// TIA Portal V17 export
// export: Created 2025-07-01T14:26:11.2068104Z, ExportSetting WithDefaults, DisplayName Totally Integrated Automation Portal, DisplayVersion V17 Update 8, DisplayName TIA Portal Openness, DisplayVersion V17 Update 8, DisplayName TIA Portal Version Control Interface, DisplayVersion V17, DisplayName SINAMICS Startdrive Advanced, DisplayVersion V17 SP2, DisplayName SINAMICS Startdrive G110M, G120, G120C, G120D, G120P, G115D, DisplayVersion V17 SP2, DisplayName SINAMICS Startdrive G130, G150, S120, S150, SINAMICS MV, S210, DisplayVersion V17 SP2, DisplayName STEP 7 Professional, DisplayVersion V17 Update 8, DisplayName SINUMERIK ONE STEP 7 Toolbox, DisplayVersion V17 Update 12, DisplayName SINUMERIK ONE PLC Basic Program Plus, DisplayVersion V17 Update 12, DisplayName SINUMERIK 840D sl STEP 7 Toolbox, DisplayVersion V17 Update 12, DisplayName STEP 7 Safety, DisplayVersion V17 Update 6, DisplayName WinCC Advanced, DisplayVersion V17 Update 8
FUNCTION "FC16014_METHOD_CALLS_U2_STA3_MEAS" : Void   // FC16014, LAD
{ S7_Optimized_Access := 'FALSE' }
VERSION : 0.1
// STATUS VALUES:
// 0 = IDLE
// 1 = CALIBRATING
// 2 = ANALYZING DISTANCE
// 3 = ANALYZING LAYER THICKNESS
// -1 = ERROR
// stored: AutoNumber false, IsIECCheckEnabled false, SetENOAutomatically false, UDAEnableTagReadback false
   VAR_TEMP
      AUX_WSTRING_PART_ID_STA3 : WString;
      AUX_WCHARS : Array[0..63] of WChar;
      index : Int;
      ALARM_AUX : Bool;
      TEMP_PULSE : Bool;
      STATUS_BLKMOV : Int;   // STATUS BLKMOV
      ZERO : Int;
   END_VAR
   VAR CONSTANT
      VERSIONS_MAJOR : UInt := 2;
      VERSIONS_MINOR : UInt;
      FC_NUMBER : DInt := 16014;
   END_VAR
   VAR_TEMP   // added for the SCL form of the ladder/FBD networks
      _w1 : Bool;
      _w2 : Bool;
      _w3 : Bool;
      _s5time1 : S5Time;
      _w4 : Bool;
   END_VAR
BEGIN

REGION Network 1: ZERO
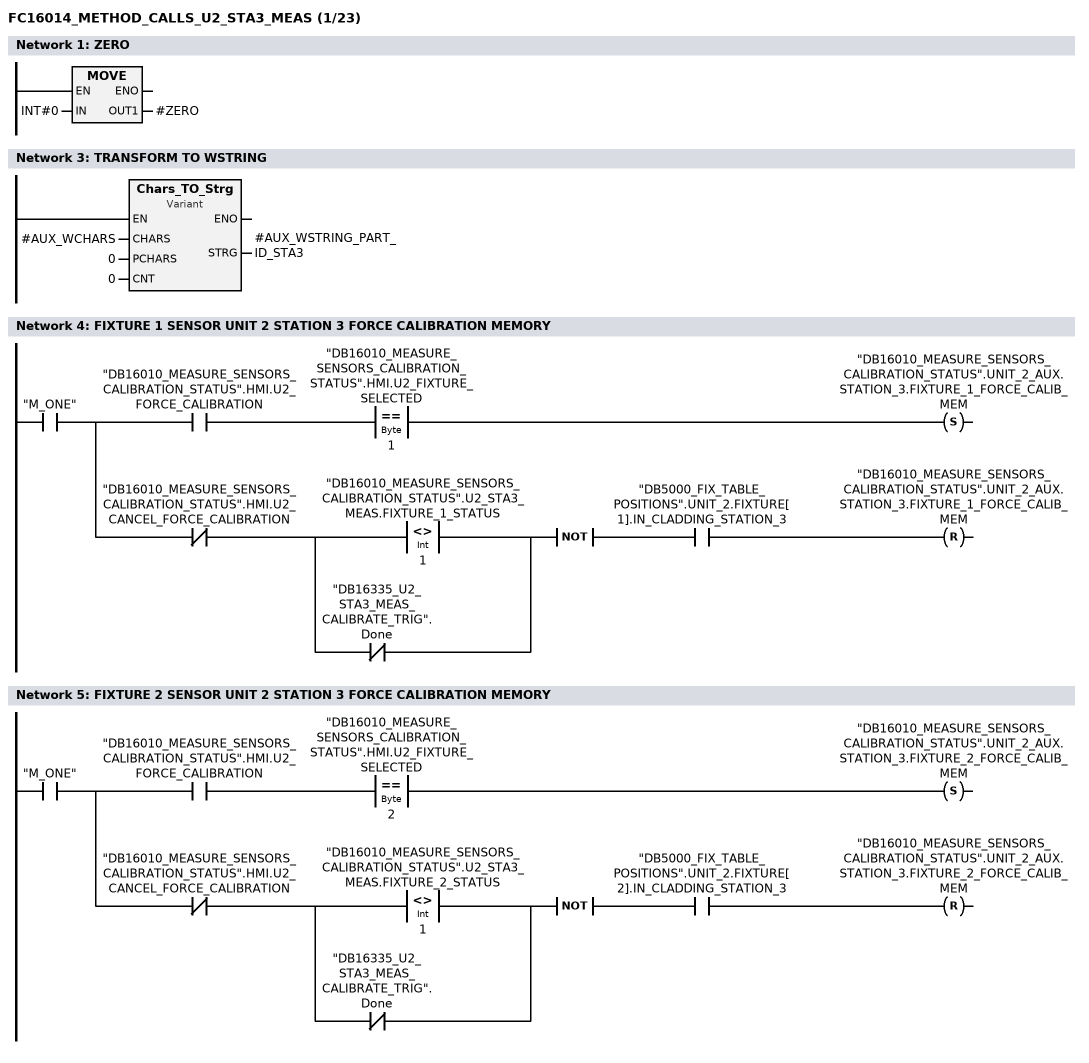
   RUNG wire#powerrail
      { S7_GenerateENO := "TRUE" } Move(in := INT#0, out1 => #ZERO)
   END_RUNG
   // the same network as SCL:
   #ZERO := INT#0;
END_REGION

REGION Network 2 (SCL): TRANSFORM TO WCHARS
   FOR #index := 0 TO 63 DO
       #AUX_WCHARS[#index] := CHAR_TO_WCHAR("DB8000_PART_STATUS".UNIT_2.STATION_3.PART_A.PART_ID[#index]);
   END_FOR;
END_REGION

REGION Network 3: TRANSFORM TO WSTRING
   RUNG wire#powerrail
      { S7_Templates := "[ptr_type := Variant, str_type := WString]" } Chars_TO_Strg(Chars := #AUX_WCHARS, pChars := 0, Cnt := 0, Strg => #AUX_WSTRING_PART_ID_STA3)
   END_RUNG
   // the same network as SCL:
   Chars_TO_Strg(Chars := #AUX_WCHARS, pChars := 0, Cnt := 0, Strg => #AUX_WSTRING_PART_ID_STA3);
END_REGION

REGION Network 4: FIXTURE 1 SENSOR UNIT 2 STATION 3 FORCE CALIBRATION MEMORY
   RUNG wire#powerrail
      Contact( "M_ONE" )
      wire#w1
      Contact( "DB16010_MEASURE_SENSORS_CALIBRATION_STATUS".HMI.U2_FORCE_CALIBRATION )
      { S7_Templates := "SrcType := Byte" } EQ_Contact(in1 := "DB16010_MEASURE_SENSORS_CALIBRATION_STATUS".HMI.U2_FIXTURE_SELECTED, in2 := 1)
      S_Coil( "DB16010_MEASURE_SENSORS_CALIBRATION_STATUS".UNIT_2_AUX.STATION_3.FIXTURE_1_FORCE_CALIB_MEM )
   END_RUNG
   RUNG wire#w1
      I_Contact( "DB16010_MEASURE_SENSORS_CALIBRATION_STATUS".HMI.U2_CANCEL_FORCE_CALIBRATION )
      wire#w2
      { S7_Templates := "SrcType := Int" } NE_Contact(in1 := "DB16010_MEASURE_SENSORS_CALIBRATION_STATUS".U2_STA3_MEAS.FIXTURE_1_STATUS, in2 := 1)
      wire#w3
      Not()
      Contact( "DB5000_FIX_TABLE_POSITIONS".UNIT_2.FIXTURE[1].IN_CLADDING_STATION_3 )
      R_Coil( "DB16010_MEASURE_SENSORS_CALIBRATION_STATUS".UNIT_2_AUX.STATION_3.FIXTURE_1_FORCE_CALIB_MEM )
   END_RUNG
   RUNG wire#w2
      I_Contact( "DB16335_U2_STA3_MEAS_CALIBRATE_TRIG".Done )
   END_RUNG wire#w3
   // the same network as SCL:
   IF "M_ONE" AND "DB16010_MEASURE_SENSORS_CALIBRATION_STATUS".HMI.U2_FORCE_CALIBRATION AND ("DB16010_MEASURE_SENSORS_CALIBRATION_STATUS".HMI.U2_FIXTURE_SELECTED = 1) THEN
       "DB16010_MEASURE_SENSORS_CALIBRATION_STATUS".UNIT_2_AUX.STATION_3.FIXTURE_1_FORCE_CALIB_MEM := TRUE;
   END_IF;
   IF NOT ("M_ONE" AND NOT "DB16010_MEASURE_SENSORS_CALIBRATION_STATUS".HMI.U2_CANCEL_FORCE_CALIBRATION AND (("DB16010_MEASURE_SENSORS_CALIBRATION_STATUS".U2_STA3_MEAS.FIXTURE_1_STATUS <> 1) OR NOT "DB16335_U2_STA3_MEAS_CALIBRATE_TRIG".Done)) AND "DB5000_FIX_TABLE_POSITIONS".UNIT_2.FIXTURE[1].IN_CLADDING_STATION_3 THEN
       "DB16010_MEASURE_SENSORS_CALIBRATION_STATUS".UNIT_2_AUX.STATION_3.FIXTURE_1_FORCE_CALIB_MEM := FALSE;
   END_IF;
END_REGION

REGION Network 5: FIXTURE 2 SENSOR UNIT 2 STATION 3 FORCE CALIBRATION MEMORY
   RUNG wire#powerrail
      Contact( "M_ONE" )
      wire#w1
      Contact( "DB16010_MEASURE_SENSORS_CALIBRATION_STATUS".HMI.U2_FORCE_CALIBRATION )
      { S7_Templates := "SrcType := Byte" } EQ_Contact(in1 := "DB16010_MEASURE_SENSORS_CALIBRATION_STATUS".HMI.U2_FIXTURE_SELECTED, in2 := 2)
      S_Coil( "DB16010_MEASURE_SENSORS_CALIBRATION_STATUS".UNIT_2_AUX.STATION_3.FIXTURE_2_FORCE_CALIB_MEM )
   END_RUNG
   RUNG wire#w1
      I_Contact( "DB16010_MEASURE_SENSORS_CALIBRATION_STATUS".HMI.U2_CANCEL_FORCE_CALIBRATION )
      wire#w2
      { S7_Templates := "SrcType := Int" } NE_Contact(in1 := "DB16010_MEASURE_SENSORS_CALIBRATION_STATUS".U2_STA3_MEAS.FIXTURE_2_STATUS, in2 := 1)
      wire#w3
      Not()
      Contact( "DB5000_FIX_TABLE_POSITIONS".UNIT_2.FIXTURE[2].IN_CLADDING_STATION_3 )
      R_Coil( "DB16010_MEASURE_SENSORS_CALIBRATION_STATUS".UNIT_2_AUX.STATION_3.FIXTURE_2_FORCE_CALIB_MEM )
   END_RUNG
   RUNG wire#w2
      I_Contact( "DB16335_U2_STA3_MEAS_CALIBRATE_TRIG".Done )
   END_RUNG wire#w3
   // the same network as SCL:
   IF "M_ONE" AND "DB16010_MEASURE_SENSORS_CALIBRATION_STATUS".HMI.U2_FORCE_CALIBRATION AND ("DB16010_MEASURE_SENSORS_CALIBRATION_STATUS".HMI.U2_FIXTURE_SELECTED = 2) THEN
       "DB16010_MEASURE_SENSORS_CALIBRATION_STATUS".UNIT_2_AUX.STATION_3.FIXTURE_2_FORCE_CALIB_MEM := TRUE;
   END_IF;
   IF NOT ("M_ONE" AND NOT "DB16010_MEASURE_SENSORS_CALIBRATION_STATUS".HMI.U2_CANCEL_FORCE_CALIBRATION AND (("DB16010_MEASURE_SENSORS_CALIBRATION_STATUS".U2_STA3_MEAS.FIXTURE_2_STATUS <> 1) OR NOT "DB16335_U2_STA3_MEAS_CALIBRATE_TRIG".Done)) AND "DB5000_FIX_TABLE_POSITIONS".UNIT_2.FIXTURE[2].IN_CLADDING_STATION_3 THEN
       "DB16010_MEASURE_SENSORS_CALIBRATION_STATUS".UNIT_2_AUX.STATION_3.FIXTURE_2_FORCE_CALIB_MEM := FALSE;
   END_IF;
END_REGION

REGION Network 6: FIXTURE 3 SENSOR UNIT 2 STATION 3 FORCE CALIBRATION MEMORY
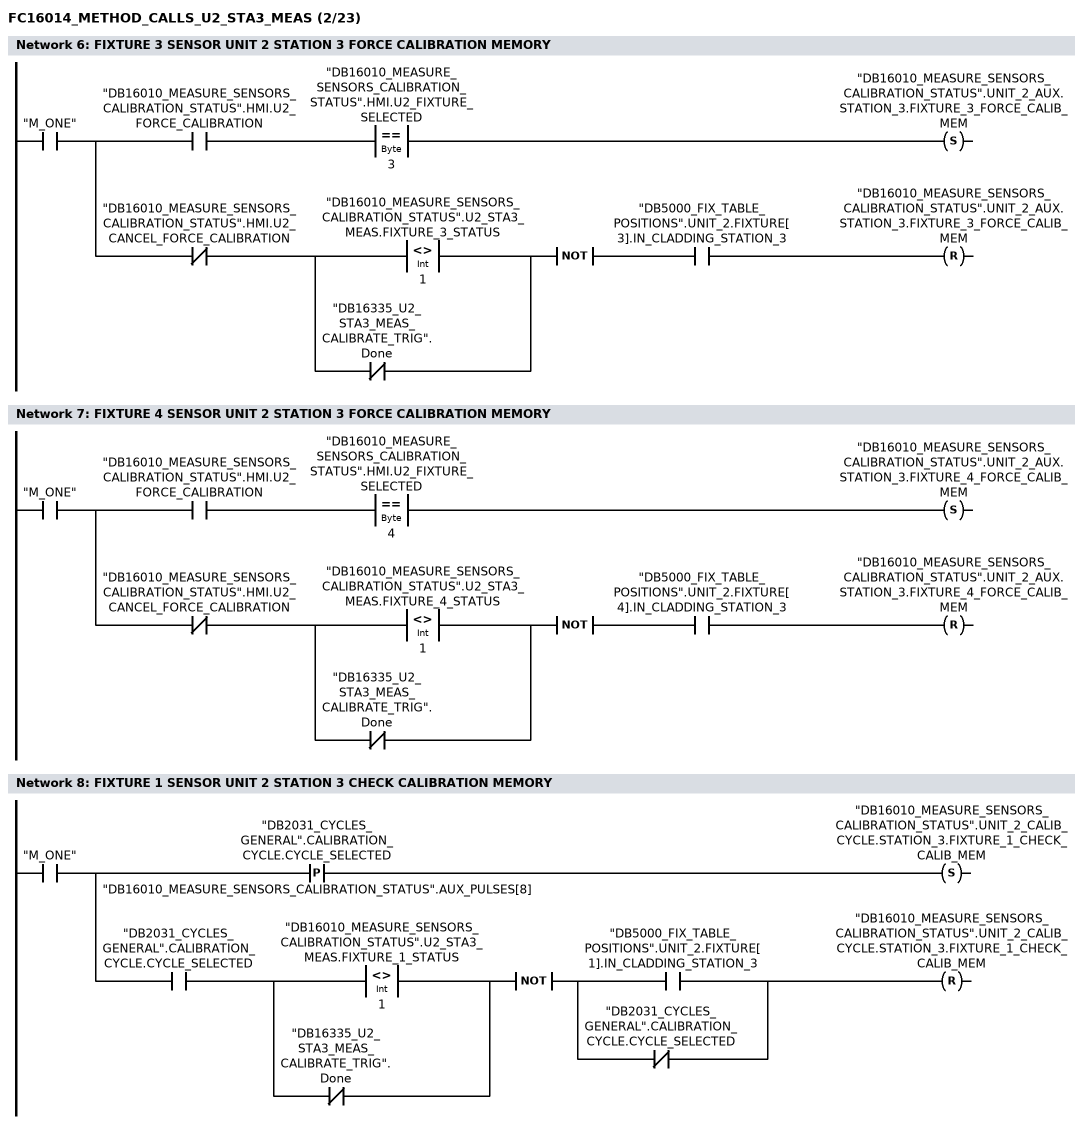
   RUNG wire#powerrail
      Contact( "M_ONE" )
      wire#w1
      Contact( "DB16010_MEASURE_SENSORS_CALIBRATION_STATUS".HMI.U2_FORCE_CALIBRATION )
      { S7_Templates := "SrcType := Byte" } EQ_Contact(in1 := "DB16010_MEASURE_SENSORS_CALIBRATION_STATUS".HMI.U2_FIXTURE_SELECTED, in2 := 3)
      S_Coil( "DB16010_MEASURE_SENSORS_CALIBRATION_STATUS".UNIT_2_AUX.STATION_3.FIXTURE_3_FORCE_CALIB_MEM )
   END_RUNG
   RUNG wire#w1
      I_Contact( "DB16010_MEASURE_SENSORS_CALIBRATION_STATUS".HMI.U2_CANCEL_FORCE_CALIBRATION )
      wire#w2
      { S7_Templates := "SrcType := Int" } NE_Contact(in1 := "DB16010_MEASURE_SENSORS_CALIBRATION_STATUS".U2_STA3_MEAS.FIXTURE_3_STATUS, in2 := 1)
      wire#w3
      Not()
      Contact( "DB5000_FIX_TABLE_POSITIONS".UNIT_2.FIXTURE[3].IN_CLADDING_STATION_3 )
      R_Coil( "DB16010_MEASURE_SENSORS_CALIBRATION_STATUS".UNIT_2_AUX.STATION_3.FIXTURE_3_FORCE_CALIB_MEM )
   END_RUNG
   RUNG wire#w2
      I_Contact( "DB16335_U2_STA3_MEAS_CALIBRATE_TRIG".Done )
   END_RUNG wire#w3
   // the same network as SCL:
   IF "M_ONE" AND "DB16010_MEASURE_SENSORS_CALIBRATION_STATUS".HMI.U2_FORCE_CALIBRATION AND ("DB16010_MEASURE_SENSORS_CALIBRATION_STATUS".HMI.U2_FIXTURE_SELECTED = 3) THEN
       "DB16010_MEASURE_SENSORS_CALIBRATION_STATUS".UNIT_2_AUX.STATION_3.FIXTURE_3_FORCE_CALIB_MEM := TRUE;
   END_IF;
   IF NOT ("M_ONE" AND NOT "DB16010_MEASURE_SENSORS_CALIBRATION_STATUS".HMI.U2_CANCEL_FORCE_CALIBRATION AND (("DB16010_MEASURE_SENSORS_CALIBRATION_STATUS".U2_STA3_MEAS.FIXTURE_3_STATUS <> 1) OR NOT "DB16335_U2_STA3_MEAS_CALIBRATE_TRIG".Done)) AND "DB5000_FIX_TABLE_POSITIONS".UNIT_2.FIXTURE[3].IN_CLADDING_STATION_3 THEN
       "DB16010_MEASURE_SENSORS_CALIBRATION_STATUS".UNIT_2_AUX.STATION_3.FIXTURE_3_FORCE_CALIB_MEM := FALSE;
   END_IF;
END_REGION

REGION Network 7: FIXTURE 4 SENSOR UNIT 2 STATION 3 FORCE CALIBRATION MEMORY
   RUNG wire#powerrail
      Contact( "M_ONE" )
      wire#w1
      Contact( "DB16010_MEASURE_SENSORS_CALIBRATION_STATUS".HMI.U2_FORCE_CALIBRATION )
      { S7_Templates := "SrcType := Byte" } EQ_Contact(in1 := "DB16010_MEASURE_SENSORS_CALIBRATION_STATUS".HMI.U2_FIXTURE_SELECTED, in2 := 4)
      S_Coil( "DB16010_MEASURE_SENSORS_CALIBRATION_STATUS".UNIT_2_AUX.STATION_3.FIXTURE_4_FORCE_CALIB_MEM )
   END_RUNG
   RUNG wire#w1
      I_Contact( "DB16010_MEASURE_SENSORS_CALIBRATION_STATUS".HMI.U2_CANCEL_FORCE_CALIBRATION )
      wire#w2
      { S7_Templates := "SrcType := Int" } NE_Contact(in1 := "DB16010_MEASURE_SENSORS_CALIBRATION_STATUS".U2_STA3_MEAS.FIXTURE_4_STATUS, in2 := 1)
      wire#w3
      Not()
      Contact( "DB5000_FIX_TABLE_POSITIONS".UNIT_2.FIXTURE[4].IN_CLADDING_STATION_3 )
      R_Coil( "DB16010_MEASURE_SENSORS_CALIBRATION_STATUS".UNIT_2_AUX.STATION_3.FIXTURE_4_FORCE_CALIB_MEM )
   END_RUNG
   RUNG wire#w2
      I_Contact( "DB16335_U2_STA3_MEAS_CALIBRATE_TRIG".Done )
   END_RUNG wire#w3
   // the same network as SCL:
   IF "M_ONE" AND "DB16010_MEASURE_SENSORS_CALIBRATION_STATUS".HMI.U2_FORCE_CALIBRATION AND ("DB16010_MEASURE_SENSORS_CALIBRATION_STATUS".HMI.U2_FIXTURE_SELECTED = 4) THEN
       "DB16010_MEASURE_SENSORS_CALIBRATION_STATUS".UNIT_2_AUX.STATION_3.FIXTURE_4_FORCE_CALIB_MEM := TRUE;
   END_IF;
   IF NOT ("M_ONE" AND NOT "DB16010_MEASURE_SENSORS_CALIBRATION_STATUS".HMI.U2_CANCEL_FORCE_CALIBRATION AND (("DB16010_MEASURE_SENSORS_CALIBRATION_STATUS".U2_STA3_MEAS.FIXTURE_4_STATUS <> 1) OR NOT "DB16335_U2_STA3_MEAS_CALIBRATE_TRIG".Done)) AND "DB5000_FIX_TABLE_POSITIONS".UNIT_2.FIXTURE[4].IN_CLADDING_STATION_3 THEN
       "DB16010_MEASURE_SENSORS_CALIBRATION_STATUS".UNIT_2_AUX.STATION_3.FIXTURE_4_FORCE_CALIB_MEM := FALSE;
   END_IF;
END_REGION

REGION Network 8: FIXTURE 1 SENSOR UNIT 2 STATION 3 CHECK CALIBRATION MEMORY
   RUNG wire#powerrail
      Contact( "M_ONE" )
      wire#w1
      P_Contact(operand := "DB2031_CYCLES_GENERAL".CALIBRATION_CYCLE.CYCLE_SELECTED, bit := "DB16010_MEASURE_SENSORS_CALIBRATION_STATUS".AUX_PULSES[8])
      S_Coil( "DB16010_MEASURE_SENSORS_CALIBRATION_STATUS".UNIT_2_CALIB_CYCLE.STATION_3.FIXTURE_1_CHECK_CALIB_MEM )
   END_RUNG
   RUNG wire#w1
      Contact( "DB2031_CYCLES_GENERAL".CALIBRATION_CYCLE.CYCLE_SELECTED )
      wire#w2
      { S7_Templates := "SrcType := Int" } NE_Contact(in1 := "DB16010_MEASURE_SENSORS_CALIBRATION_STATUS".U2_STA3_MEAS.FIXTURE_1_STATUS, in2 := 1)
      wire#w3
      Not()
      wire#w4
      Contact( "DB5000_FIX_TABLE_POSITIONS".UNIT_2.FIXTURE[1].IN_CLADDING_STATION_3 )
      wire#w5
      R_Coil( "DB16010_MEASURE_SENSORS_CALIBRATION_STATUS".UNIT_2_CALIB_CYCLE.STATION_3.FIXTURE_1_CHECK_CALIB_MEM )
   END_RUNG
   RUNG wire#w2
      I_Contact( "DB16335_U2_STA3_MEAS_CALIBRATE_TRIG".Done )
   END_RUNG wire#w3
   RUNG wire#w4
      I_Contact( "DB2031_CYCLES_GENERAL".CALIBRATION_CYCLE.CYCLE_SELECTED )
   END_RUNG wire#w5
   // the same network as SCL:
   #_w1 := "M_ONE" AND "DB2031_CYCLES_GENERAL".CALIBRATION_CYCLE.CYCLE_SELECTED AND NOT "DB16010_MEASURE_SENSORS_CALIBRATION_STATUS".AUX_PULSES[8];   // rising edge of "DB2031_CYCLES_GENERAL".CALIBRATION_CYCLE.CYCLE_SELECTED
   "DB16010_MEASURE_SENSORS_CALIBRATION_STATUS".AUX_PULSES[8] := "DB2031_CYCLES_GENERAL".CALIBRATION_CYCLE.CYCLE_SELECTED;
   IF #_w1 THEN
       "DB16010_MEASURE_SENSORS_CALIBRATION_STATUS".UNIT_2_CALIB_CYCLE.STATION_3.FIXTURE_1_CHECK_CALIB_MEM := TRUE;
   END_IF;
   IF NOT ("M_ONE" AND "DB2031_CYCLES_GENERAL".CALIBRATION_CYCLE.CYCLE_SELECTED AND (("DB16010_MEASURE_SENSORS_CALIBRATION_STATUS".U2_STA3_MEAS.FIXTURE_1_STATUS <> 1) OR NOT "DB16335_U2_STA3_MEAS_CALIBRATE_TRIG".Done)) AND ("DB5000_FIX_TABLE_POSITIONS".UNIT_2.FIXTURE[1].IN_CLADDING_STATION_3 OR NOT "DB2031_CYCLES_GENERAL".CALIBRATION_CYCLE.CYCLE_SELECTED) THEN
       "DB16010_MEASURE_SENSORS_CALIBRATION_STATUS".UNIT_2_CALIB_CYCLE.STATION_3.FIXTURE_1_CHECK_CALIB_MEM := FALSE;
   END_IF;
END_REGION

REGION Network 9: FIXTURE 2 SENSOR UNIT 2 STATION 3 CHECK CALIBRATION MEMORY
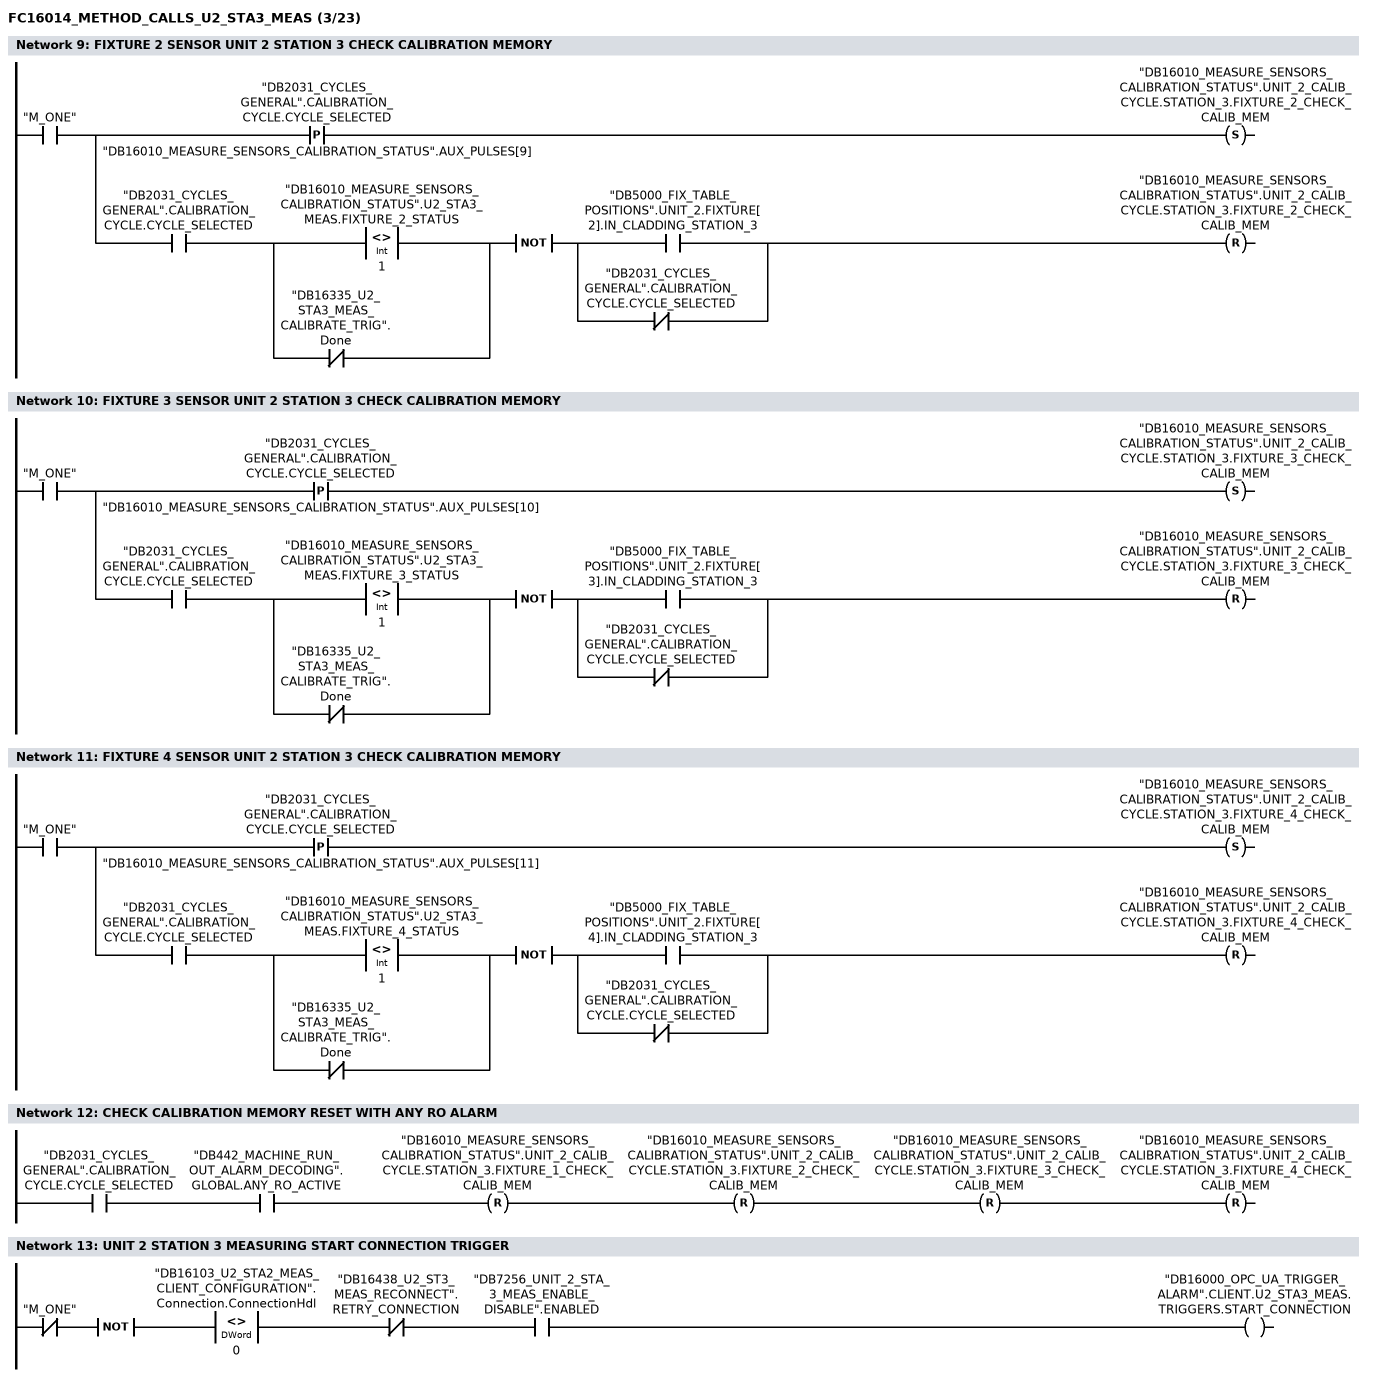
   RUNG wire#powerrail
      Contact( "M_ONE" )
      wire#w1
      P_Contact(operand := "DB2031_CYCLES_GENERAL".CALIBRATION_CYCLE.CYCLE_SELECTED, bit := "DB16010_MEASURE_SENSORS_CALIBRATION_STATUS".AUX_PULSES[9])
      S_Coil( "DB16010_MEASURE_SENSORS_CALIBRATION_STATUS".UNIT_2_CALIB_CYCLE.STATION_3.FIXTURE_2_CHECK_CALIB_MEM )
   END_RUNG
   RUNG wire#w1
      Contact( "DB2031_CYCLES_GENERAL".CALIBRATION_CYCLE.CYCLE_SELECTED )
      wire#w2
      { S7_Templates := "SrcType := Int" } NE_Contact(in1 := "DB16010_MEASURE_SENSORS_CALIBRATION_STATUS".U2_STA3_MEAS.FIXTURE_2_STATUS, in2 := 1)
      wire#w3
      Not()
      wire#w4
      Contact( "DB5000_FIX_TABLE_POSITIONS".UNIT_2.FIXTURE[2].IN_CLADDING_STATION_3 )
      wire#w5
      R_Coil( "DB16010_MEASURE_SENSORS_CALIBRATION_STATUS".UNIT_2_CALIB_CYCLE.STATION_3.FIXTURE_2_CHECK_CALIB_MEM )
   END_RUNG
   RUNG wire#w2
      I_Contact( "DB16335_U2_STA3_MEAS_CALIBRATE_TRIG".Done )
   END_RUNG wire#w3
   RUNG wire#w4
      I_Contact( "DB2031_CYCLES_GENERAL".CALIBRATION_CYCLE.CYCLE_SELECTED )
   END_RUNG wire#w5
   // the same network as SCL:
   #_w1 := "M_ONE" AND "DB2031_CYCLES_GENERAL".CALIBRATION_CYCLE.CYCLE_SELECTED AND NOT "DB16010_MEASURE_SENSORS_CALIBRATION_STATUS".AUX_PULSES[9];   // rising edge of "DB2031_CYCLES_GENERAL".CALIBRATION_CYCLE.CYCLE_SELECTED
   "DB16010_MEASURE_SENSORS_CALIBRATION_STATUS".AUX_PULSES[9] := "DB2031_CYCLES_GENERAL".CALIBRATION_CYCLE.CYCLE_SELECTED;
   IF #_w1 THEN
       "DB16010_MEASURE_SENSORS_CALIBRATION_STATUS".UNIT_2_CALIB_CYCLE.STATION_3.FIXTURE_2_CHECK_CALIB_MEM := TRUE;
   END_IF;
   IF NOT ("M_ONE" AND "DB2031_CYCLES_GENERAL".CALIBRATION_CYCLE.CYCLE_SELECTED AND (("DB16010_MEASURE_SENSORS_CALIBRATION_STATUS".U2_STA3_MEAS.FIXTURE_2_STATUS <> 1) OR NOT "DB16335_U2_STA3_MEAS_CALIBRATE_TRIG".Done)) AND ("DB5000_FIX_TABLE_POSITIONS".UNIT_2.FIXTURE[2].IN_CLADDING_STATION_3 OR NOT "DB2031_CYCLES_GENERAL".CALIBRATION_CYCLE.CYCLE_SELECTED) THEN
       "DB16010_MEASURE_SENSORS_CALIBRATION_STATUS".UNIT_2_CALIB_CYCLE.STATION_3.FIXTURE_2_CHECK_CALIB_MEM := FALSE;
   END_IF;
END_REGION

REGION Network 10: FIXTURE 3 SENSOR UNIT 2 STATION 3 CHECK CALIBRATION MEMORY
   RUNG wire#powerrail
      Contact( "M_ONE" )
      wire#w1
      P_Contact(operand := "DB2031_CYCLES_GENERAL".CALIBRATION_CYCLE.CYCLE_SELECTED, bit := "DB16010_MEASURE_SENSORS_CALIBRATION_STATUS".AUX_PULSES[10])
      S_Coil( "DB16010_MEASURE_SENSORS_CALIBRATION_STATUS".UNIT_2_CALIB_CYCLE.STATION_3.FIXTURE_3_CHECK_CALIB_MEM )
   END_RUNG
   RUNG wire#w1
      Contact( "DB2031_CYCLES_GENERAL".CALIBRATION_CYCLE.CYCLE_SELECTED )
      wire#w2
      { S7_Templates := "SrcType := Int" } NE_Contact(in1 := "DB16010_MEASURE_SENSORS_CALIBRATION_STATUS".U2_STA3_MEAS.FIXTURE_3_STATUS, in2 := 1)
      wire#w3
      Not()
      wire#w4
      Contact( "DB5000_FIX_TABLE_POSITIONS".UNIT_2.FIXTURE[3].IN_CLADDING_STATION_3 )
      wire#w5
      R_Coil( "DB16010_MEASURE_SENSORS_CALIBRATION_STATUS".UNIT_2_CALIB_CYCLE.STATION_3.FIXTURE_3_CHECK_CALIB_MEM )
   END_RUNG
   RUNG wire#w2
      I_Contact( "DB16335_U2_STA3_MEAS_CALIBRATE_TRIG".Done )
   END_RUNG wire#w3
   RUNG wire#w4
      I_Contact( "DB2031_CYCLES_GENERAL".CALIBRATION_CYCLE.CYCLE_SELECTED )
   END_RUNG wire#w5
   // the same network as SCL:
   #_w1 := "M_ONE" AND "DB2031_CYCLES_GENERAL".CALIBRATION_CYCLE.CYCLE_SELECTED AND NOT "DB16010_MEASURE_SENSORS_CALIBRATION_STATUS".AUX_PULSES[10];   // rising edge of "DB2031_CYCLES_GENERAL".CALIBRATION_CYCLE.CYCLE_SELECTED
   "DB16010_MEASURE_SENSORS_CALIBRATION_STATUS".AUX_PULSES[10] := "DB2031_CYCLES_GENERAL".CALIBRATION_CYCLE.CYCLE_SELECTED;
   IF #_w1 THEN
       "DB16010_MEASURE_SENSORS_CALIBRATION_STATUS".UNIT_2_CALIB_CYCLE.STATION_3.FIXTURE_3_CHECK_CALIB_MEM := TRUE;
   END_IF;
   IF NOT ("M_ONE" AND "DB2031_CYCLES_GENERAL".CALIBRATION_CYCLE.CYCLE_SELECTED AND (("DB16010_MEASURE_SENSORS_CALIBRATION_STATUS".U2_STA3_MEAS.FIXTURE_3_STATUS <> 1) OR NOT "DB16335_U2_STA3_MEAS_CALIBRATE_TRIG".Done)) AND ("DB5000_FIX_TABLE_POSITIONS".UNIT_2.FIXTURE[3].IN_CLADDING_STATION_3 OR NOT "DB2031_CYCLES_GENERAL".CALIBRATION_CYCLE.CYCLE_SELECTED) THEN
       "DB16010_MEASURE_SENSORS_CALIBRATION_STATUS".UNIT_2_CALIB_CYCLE.STATION_3.FIXTURE_3_CHECK_CALIB_MEM := FALSE;
   END_IF;
END_REGION

REGION Network 11: FIXTURE 4 SENSOR UNIT 2 STATION 3 CHECK CALIBRATION MEMORY
   RUNG wire#powerrail
      Contact( "M_ONE" )
      wire#w1
      P_Contact(operand := "DB2031_CYCLES_GENERAL".CALIBRATION_CYCLE.CYCLE_SELECTED, bit := "DB16010_MEASURE_SENSORS_CALIBRATION_STATUS".AUX_PULSES[11])
      S_Coil( "DB16010_MEASURE_SENSORS_CALIBRATION_STATUS".UNIT_2_CALIB_CYCLE.STATION_3.FIXTURE_4_CHECK_CALIB_MEM )
   END_RUNG
   RUNG wire#w1
      Contact( "DB2031_CYCLES_GENERAL".CALIBRATION_CYCLE.CYCLE_SELECTED )
      wire#w2
      { S7_Templates := "SrcType := Int" } NE_Contact(in1 := "DB16010_MEASURE_SENSORS_CALIBRATION_STATUS".U2_STA3_MEAS.FIXTURE_4_STATUS, in2 := 1)
      wire#w3
      Not()
      wire#w4
      Contact( "DB5000_FIX_TABLE_POSITIONS".UNIT_2.FIXTURE[4].IN_CLADDING_STATION_3 )
      wire#w5
      R_Coil( "DB16010_MEASURE_SENSORS_CALIBRATION_STATUS".UNIT_2_CALIB_CYCLE.STATION_3.FIXTURE_4_CHECK_CALIB_MEM )
   END_RUNG
   RUNG wire#w2
      I_Contact( "DB16335_U2_STA3_MEAS_CALIBRATE_TRIG".Done )
   END_RUNG wire#w3
   RUNG wire#w4
      I_Contact( "DB2031_CYCLES_GENERAL".CALIBRATION_CYCLE.CYCLE_SELECTED )
   END_RUNG wire#w5
   // the same network as SCL:
   #_w1 := "M_ONE" AND "DB2031_CYCLES_GENERAL".CALIBRATION_CYCLE.CYCLE_SELECTED AND NOT "DB16010_MEASURE_SENSORS_CALIBRATION_STATUS".AUX_PULSES[11];   // rising edge of "DB2031_CYCLES_GENERAL".CALIBRATION_CYCLE.CYCLE_SELECTED
   "DB16010_MEASURE_SENSORS_CALIBRATION_STATUS".AUX_PULSES[11] := "DB2031_CYCLES_GENERAL".CALIBRATION_CYCLE.CYCLE_SELECTED;
   IF #_w1 THEN
       "DB16010_MEASURE_SENSORS_CALIBRATION_STATUS".UNIT_2_CALIB_CYCLE.STATION_3.FIXTURE_4_CHECK_CALIB_MEM := TRUE;
   END_IF;
   IF NOT ("M_ONE" AND "DB2031_CYCLES_GENERAL".CALIBRATION_CYCLE.CYCLE_SELECTED AND (("DB16010_MEASURE_SENSORS_CALIBRATION_STATUS".U2_STA3_MEAS.FIXTURE_4_STATUS <> 1) OR NOT "DB16335_U2_STA3_MEAS_CALIBRATE_TRIG".Done)) AND ("DB5000_FIX_TABLE_POSITIONS".UNIT_2.FIXTURE[4].IN_CLADDING_STATION_3 OR NOT "DB2031_CYCLES_GENERAL".CALIBRATION_CYCLE.CYCLE_SELECTED) THEN
       "DB16010_MEASURE_SENSORS_CALIBRATION_STATUS".UNIT_2_CALIB_CYCLE.STATION_3.FIXTURE_4_CHECK_CALIB_MEM := FALSE;
   END_IF;
END_REGION

REGION Network 12: CHECK CALIBRATION MEMORY RESET WITH ANY RO ALARM
   RUNG wire#powerrail
      Contact( "DB2031_CYCLES_GENERAL".CALIBRATION_CYCLE.CYCLE_SELECTED )
      Contact( "DB442_MACHINE_RUN_OUT_ALARM_DECODING".GLOBAL.ANY_RO_ACTIVE )
      R_Coil( "DB16010_MEASURE_SENSORS_CALIBRATION_STATUS".UNIT_2_CALIB_CYCLE.STATION_3.FIXTURE_1_CHECK_CALIB_MEM )
      R_Coil( "DB16010_MEASURE_SENSORS_CALIBRATION_STATUS".UNIT_2_CALIB_CYCLE.STATION_3.FIXTURE_2_CHECK_CALIB_MEM )
      R_Coil( "DB16010_MEASURE_SENSORS_CALIBRATION_STATUS".UNIT_2_CALIB_CYCLE.STATION_3.FIXTURE_3_CHECK_CALIB_MEM )
      R_Coil( "DB16010_MEASURE_SENSORS_CALIBRATION_STATUS".UNIT_2_CALIB_CYCLE.STATION_3.FIXTURE_4_CHECK_CALIB_MEM )
   END_RUNG
   // the same network as SCL:
   IF "DB2031_CYCLES_GENERAL".CALIBRATION_CYCLE.CYCLE_SELECTED AND "DB442_MACHINE_RUN_OUT_ALARM_DECODING".GLOBAL.ANY_RO_ACTIVE THEN
       "DB16010_MEASURE_SENSORS_CALIBRATION_STATUS".UNIT_2_CALIB_CYCLE.STATION_3.FIXTURE_1_CHECK_CALIB_MEM := FALSE;
       "DB16010_MEASURE_SENSORS_CALIBRATION_STATUS".UNIT_2_CALIB_CYCLE.STATION_3.FIXTURE_2_CHECK_CALIB_MEM := FALSE;
       "DB16010_MEASURE_SENSORS_CALIBRATION_STATUS".UNIT_2_CALIB_CYCLE.STATION_3.FIXTURE_3_CHECK_CALIB_MEM := FALSE;
       "DB16010_MEASURE_SENSORS_CALIBRATION_STATUS".UNIT_2_CALIB_CYCLE.STATION_3.FIXTURE_4_CHECK_CALIB_MEM := FALSE;
   END_IF;
END_REGION

REGION Network 13: UNIT 2 STATION 3 MEASURING START CONNECTION TRIGGER
   RUNG wire#powerrail
      I_Contact( "M_ONE" )
      Not()
      { S7_Templates := "SrcType := DWord" } NE_Contact(in1 := "DB16103_U2_STA2_MEAS_CLIENT_CONFIGURATION".Connection.ConnectionHdl, in2 := 0)
      I_Contact( "DB16438_U2_ST3_MEAS_RECONNECT".RETRY_CONNECTION )
      Contact( "DB7256_UNIT_2_STA_3_MEAS_ENABLE_DISABLE".ENABLED )
      Coil( "DB16000_OPC_UA_TRIGGER_ALARM".CLIENT.U2_STA3_MEAS.TRIGGERS.START_CONNECTION )
   END_RUNG
   // the same network as SCL:
   "DB16000_OPC_UA_TRIGGER_ALARM".CLIENT.U2_STA3_MEAS.TRIGGERS.START_CONNECTION := NOT (NOT "M_ONE") AND ("DB16103_U2_STA2_MEAS_CLIENT_CONFIGURATION".Connection.ConnectionHdl <> 0) AND NOT "DB16438_U2_ST3_MEAS_RECONNECT".RETRY_CONNECTION AND "DB7256_UNIT_2_STA_3_MEAS_ENABLE_DISABLE".ENABLED;
END_REGION

REGION Network 14: UNIT 2 STATION 3 MEASURING GET INDEX LIST TRIGGER
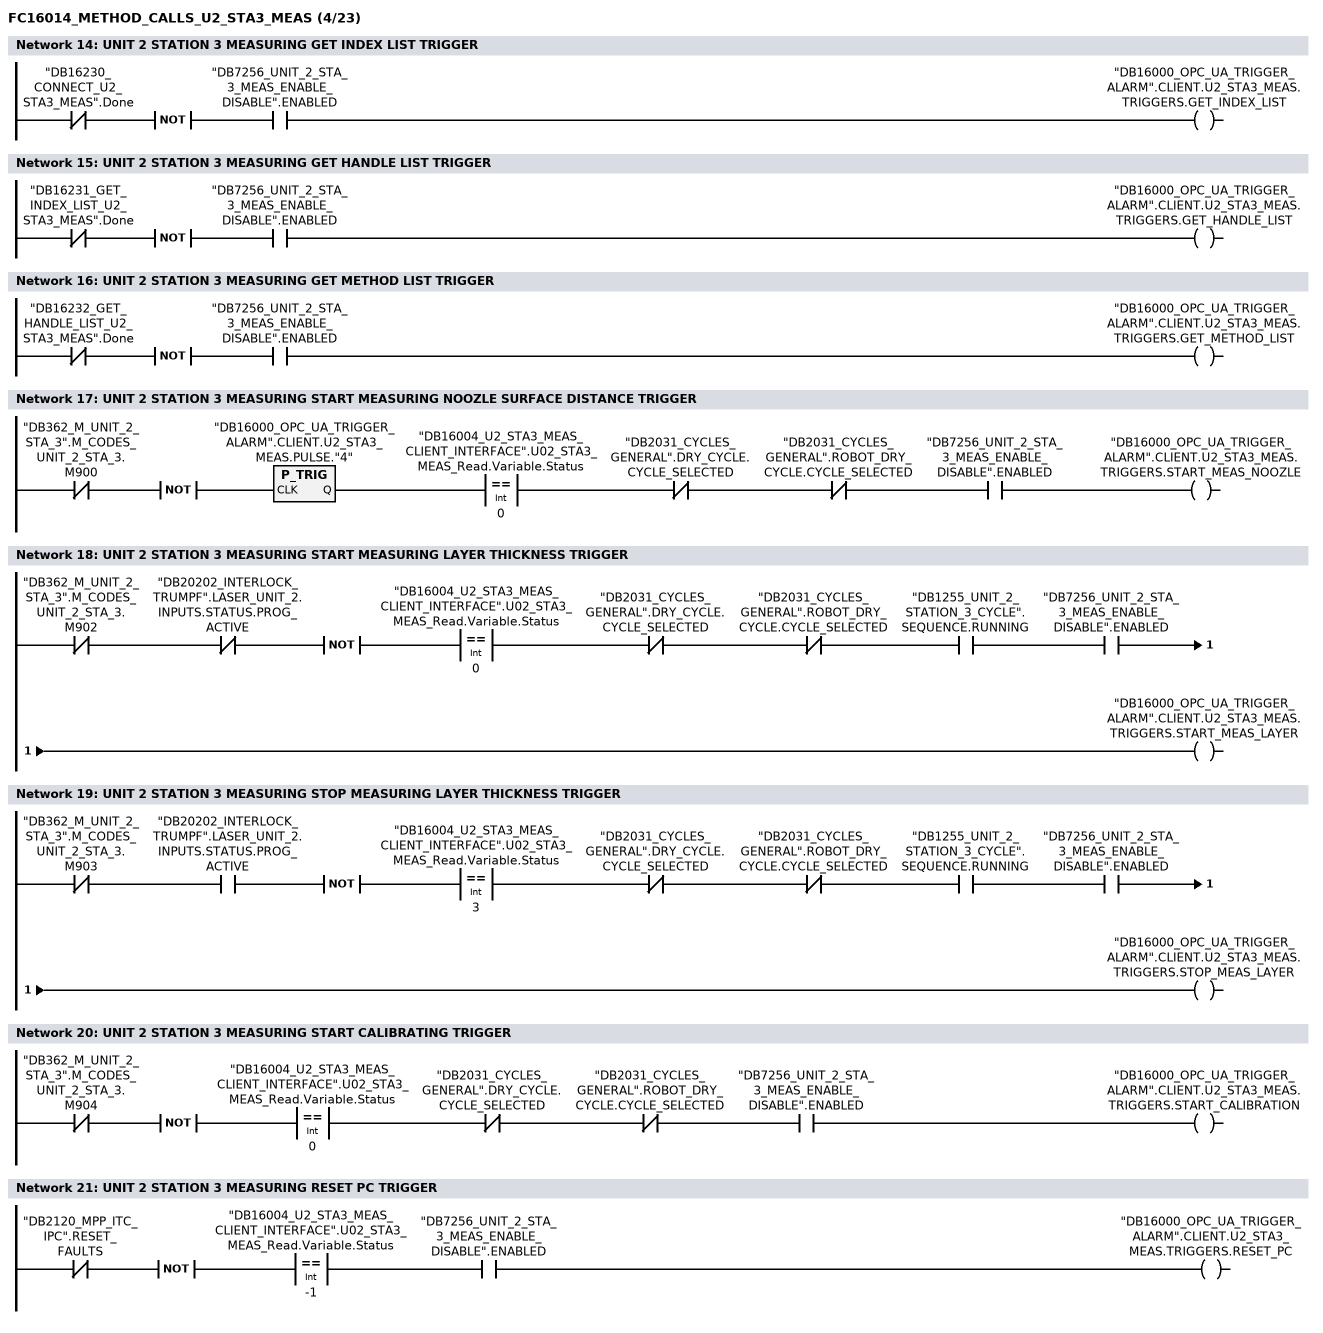
   RUNG wire#powerrail
      I_Contact( "DB16230_CONNECT_U2_STA3_MEAS".Done )
      Not()
      Contact( "DB7256_UNIT_2_STA_3_MEAS_ENABLE_DISABLE".ENABLED )
      Coil( "DB16000_OPC_UA_TRIGGER_ALARM".CLIENT.U2_STA3_MEAS.TRIGGERS.GET_INDEX_LIST )
   END_RUNG
   // the same network as SCL:
   "DB16000_OPC_UA_TRIGGER_ALARM".CLIENT.U2_STA3_MEAS.TRIGGERS.GET_INDEX_LIST := NOT (NOT "DB16230_CONNECT_U2_STA3_MEAS".Done) AND "DB7256_UNIT_2_STA_3_MEAS_ENABLE_DISABLE".ENABLED;
END_REGION

REGION Network 15: UNIT 2 STATION 3 MEASURING GET HANDLE LIST TRIGGER
   RUNG wire#powerrail
      I_Contact( "DB16231_GET_INDEX_LIST_U2_STA3_MEAS".Done )
      Not()
      Contact( "DB7256_UNIT_2_STA_3_MEAS_ENABLE_DISABLE".ENABLED )
      Coil( "DB16000_OPC_UA_TRIGGER_ALARM".CLIENT.U2_STA3_MEAS.TRIGGERS.GET_HANDLE_LIST )
   END_RUNG
   // the same network as SCL:
   "DB16000_OPC_UA_TRIGGER_ALARM".CLIENT.U2_STA3_MEAS.TRIGGERS.GET_HANDLE_LIST := NOT (NOT "DB16231_GET_INDEX_LIST_U2_STA3_MEAS".Done) AND "DB7256_UNIT_2_STA_3_MEAS_ENABLE_DISABLE".ENABLED;
END_REGION

REGION Network 16: UNIT 2 STATION 3 MEASURING GET METHOD LIST TRIGGER
   RUNG wire#powerrail
      I_Contact( "DB16232_GET_HANDLE_LIST_U2_STA3_MEAS".Done )
      Not()
      Contact( "DB7256_UNIT_2_STA_3_MEAS_ENABLE_DISABLE".ENABLED )
      Coil( "DB16000_OPC_UA_TRIGGER_ALARM".CLIENT.U2_STA3_MEAS.TRIGGERS.GET_METHOD_LIST )
   END_RUNG
   // the same network as SCL:
   "DB16000_OPC_UA_TRIGGER_ALARM".CLIENT.U2_STA3_MEAS.TRIGGERS.GET_METHOD_LIST := NOT (NOT "DB16232_GET_HANDLE_LIST_U2_STA3_MEAS".Done) AND "DB7256_UNIT_2_STA_3_MEAS_ENABLE_DISABLE".ENABLED;
END_REGION

REGION Network 17: UNIT 2 STATION 3 MEASURING START MEASURING NOOZLE SURFACE DISTANCE TRIGGER
   RUNG wire#powerrail
      I_Contact( "DB362_M_UNIT_2_STA_3".M_CODES_UNIT_2_STA_3.M900 )
      Not()
      P_Trig( "DB16000_OPC_UA_TRIGGER_ALARM".CLIENT.U2_STA3_MEAS.PULSE."4" )
      { S7_Templates := "SrcType := Int" } EQ_Contact(in1 := "DB16004_U2_STA3_MEAS_CLIENT_INTERFACE".U02_STA3_MEAS_Read.Variable.Status, in2 := 0)
      I_Contact( "DB2031_CYCLES_GENERAL".DRY_CYCLE.CYCLE_SELECTED )
      I_Contact( "DB2031_CYCLES_GENERAL".ROBOT_DRY_CYCLE.CYCLE_SELECTED )
      Contact( "DB7256_UNIT_2_STA_3_MEAS_ENABLE_DISABLE".ENABLED )
      Coil( "DB16000_OPC_UA_TRIGGER_ALARM".CLIENT.U2_STA3_MEAS.TRIGGERS.START_MEAS_NOOZLE )
   END_RUNG
   // the same network as SCL:
   #_w1 := NOT (NOT "DB362_M_UNIT_2_STA_3".M_CODES_UNIT_2_STA_3.M900) AND NOT "DB16000_OPC_UA_TRIGGER_ALARM".CLIENT.U2_STA3_MEAS.PULSE."4";   // rising edge
   "DB16000_OPC_UA_TRIGGER_ALARM".CLIENT.U2_STA3_MEAS.PULSE."4" := NOT (NOT "DB362_M_UNIT_2_STA_3".M_CODES_UNIT_2_STA_3.M900);
   "DB16000_OPC_UA_TRIGGER_ALARM".CLIENT.U2_STA3_MEAS.TRIGGERS.START_MEAS_NOOZLE := #_w1 AND ("DB16004_U2_STA3_MEAS_CLIENT_INTERFACE".U02_STA3_MEAS_Read.Variable.Status = 0) AND NOT "DB2031_CYCLES_GENERAL".DRY_CYCLE.CYCLE_SELECTED AND NOT "DB2031_CYCLES_GENERAL".ROBOT_DRY_CYCLE.CYCLE_SELECTED AND "DB7256_UNIT_2_STA_3_MEAS_ENABLE_DISABLE".ENABLED;
END_REGION

REGION Network 18: UNIT 2 STATION 3 MEASURING START MEASURING LAYER THICKNESS TRIGGER
   RUNG wire#powerrail
      I_Contact( "DB362_M_UNIT_2_STA_3".M_CODES_UNIT_2_STA_3.M902 )
      I_Contact( "DB20202_INTERLOCK_TRUMPF".LASER_UNIT_2.INPUTS.STATUS.PROG_ACTIVE )
      Not()
      { S7_Templates := "SrcType := Int" } EQ_Contact(in1 := "DB16004_U2_STA3_MEAS_CLIENT_INTERFACE".U02_STA3_MEAS_Read.Variable.Status, in2 := 0)
      I_Contact( "DB2031_CYCLES_GENERAL".DRY_CYCLE.CYCLE_SELECTED )
      I_Contact( "DB2031_CYCLES_GENERAL".ROBOT_DRY_CYCLE.CYCLE_SELECTED )
      Contact( "DB1255_UNIT_2_STATION_3_CYCLE".SEQUENCE.RUNNING )
      Contact( "DB7256_UNIT_2_STA_3_MEAS_ENABLE_DISABLE".ENABLED )
      Coil( "DB16000_OPC_UA_TRIGGER_ALARM".CLIENT.U2_STA3_MEAS.TRIGGERS.START_MEAS_LAYER )
   END_RUNG
   // the same network as SCL:
   "DB16000_OPC_UA_TRIGGER_ALARM".CLIENT.U2_STA3_MEAS.TRIGGERS.START_MEAS_LAYER := NOT (NOT "DB362_M_UNIT_2_STA_3".M_CODES_UNIT_2_STA_3.M902 AND NOT "DB20202_INTERLOCK_TRUMPF".LASER_UNIT_2.INPUTS.STATUS.PROG_ACTIVE) AND ("DB16004_U2_STA3_MEAS_CLIENT_INTERFACE".U02_STA3_MEAS_Read.Variable.Status = 0) AND NOT "DB2031_CYCLES_GENERAL".DRY_CYCLE.CYCLE_SELECTED AND NOT "DB2031_CYCLES_GENERAL".ROBOT_DRY_CYCLE.CYCLE_SELECTED AND "DB1255_UNIT_2_STATION_3_CYCLE".SEQUENCE.RUNNING AND "DB7256_UNIT_2_STA_3_MEAS_ENABLE_DISABLE".ENABLED;
END_REGION

REGION Network 19: UNIT 2 STATION 3 MEASURING STOP MEASURING LAYER THICKNESS TRIGGER
   RUNG wire#powerrail
      I_Contact( "DB362_M_UNIT_2_STA_3".M_CODES_UNIT_2_STA_3.M903 )
      Contact( "DB20202_INTERLOCK_TRUMPF".LASER_UNIT_2.INPUTS.STATUS.PROG_ACTIVE )
      Not()
      { S7_Templates := "SrcType := Int" } EQ_Contact(in1 := "DB16004_U2_STA3_MEAS_CLIENT_INTERFACE".U02_STA3_MEAS_Read.Variable.Status, in2 := 3)
      I_Contact( "DB2031_CYCLES_GENERAL".DRY_CYCLE.CYCLE_SELECTED )
      I_Contact( "DB2031_CYCLES_GENERAL".ROBOT_DRY_CYCLE.CYCLE_SELECTED )
      Contact( "DB1255_UNIT_2_STATION_3_CYCLE".SEQUENCE.RUNNING )
      Contact( "DB7256_UNIT_2_STA_3_MEAS_ENABLE_DISABLE".ENABLED )
      Coil( "DB16000_OPC_UA_TRIGGER_ALARM".CLIENT.U2_STA3_MEAS.TRIGGERS.STOP_MEAS_LAYER )
   END_RUNG
   // the same network as SCL:
   "DB16000_OPC_UA_TRIGGER_ALARM".CLIENT.U2_STA3_MEAS.TRIGGERS.STOP_MEAS_LAYER := NOT (NOT "DB362_M_UNIT_2_STA_3".M_CODES_UNIT_2_STA_3.M903 AND "DB20202_INTERLOCK_TRUMPF".LASER_UNIT_2.INPUTS.STATUS.PROG_ACTIVE) AND ("DB16004_U2_STA3_MEAS_CLIENT_INTERFACE".U02_STA3_MEAS_Read.Variable.Status = 3) AND NOT "DB2031_CYCLES_GENERAL".DRY_CYCLE.CYCLE_SELECTED AND NOT "DB2031_CYCLES_GENERAL".ROBOT_DRY_CYCLE.CYCLE_SELECTED AND "DB1255_UNIT_2_STATION_3_CYCLE".SEQUENCE.RUNNING AND "DB7256_UNIT_2_STA_3_MEAS_ENABLE_DISABLE".ENABLED;
END_REGION

REGION Network 20: UNIT 2 STATION 3 MEASURING START CALIBRATING TRIGGER
   RUNG wire#powerrail
      I_Contact( "DB362_M_UNIT_2_STA_3".M_CODES_UNIT_2_STA_3.M904 )
      Not()
      { S7_Templates := "SrcType := Int" } EQ_Contact(in1 := "DB16004_U2_STA3_MEAS_CLIENT_INTERFACE".U02_STA3_MEAS_Read.Variable.Status, in2 := 0)
      I_Contact( "DB2031_CYCLES_GENERAL".DRY_CYCLE.CYCLE_SELECTED )
      I_Contact( "DB2031_CYCLES_GENERAL".ROBOT_DRY_CYCLE.CYCLE_SELECTED )
      Contact( "DB7256_UNIT_2_STA_3_MEAS_ENABLE_DISABLE".ENABLED )
      Coil( "DB16000_OPC_UA_TRIGGER_ALARM".CLIENT.U2_STA3_MEAS.TRIGGERS.START_CALIBRATION )
   END_RUNG
   // the same network as SCL:
   "DB16000_OPC_UA_TRIGGER_ALARM".CLIENT.U2_STA3_MEAS.TRIGGERS.START_CALIBRATION := NOT (NOT "DB362_M_UNIT_2_STA_3".M_CODES_UNIT_2_STA_3.M904) AND ("DB16004_U2_STA3_MEAS_CLIENT_INTERFACE".U02_STA3_MEAS_Read.Variable.Status = 0) AND NOT "DB2031_CYCLES_GENERAL".DRY_CYCLE.CYCLE_SELECTED AND NOT "DB2031_CYCLES_GENERAL".ROBOT_DRY_CYCLE.CYCLE_SELECTED AND "DB7256_UNIT_2_STA_3_MEAS_ENABLE_DISABLE".ENABLED;
END_REGION

REGION Network 21: UNIT 2 STATION 3 MEASURING RESET PC TRIGGER
   RUNG wire#powerrail
      I_Contact( "DB2120_MPP_ITC_IPC".RESET_FAULTS )
      Not()
      { S7_Templates := "SrcType := Int" } EQ_Contact(in1 := "DB16004_U2_STA3_MEAS_CLIENT_INTERFACE".U02_STA3_MEAS_Read.Variable.Status, in2 := -1)
      Contact( "DB7256_UNIT_2_STA_3_MEAS_ENABLE_DISABLE".ENABLED )
      Coil( "DB16000_OPC_UA_TRIGGER_ALARM".CLIENT.U2_STA3_MEAS.TRIGGERS.RESET_PC )
   END_RUNG
   // the same network as SCL:
   "DB16000_OPC_UA_TRIGGER_ALARM".CLIENT.U2_STA3_MEAS.TRIGGERS.RESET_PC := NOT (NOT "DB2120_MPP_ITC_IPC".RESET_FAULTS) AND ("DB16004_U2_STA3_MEAS_CLIENT_INTERFACE".U02_STA3_MEAS_Read.Variable.Status = (-1)) AND "DB7256_UNIT_2_STA_3_MEAS_ENABLE_DISABLE".ENABLED;
END_REGION

REGION Network 22: UNIT 2 STATION 3 MEASURING READ VARIABLES TRIGGER
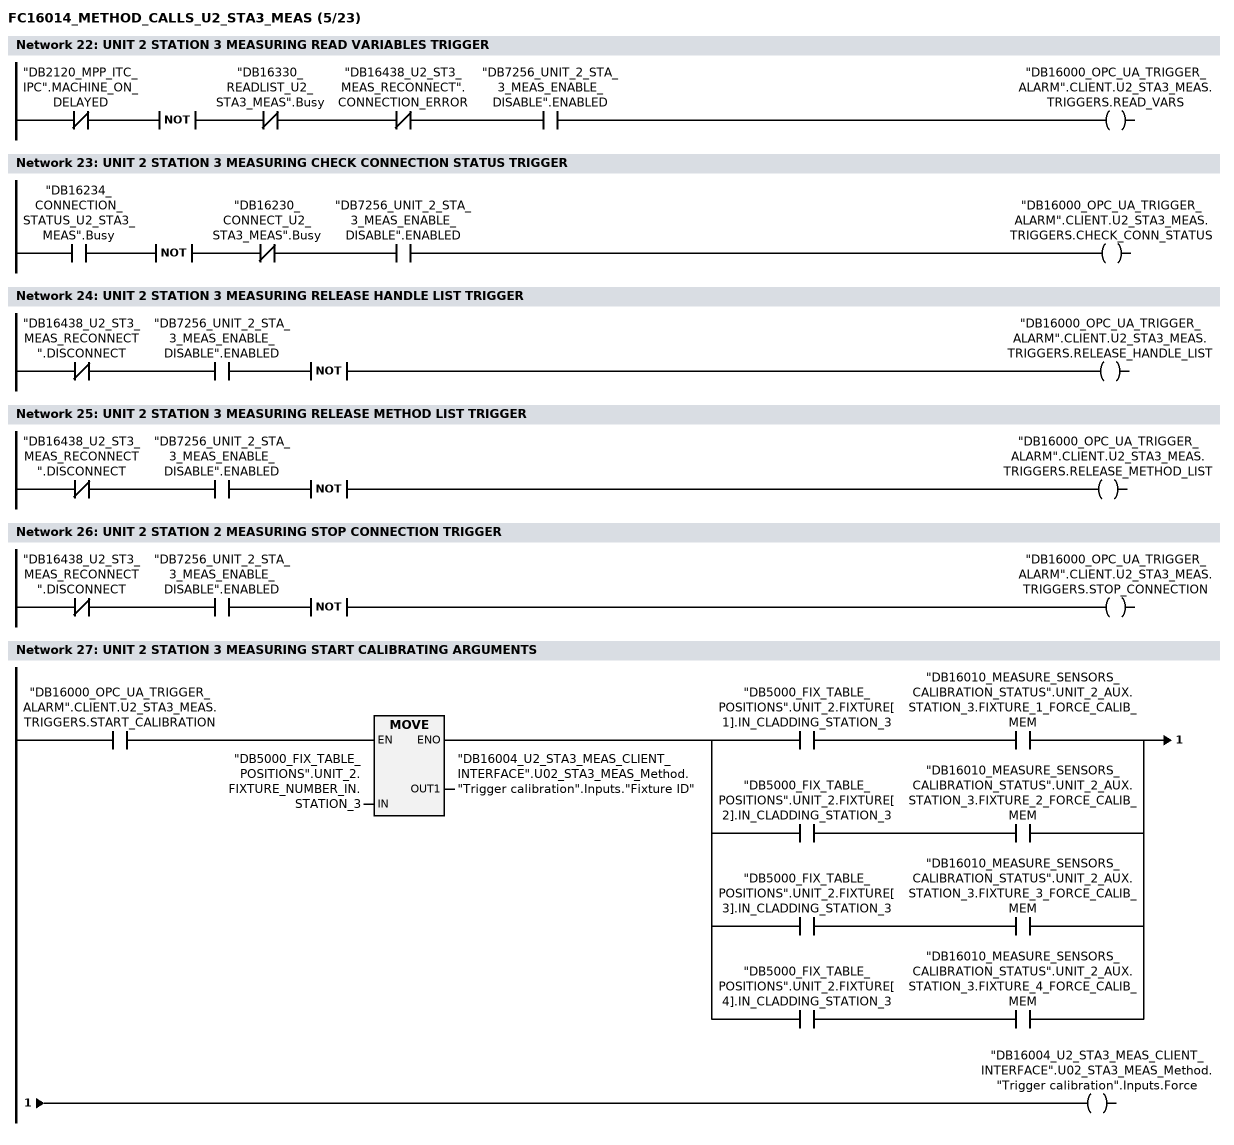
   RUNG wire#powerrail
      I_Contact( "DB2120_MPP_ITC_IPC".MACHINE_ON_DELAYED )
      Not()
      I_Contact( "DB16330_READLIST_U2_STA3_MEAS".Busy )
      I_Contact( "DB16438_U2_ST3_MEAS_RECONNECT".CONNECTION_ERROR )
      Contact( "DB7256_UNIT_2_STA_3_MEAS_ENABLE_DISABLE".ENABLED )
      Coil( "DB16000_OPC_UA_TRIGGER_ALARM".CLIENT.U2_STA3_MEAS.TRIGGERS.READ_VARS )
   END_RUNG
   // the same network as SCL:
   "DB16000_OPC_UA_TRIGGER_ALARM".CLIENT.U2_STA3_MEAS.TRIGGERS.READ_VARS := NOT (NOT "DB2120_MPP_ITC_IPC".MACHINE_ON_DELAYED) AND NOT "DB16330_READLIST_U2_STA3_MEAS".Busy AND NOT "DB16438_U2_ST3_MEAS_RECONNECT".CONNECTION_ERROR AND "DB7256_UNIT_2_STA_3_MEAS_ENABLE_DISABLE".ENABLED;
END_REGION

REGION Network 23: UNIT 2 STATION 3 MEASURING CHECK CONNECTION STATUS TRIGGER
   RUNG wire#powerrail
      Contact( "DB16234_CONNECTION_STATUS_U2_STA3_MEAS".Busy )
      Not()
      I_Contact( "DB16230_CONNECT_U2_STA3_MEAS".Busy )
      Contact( "DB7256_UNIT_2_STA_3_MEAS_ENABLE_DISABLE".ENABLED )
      Coil( "DB16000_OPC_UA_TRIGGER_ALARM".CLIENT.U2_STA3_MEAS.TRIGGERS.CHECK_CONN_STATUS )
   END_RUNG
   // the same network as SCL:
   "DB16000_OPC_UA_TRIGGER_ALARM".CLIENT.U2_STA3_MEAS.TRIGGERS.CHECK_CONN_STATUS := NOT "DB16234_CONNECTION_STATUS_U2_STA3_MEAS".Busy AND NOT "DB16230_CONNECT_U2_STA3_MEAS".Busy AND "DB7256_UNIT_2_STA_3_MEAS_ENABLE_DISABLE".ENABLED;
END_REGION

REGION Network 24: UNIT 2 STATION 3 MEASURING RELEASE HANDLE LIST TRIGGER
   RUNG wire#powerrail
      I_Contact( "DB16438_U2_ST3_MEAS_RECONNECT".DISCONNECT )
      Contact( "DB7256_UNIT_2_STA_3_MEAS_ENABLE_DISABLE".ENABLED )
      Not()
      Coil( "DB16000_OPC_UA_TRIGGER_ALARM".CLIENT.U2_STA3_MEAS.TRIGGERS.RELEASE_HANDLE_LIST )
   END_RUNG
   // the same network as SCL:
   "DB16000_OPC_UA_TRIGGER_ALARM".CLIENT.U2_STA3_MEAS.TRIGGERS.RELEASE_HANDLE_LIST := NOT (NOT "DB16438_U2_ST3_MEAS_RECONNECT".DISCONNECT AND "DB7256_UNIT_2_STA_3_MEAS_ENABLE_DISABLE".ENABLED);
END_REGION

REGION Network 25: UNIT 2 STATION 3 MEASURING RELEASE METHOD LIST TRIGGER
   RUNG wire#powerrail
      I_Contact( "DB16438_U2_ST3_MEAS_RECONNECT".DISCONNECT )
      Contact( "DB7256_UNIT_2_STA_3_MEAS_ENABLE_DISABLE".ENABLED )
      Not()
      Coil( "DB16000_OPC_UA_TRIGGER_ALARM".CLIENT.U2_STA3_MEAS.TRIGGERS.RELEASE_METHOD_LIST )
   END_RUNG
   // the same network as SCL:
   "DB16000_OPC_UA_TRIGGER_ALARM".CLIENT.U2_STA3_MEAS.TRIGGERS.RELEASE_METHOD_LIST := NOT (NOT "DB16438_U2_ST3_MEAS_RECONNECT".DISCONNECT AND "DB7256_UNIT_2_STA_3_MEAS_ENABLE_DISABLE".ENABLED);
END_REGION

REGION Network 26: UNIT 2 STATION 2 MEASURING STOP CONNECTION TRIGGER
   RUNG wire#powerrail
      I_Contact( "DB16438_U2_ST3_MEAS_RECONNECT".DISCONNECT )
      Contact( "DB7256_UNIT_2_STA_3_MEAS_ENABLE_DISABLE".ENABLED )
      Not()
      Coil( "DB16000_OPC_UA_TRIGGER_ALARM".CLIENT.U2_STA3_MEAS.TRIGGERS.STOP_CONNECTION )
   END_RUNG
   // the same network as SCL:
   "DB16000_OPC_UA_TRIGGER_ALARM".CLIENT.U2_STA3_MEAS.TRIGGERS.STOP_CONNECTION := NOT (NOT "DB16438_U2_ST3_MEAS_RECONNECT".DISCONNECT AND "DB7256_UNIT_2_STA_3_MEAS_ENABLE_DISABLE".ENABLED);
END_REGION

REGION Network 27: UNIT 2 STATION 3 MEASURING START CALIBRATING ARGUMENTS
   RUNG wire#powerrail
      Contact( "DB16000_OPC_UA_TRIGGER_ALARM".CLIENT.U2_STA3_MEAS.TRIGGERS.START_CALIBRATION )
      Move(in := "DB5000_FIX_TABLE_POSITIONS".UNIT_2.FIXTURE_NUMBER_IN.STATION_3, out1 => "DB16004_U2_STA3_MEAS_CLIENT_INTERFACE".U02_STA3_MEAS_Method."Trigger calibration".Inputs."Fixture ID")
      wire#w1
      Contact( "DB5000_FIX_TABLE_POSITIONS".UNIT_2.FIXTURE[1].IN_CLADDING_STATION_3 )
      Contact( "DB16010_MEASURE_SENSORS_CALIBRATION_STATUS".UNIT_2_AUX.STATION_3.FIXTURE_1_FORCE_CALIB_MEM )
      wire#w2
      Coil( "DB16004_U2_STA3_MEAS_CLIENT_INTERFACE".U02_STA3_MEAS_Method."Trigger calibration".Inputs.Force )
   END_RUNG
   RUNG wire#w1
      Contact( "DB5000_FIX_TABLE_POSITIONS".UNIT_2.FIXTURE[2].IN_CLADDING_STATION_3 )
      Contact( "DB16010_MEASURE_SENSORS_CALIBRATION_STATUS".UNIT_2_AUX.STATION_3.FIXTURE_2_FORCE_CALIB_MEM )
   END_RUNG wire#w2
   RUNG wire#w1
      Contact( "DB5000_FIX_TABLE_POSITIONS".UNIT_2.FIXTURE[3].IN_CLADDING_STATION_3 )
      Contact( "DB16010_MEASURE_SENSORS_CALIBRATION_STATUS".UNIT_2_AUX.STATION_3.FIXTURE_3_FORCE_CALIB_MEM )
   END_RUNG wire#w2
   RUNG wire#w1
      Contact( "DB5000_FIX_TABLE_POSITIONS".UNIT_2.FIXTURE[4].IN_CLADDING_STATION_3 )
      Contact( "DB16010_MEASURE_SENSORS_CALIBRATION_STATUS".UNIT_2_AUX.STATION_3.FIXTURE_4_FORCE_CALIB_MEM )
   END_RUNG wire#w2
   // the same network as SCL:
   IF "DB16000_OPC_UA_TRIGGER_ALARM".CLIENT.U2_STA3_MEAS.TRIGGERS.START_CALIBRATION THEN
       "DB16004_U2_STA3_MEAS_CLIENT_INTERFACE".U02_STA3_MEAS_Method."Trigger calibration".Inputs."Fixture ID" := "DB5000_FIX_TABLE_POSITIONS".UNIT_2.FIXTURE_NUMBER_IN.STATION_3;
   END_IF;
   "DB16004_U2_STA3_MEAS_CLIENT_INTERFACE".U02_STA3_MEAS_Method."Trigger calibration".Inputs.Force := "DB16000_OPC_UA_TRIGGER_ALARM".CLIENT.U2_STA3_MEAS.TRIGGERS.START_CALIBRATION AND (("DB5000_FIX_TABLE_POSITIONS".UNIT_2.FIXTURE[1].IN_CLADDING_STATION_3 AND "DB16010_MEASURE_SENSORS_CALIBRATION_STATUS".UNIT_2_AUX.STATION_3.FIXTURE_1_FORCE_CALIB_MEM) OR ("DB5000_FIX_TABLE_POSITIONS".UNIT_2.FIXTURE[2].IN_CLADDING_STATION_3 AND "DB16010_MEASURE_SENSORS_CALIBRATION_STATUS".UNIT_2_AUX.STATION_3.FIXTURE_2_FORCE_CALIB_MEM) OR ("DB5000_FIX_TABLE_POSITIONS".UNIT_2.FIXTURE[3].IN_CLADDING_STATION_3 AND "DB16010_MEASURE_SENSORS_CALIBRATION_STATUS".UNIT_2_AUX.STATION_3.FIXTURE_3_FORCE_CALIB_MEM) OR ("DB5000_FIX_TABLE_POSITIONS".UNIT_2.FIXTURE[4].IN_CLADDING_STATION_3 AND "DB16010_MEASURE_SENSORS_CALIBRATION_STATUS".UNIT_2_AUX.STATION_3.FIXTURE_4_FORCE_CALIB_MEM));
END_REGION

REGION Network 28: UNIT 2 STATION 3 CONNECTION CALL
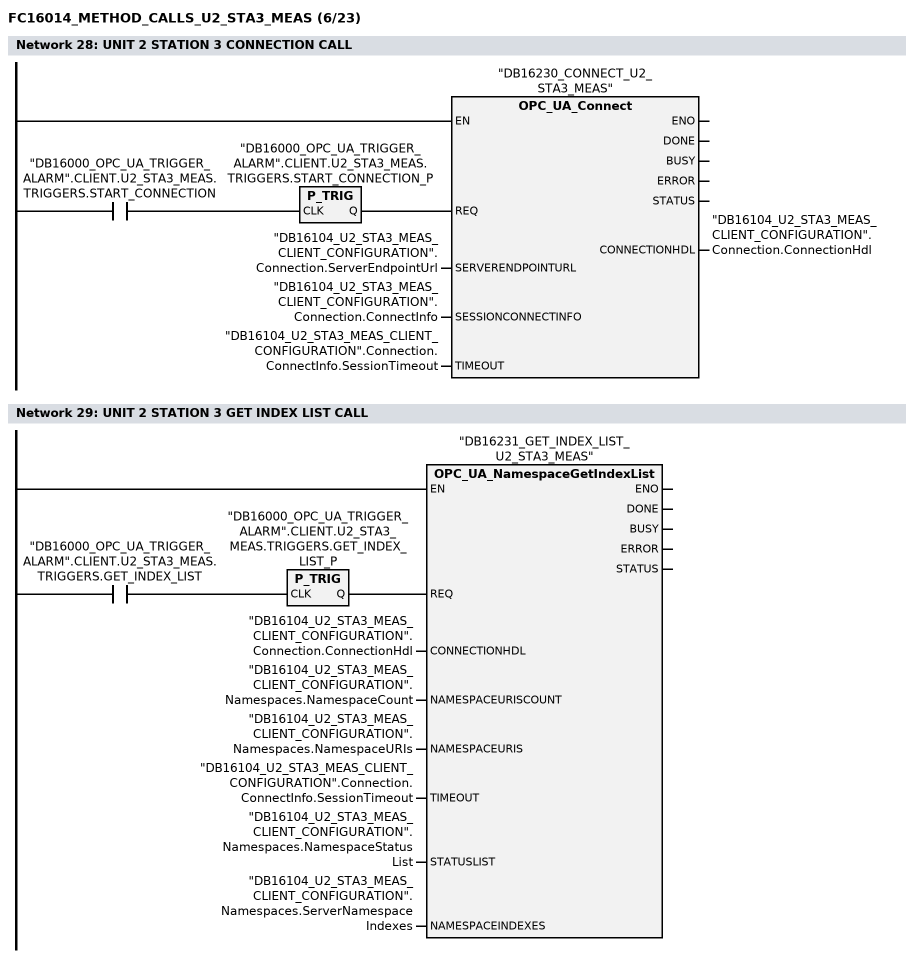
   RUNG wire#powerrail
      "DB16230_CONNECT_U2_STA3_MEAS".OPC_UA_Connect(REQ := wire#w1, ServerEndpointUrl := "DB16104_U2_STA3_MEAS_CLIENT_CONFIGURATION".Connection.ServerEndpointUrl, SessionConnectInfo := "DB16104_U2_STA3_MEAS_CLIENT_CONFIGURATION".Connection.ConnectInfo, Timeout := "DB16104_U2_STA3_MEAS_CLIENT_CONFIGURATION".Connection.ConnectInfo.SessionTimeout, Done =>, Busy =>, Error =>, Status =>, ConnectionHdl => "DB16104_U2_STA3_MEAS_CLIENT_CONFIGURATION".Connection.ConnectionHdl)
   END_RUNG
   RUNG wire#powerrail
      Contact( "DB16000_OPC_UA_TRIGGER_ALARM".CLIENT.U2_STA3_MEAS.TRIGGERS.START_CONNECTION )
      P_Trig( "DB16000_OPC_UA_TRIGGER_ALARM".CLIENT.U2_STA3_MEAS.TRIGGERS.START_CONNECTION_P )
   END_RUNG wire#w1
   // the same network as SCL:
   #_w1 := "DB16000_OPC_UA_TRIGGER_ALARM".CLIENT.U2_STA3_MEAS.TRIGGERS.START_CONNECTION AND NOT "DB16000_OPC_UA_TRIGGER_ALARM".CLIENT.U2_STA3_MEAS.TRIGGERS.START_CONNECTION_P;   // rising edge
   "DB16000_OPC_UA_TRIGGER_ALARM".CLIENT.U2_STA3_MEAS.TRIGGERS.START_CONNECTION_P := "DB16000_OPC_UA_TRIGGER_ALARM".CLIENT.U2_STA3_MEAS.TRIGGERS.START_CONNECTION;
   "DB16230_CONNECT_U2_STA3_MEAS"(REQ := #_w1,   // OPC_UA_Connect
                           ServerEndpointUrl := "DB16104_U2_STA3_MEAS_CLIENT_CONFIGURATION".Connection.ServerEndpointUrl,
                           SessionConnectInfo := "DB16104_U2_STA3_MEAS_CLIENT_CONFIGURATION".Connection.ConnectInfo,
                           Timeout := "DB16104_U2_STA3_MEAS_CLIENT_CONFIGURATION".Connection.ConnectInfo.SessionTimeout,
                           ConnectionHdl => "DB16104_U2_STA3_MEAS_CLIENT_CONFIGURATION".Connection.ConnectionHdl);
END_REGION

REGION Network 29: UNIT 2 STATION 3 GET INDEX LIST CALL
   RUNG wire#powerrail
      "DB16231_GET_INDEX_LIST_U2_STA3_MEAS".OPC_UA_NamespaceGetIndexList(REQ := wire#w1, ConnectionHdl := "DB16104_U2_STA3_MEAS_CLIENT_CONFIGURATION".Connection.ConnectionHdl, NamespaceUrisCount := "DB16104_U2_STA3_MEAS_CLIENT_CONFIGURATION".Namespaces.NamespaceCount, NamespaceUris := "DB16104_U2_STA3_MEAS_CLIENT_CONFIGURATION".Namespaces.NamespaceURIs, Timeout := "DB16104_U2_STA3_MEAS_CLIENT_CONFIGURATION".Connection.ConnectInfo.SessionTimeout, StatusList := "DB16104_U2_STA3_MEAS_CLIENT_CONFIGURATION".Namespaces.NamespaceStatusList, NamespaceIndexes := "DB16104_U2_STA3_MEAS_CLIENT_CONFIGURATION".Namespaces.ServerNamespaceIndexes, Done =>, Busy =>, Error =>, Status =>)
   END_RUNG
   RUNG wire#powerrail
      Contact( "DB16000_OPC_UA_TRIGGER_ALARM".CLIENT.U2_STA3_MEAS.TRIGGERS.GET_INDEX_LIST )
      P_Trig( "DB16000_OPC_UA_TRIGGER_ALARM".CLIENT.U2_STA3_MEAS.TRIGGERS.GET_INDEX_LIST_P )
   END_RUNG wire#w1
   // the same network as SCL:
   #_w1 := "DB16000_OPC_UA_TRIGGER_ALARM".CLIENT.U2_STA3_MEAS.TRIGGERS.GET_INDEX_LIST AND NOT "DB16000_OPC_UA_TRIGGER_ALARM".CLIENT.U2_STA3_MEAS.TRIGGERS.GET_INDEX_LIST_P;   // rising edge
   "DB16000_OPC_UA_TRIGGER_ALARM".CLIENT.U2_STA3_MEAS.TRIGGERS.GET_INDEX_LIST_P := "DB16000_OPC_UA_TRIGGER_ALARM".CLIENT.U2_STA3_MEAS.TRIGGERS.GET_INDEX_LIST;
   "DB16231_GET_INDEX_LIST_U2_STA3_MEAS"(REQ := #_w1,   // OPC_UA_NamespaceGetIndexList
                           ConnectionHdl := "DB16104_U2_STA3_MEAS_CLIENT_CONFIGURATION".Connection.ConnectionHdl,
                           NamespaceUrisCount := "DB16104_U2_STA3_MEAS_CLIENT_CONFIGURATION".Namespaces.NamespaceCount,
                           NamespaceUris := "DB16104_U2_STA3_MEAS_CLIENT_CONFIGURATION".Namespaces.NamespaceURIs,
                           Timeout := "DB16104_U2_STA3_MEAS_CLIENT_CONFIGURATION".Connection.ConnectInfo.SessionTimeout,
                           StatusList := "DB16104_U2_STA3_MEAS_CLIENT_CONFIGURATION".Namespaces.NamespaceStatusList,
                           NamespaceIndexes := "DB16104_U2_STA3_MEAS_CLIENT_CONFIGURATION".Namespaces.ServerNamespaceIndexes);
END_REGION

REGION Network 30: UNIT 2 STATION 3 GET HANDLE LIST CALL
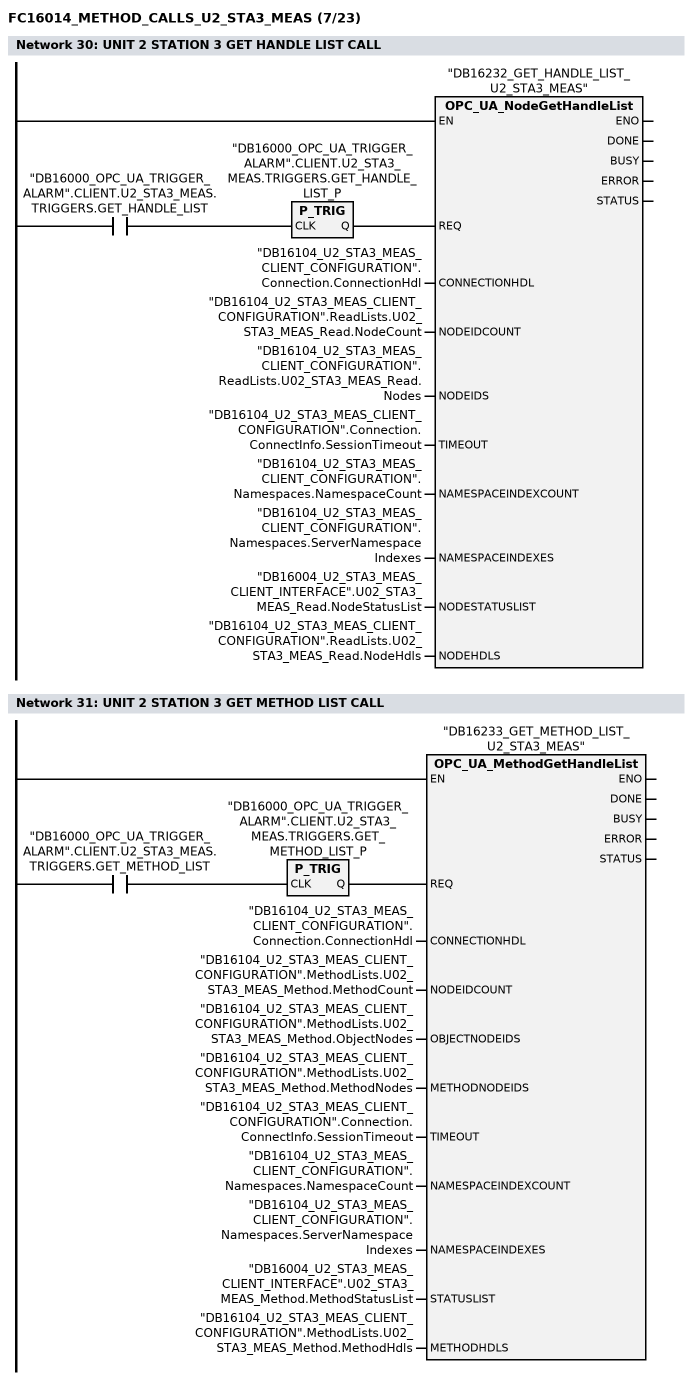
   RUNG wire#powerrail
      "DB16232_GET_HANDLE_LIST_U2_STA3_MEAS".OPC_UA_NodeGetHandleList(REQ := wire#w1, ConnectionHdl := "DB16104_U2_STA3_MEAS_CLIENT_CONFIGURATION".Connection.ConnectionHdl, NodeIDCount := "DB16104_U2_STA3_MEAS_CLIENT_CONFIGURATION".ReadLists.U02_STA3_MEAS_Read.NodeCount, NodeIDs := "DB16104_U2_STA3_MEAS_CLIENT_CONFIGURATION".ReadLists.U02_STA3_MEAS_Read.Nodes, Timeout := "DB16104_U2_STA3_MEAS_CLIENT_CONFIGURATION".Connection.ConnectInfo.SessionTimeout, NamespaceIndexCount := "DB16104_U2_STA3_MEAS_CLIENT_CONFIGURATION".Namespaces.NamespaceCount, NamespaceIndexes := "DB16104_U2_STA3_MEAS_CLIENT_CONFIGURATION".Namespaces.ServerNamespaceIndexes, NodeStatusList := "DB16004_U2_STA3_MEAS_CLIENT_INTERFACE".U02_STA3_MEAS_Read.NodeStatusList, NodeHdls := "DB16104_U2_STA3_MEAS_CLIENT_CONFIGURATION".ReadLists.U02_STA3_MEAS_Read.NodeHdls, Done =>, Busy =>, Error =>, Status =>)
   END_RUNG
   RUNG wire#powerrail
      Contact( "DB16000_OPC_UA_TRIGGER_ALARM".CLIENT.U2_STA3_MEAS.TRIGGERS.GET_HANDLE_LIST )
      P_Trig( "DB16000_OPC_UA_TRIGGER_ALARM".CLIENT.U2_STA3_MEAS.TRIGGERS.GET_HANDLE_LIST_P )
   END_RUNG wire#w1
   // the same network as SCL:
   #_w1 := "DB16000_OPC_UA_TRIGGER_ALARM".CLIENT.U2_STA3_MEAS.TRIGGERS.GET_HANDLE_LIST AND NOT "DB16000_OPC_UA_TRIGGER_ALARM".CLIENT.U2_STA3_MEAS.TRIGGERS.GET_HANDLE_LIST_P;   // rising edge
   "DB16000_OPC_UA_TRIGGER_ALARM".CLIENT.U2_STA3_MEAS.TRIGGERS.GET_HANDLE_LIST_P := "DB16000_OPC_UA_TRIGGER_ALARM".CLIENT.U2_STA3_MEAS.TRIGGERS.GET_HANDLE_LIST;
   "DB16232_GET_HANDLE_LIST_U2_STA3_MEAS"(REQ := #_w1,   // OPC_UA_NodeGetHandleList
                           ConnectionHdl := "DB16104_U2_STA3_MEAS_CLIENT_CONFIGURATION".Connection.ConnectionHdl,
                           NodeIDCount := "DB16104_U2_STA3_MEAS_CLIENT_CONFIGURATION".ReadLists.U02_STA3_MEAS_Read.NodeCount,
                           NodeIDs := "DB16104_U2_STA3_MEAS_CLIENT_CONFIGURATION".ReadLists.U02_STA3_MEAS_Read.Nodes,
                           Timeout := "DB16104_U2_STA3_MEAS_CLIENT_CONFIGURATION".Connection.ConnectInfo.SessionTimeout,
                           NamespaceIndexCount := "DB16104_U2_STA3_MEAS_CLIENT_CONFIGURATION".Namespaces.NamespaceCount,
                           NamespaceIndexes := "DB16104_U2_STA3_MEAS_CLIENT_CONFIGURATION".Namespaces.ServerNamespaceIndexes,
                           NodeStatusList := "DB16004_U2_STA3_MEAS_CLIENT_INTERFACE".U02_STA3_MEAS_Read.NodeStatusList,
                           NodeHdls := "DB16104_U2_STA3_MEAS_CLIENT_CONFIGURATION".ReadLists.U02_STA3_MEAS_Read.NodeHdls);
END_REGION

REGION Network 31: UNIT 2 STATION 3 GET METHOD LIST CALL
   RUNG wire#powerrail
      "DB16233_GET_METHOD_LIST_U2_STA3_MEAS".OPC_UA_MethodGetHandleList(REQ := wire#w1, ConnectionHdl := "DB16104_U2_STA3_MEAS_CLIENT_CONFIGURATION".Connection.ConnectionHdl, NodeIDCount := "DB16104_U2_STA3_MEAS_CLIENT_CONFIGURATION".MethodLists.U02_STA3_MEAS_Method.MethodCount, ObjectNodeIDs := "DB16104_U2_STA3_MEAS_CLIENT_CONFIGURATION".MethodLists.U02_STA3_MEAS_Method.ObjectNodes, MethodNodeIDs := "DB16104_U2_STA3_MEAS_CLIENT_CONFIGURATION".MethodLists.U02_STA3_MEAS_Method.MethodNodes, Timeout := "DB16104_U2_STA3_MEAS_CLIENT_CONFIGURATION".Connection.ConnectInfo.SessionTimeout, NamespaceIndexCount := "DB16104_U2_STA3_MEAS_CLIENT_CONFIGURATION".Namespaces.NamespaceCount, NamespaceIndexes := "DB16104_U2_STA3_MEAS_CLIENT_CONFIGURATION".Namespaces.ServerNamespaceIndexes, StatusList := "DB16004_U2_STA3_MEAS_CLIENT_INTERFACE".U02_STA3_MEAS_Method.MethodStatusList, MethodHdls := "DB16104_U2_STA3_MEAS_CLIENT_CONFIGURATION".MethodLists.U02_STA3_MEAS_Method.MethodHdls, Done =>, Busy =>, Error =>, Status =>)
   END_RUNG
   RUNG wire#powerrail
      Contact( "DB16000_OPC_UA_TRIGGER_ALARM".CLIENT.U2_STA3_MEAS.TRIGGERS.GET_METHOD_LIST )
      P_Trig( "DB16000_OPC_UA_TRIGGER_ALARM".CLIENT.U2_STA3_MEAS.TRIGGERS.GET_METHOD_LIST_P )
   END_RUNG wire#w1
   // the same network as SCL:
   #_w1 := "DB16000_OPC_UA_TRIGGER_ALARM".CLIENT.U2_STA3_MEAS.TRIGGERS.GET_METHOD_LIST AND NOT "DB16000_OPC_UA_TRIGGER_ALARM".CLIENT.U2_STA3_MEAS.TRIGGERS.GET_METHOD_LIST_P;   // rising edge
   "DB16000_OPC_UA_TRIGGER_ALARM".CLIENT.U2_STA3_MEAS.TRIGGERS.GET_METHOD_LIST_P := "DB16000_OPC_UA_TRIGGER_ALARM".CLIENT.U2_STA3_MEAS.TRIGGERS.GET_METHOD_LIST;
   "DB16233_GET_METHOD_LIST_U2_STA3_MEAS"(REQ := #_w1,   // OPC_UA_MethodGetHandleList
                           ConnectionHdl := "DB16104_U2_STA3_MEAS_CLIENT_CONFIGURATION".Connection.ConnectionHdl,
                           NodeIDCount := "DB16104_U2_STA3_MEAS_CLIENT_CONFIGURATION".MethodLists.U02_STA3_MEAS_Method.MethodCount,
                           ObjectNodeIDs := "DB16104_U2_STA3_MEAS_CLIENT_CONFIGURATION".MethodLists.U02_STA3_MEAS_Method.ObjectNodes,
                           MethodNodeIDs := "DB16104_U2_STA3_MEAS_CLIENT_CONFIGURATION".MethodLists.U02_STA3_MEAS_Method.MethodNodes,
                           Timeout := "DB16104_U2_STA3_MEAS_CLIENT_CONFIGURATION".Connection.ConnectInfo.SessionTimeout,
                           NamespaceIndexCount := "DB16104_U2_STA3_MEAS_CLIENT_CONFIGURATION".Namespaces.NamespaceCount,
                           NamespaceIndexes := "DB16104_U2_STA3_MEAS_CLIENT_CONFIGURATION".Namespaces.ServerNamespaceIndexes,
                           StatusList := "DB16004_U2_STA3_MEAS_CLIENT_INTERFACE".U02_STA3_MEAS_Method.MethodStatusList,
                           MethodHdls := "DB16104_U2_STA3_MEAS_CLIENT_CONFIGURATION".MethodLists.U02_STA3_MEAS_Method.MethodHdls);
END_REGION

REGION Network 32: UNIT 2 STATION 3 MEASURING START MEASURING NOOZLE SURFACE DISTANCE TRIGGER CALL
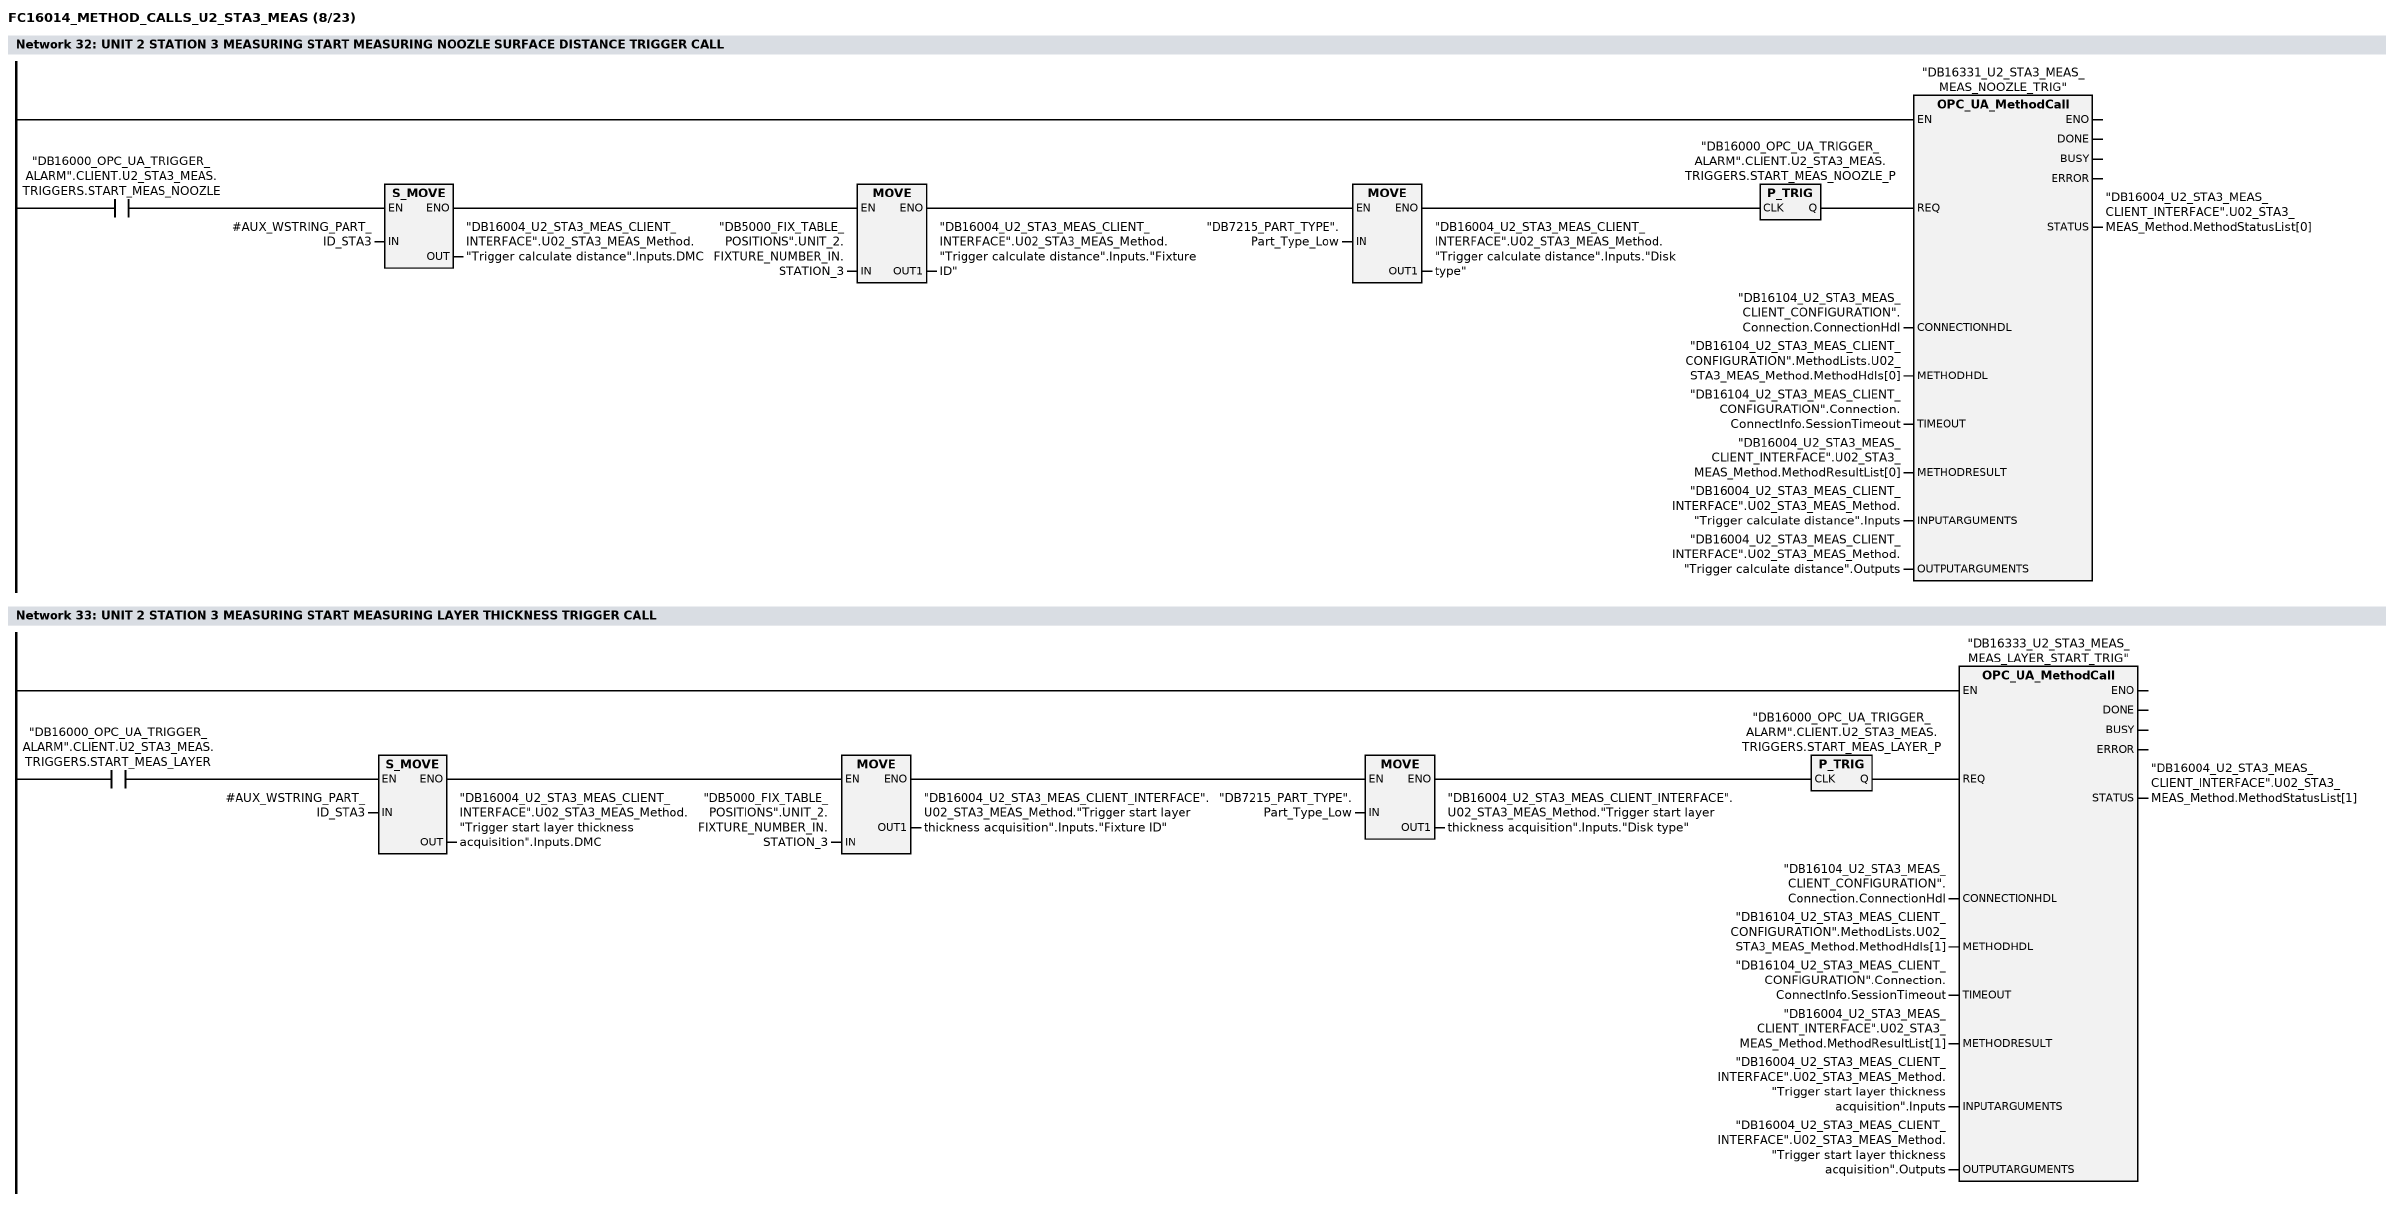
   RUNG wire#powerrail
      "DB16331_U2_STA3_MEAS_MEAS_NOOZLE_TRIG".OPC_UA_MethodCall(REQ := wire#w1, ConnectionHdl := "DB16104_U2_STA3_MEAS_CLIENT_CONFIGURATION".Connection.ConnectionHdl, MethodHdl := "DB16104_U2_STA3_MEAS_CLIENT_CONFIGURATION".MethodLists.U02_STA3_MEAS_Method.MethodHdls[0], Timeout := "DB16104_U2_STA3_MEAS_CLIENT_CONFIGURATION".Connection.ConnectInfo.SessionTimeout, MethodResult := "DB16004_U2_STA3_MEAS_CLIENT_INTERFACE".U02_STA3_MEAS_Method.MethodResultList[0], InputArguments := "DB16004_U2_STA3_MEAS_CLIENT_INTERFACE".U02_STA3_MEAS_Method."Trigger calculate distance".Inputs, OutputArguments := "DB16004_U2_STA3_MEAS_CLIENT_INTERFACE".U02_STA3_MEAS_Method."Trigger calculate distance".Outputs, Done =>, Busy =>, Error =>, Status => "DB16004_U2_STA3_MEAS_CLIENT_INTERFACE".U02_STA3_MEAS_Method.MethodStatusList[0])
   END_RUNG
   RUNG wire#powerrail
      Contact( "DB16000_OPC_UA_TRIGGER_ALARM".CLIENT.U2_STA3_MEAS.TRIGGERS.START_MEAS_NOOZLE )
      S_Move(in := #AUX_WSTRING_PART_ID_STA3, out => "DB16004_U2_STA3_MEAS_CLIENT_INTERFACE".U02_STA3_MEAS_Method."Trigger calculate distance".Inputs.DMC)
      Move(in := "DB5000_FIX_TABLE_POSITIONS".UNIT_2.FIXTURE_NUMBER_IN.STATION_3, out1 => "DB16004_U2_STA3_MEAS_CLIENT_INTERFACE".U02_STA3_MEAS_Method."Trigger calculate distance".Inputs."Fixture ID")
      Move(in := "DB7215_PART_TYPE".Part_Type_Low, out1 => "DB16004_U2_STA3_MEAS_CLIENT_INTERFACE".U02_STA3_MEAS_Method."Trigger calculate distance".Inputs."Disk type")
      P_Trig( "DB16000_OPC_UA_TRIGGER_ALARM".CLIENT.U2_STA3_MEAS.TRIGGERS.START_MEAS_NOOZLE_P )
   END_RUNG wire#w1
   // the same network as SCL:
   IF "DB16000_OPC_UA_TRIGGER_ALARM".CLIENT.U2_STA3_MEAS.TRIGGERS.START_MEAS_NOOZLE THEN
       "DB16004_U2_STA3_MEAS_CLIENT_INTERFACE".U02_STA3_MEAS_Method."Trigger calculate distance".Inputs.DMC := #AUX_WSTRING_PART_ID_STA3;
       "DB16004_U2_STA3_MEAS_CLIENT_INTERFACE".U02_STA3_MEAS_Method."Trigger calculate distance".Inputs."Fixture ID" := "DB5000_FIX_TABLE_POSITIONS".UNIT_2.FIXTURE_NUMBER_IN.STATION_3;
       "DB16004_U2_STA3_MEAS_CLIENT_INTERFACE".U02_STA3_MEAS_Method."Trigger calculate distance".Inputs."Disk type" := "DB7215_PART_TYPE".Part_Type_Low;
   END_IF;
   #_w1 := "DB16000_OPC_UA_TRIGGER_ALARM".CLIENT.U2_STA3_MEAS.TRIGGERS.START_MEAS_NOOZLE AND NOT "DB16000_OPC_UA_TRIGGER_ALARM".CLIENT.U2_STA3_MEAS.TRIGGERS.START_MEAS_NOOZLE_P;   // rising edge
   "DB16000_OPC_UA_TRIGGER_ALARM".CLIENT.U2_STA3_MEAS.TRIGGERS.START_MEAS_NOOZLE_P := "DB16000_OPC_UA_TRIGGER_ALARM".CLIENT.U2_STA3_MEAS.TRIGGERS.START_MEAS_NOOZLE;
   "DB16331_U2_STA3_MEAS_MEAS_NOOZLE_TRIG"(REQ := #_w1,   // OPC_UA_MethodCall
                           ConnectionHdl := "DB16104_U2_STA3_MEAS_CLIENT_CONFIGURATION".Connection.ConnectionHdl,
                           MethodHdl := "DB16104_U2_STA3_MEAS_CLIENT_CONFIGURATION".MethodLists.U02_STA3_MEAS_Method.MethodHdls[0],
                           Timeout := "DB16104_U2_STA3_MEAS_CLIENT_CONFIGURATION".Connection.ConnectInfo.SessionTimeout,
                           MethodResult := "DB16004_U2_STA3_MEAS_CLIENT_INTERFACE".U02_STA3_MEAS_Method.MethodResultList[0],
                           InputArguments := "DB16004_U2_STA3_MEAS_CLIENT_INTERFACE".U02_STA3_MEAS_Method."Trigger calculate distance".Inputs,
                           OutputArguments := "DB16004_U2_STA3_MEAS_CLIENT_INTERFACE".U02_STA3_MEAS_Method."Trigger calculate distance".Outputs,
                           Status => "DB16004_U2_STA3_MEAS_CLIENT_INTERFACE".U02_STA3_MEAS_Method.MethodStatusList[0]);
END_REGION

REGION Network 33: UNIT 2 STATION 3 MEASURING START MEASURING LAYER THICKNESS TRIGGER CALL
   RUNG wire#powerrail
      "DB16333_U2_STA3_MEAS_MEAS_LAYER_START_TRIG".OPC_UA_MethodCall(REQ := wire#w1, ConnectionHdl := "DB16104_U2_STA3_MEAS_CLIENT_CONFIGURATION".Connection.ConnectionHdl, MethodHdl := "DB16104_U2_STA3_MEAS_CLIENT_CONFIGURATION".MethodLists.U02_STA3_MEAS_Method.MethodHdls[1], Timeout := "DB16104_U2_STA3_MEAS_CLIENT_CONFIGURATION".Connection.ConnectInfo.SessionTimeout, MethodResult := "DB16004_U2_STA3_MEAS_CLIENT_INTERFACE".U02_STA3_MEAS_Method.MethodResultList[1], InputArguments := "DB16004_U2_STA3_MEAS_CLIENT_INTERFACE".U02_STA3_MEAS_Method."Trigger start layer thickness acquisition".Inputs, OutputArguments := "DB16004_U2_STA3_MEAS_CLIENT_INTERFACE".U02_STA3_MEAS_Method."Trigger start layer thickness acquisition".Outputs, Done =>, Busy =>, Error =>, Status => "DB16004_U2_STA3_MEAS_CLIENT_INTERFACE".U02_STA3_MEAS_Method.MethodStatusList[1])
   END_RUNG
   RUNG wire#powerrail
      Contact( "DB16000_OPC_UA_TRIGGER_ALARM".CLIENT.U2_STA3_MEAS.TRIGGERS.START_MEAS_LAYER )
      S_Move(in := #AUX_WSTRING_PART_ID_STA3, out => "DB16004_U2_STA3_MEAS_CLIENT_INTERFACE".U02_STA3_MEAS_Method."Trigger start layer thickness acquisition".Inputs.DMC)
      Move(in := "DB5000_FIX_TABLE_POSITIONS".UNIT_2.FIXTURE_NUMBER_IN.STATION_3, out1 => "DB16004_U2_STA3_MEAS_CLIENT_INTERFACE".U02_STA3_MEAS_Method."Trigger start layer thickness acquisition".Inputs."Fixture ID")
      Move(in := "DB7215_PART_TYPE".Part_Type_Low, out1 => "DB16004_U2_STA3_MEAS_CLIENT_INTERFACE".U02_STA3_MEAS_Method."Trigger start layer thickness acquisition".Inputs."Disk type")
      P_Trig( "DB16000_OPC_UA_TRIGGER_ALARM".CLIENT.U2_STA3_MEAS.TRIGGERS.START_MEAS_LAYER_P )
   END_RUNG wire#w1
   // the same network as SCL:
   IF "DB16000_OPC_UA_TRIGGER_ALARM".CLIENT.U2_STA3_MEAS.TRIGGERS.START_MEAS_LAYER THEN
       "DB16004_U2_STA3_MEAS_CLIENT_INTERFACE".U02_STA3_MEAS_Method."Trigger start layer thickness acquisition".Inputs.DMC := #AUX_WSTRING_PART_ID_STA3;
       "DB16004_U2_STA3_MEAS_CLIENT_INTERFACE".U02_STA3_MEAS_Method."Trigger start layer thickness acquisition".Inputs."Fixture ID" := "DB5000_FIX_TABLE_POSITIONS".UNIT_2.FIXTURE_NUMBER_IN.STATION_3;
       "DB16004_U2_STA3_MEAS_CLIENT_INTERFACE".U02_STA3_MEAS_Method."Trigger start layer thickness acquisition".Inputs."Disk type" := "DB7215_PART_TYPE".Part_Type_Low;
   END_IF;
   #_w1 := "DB16000_OPC_UA_TRIGGER_ALARM".CLIENT.U2_STA3_MEAS.TRIGGERS.START_MEAS_LAYER AND NOT "DB16000_OPC_UA_TRIGGER_ALARM".CLIENT.U2_STA3_MEAS.TRIGGERS.START_MEAS_LAYER_P;   // rising edge
   "DB16000_OPC_UA_TRIGGER_ALARM".CLIENT.U2_STA3_MEAS.TRIGGERS.START_MEAS_LAYER_P := "DB16000_OPC_UA_TRIGGER_ALARM".CLIENT.U2_STA3_MEAS.TRIGGERS.START_MEAS_LAYER;
   "DB16333_U2_STA3_MEAS_MEAS_LAYER_START_TRIG"(REQ := #_w1,   // OPC_UA_MethodCall
                           ConnectionHdl := "DB16104_U2_STA3_MEAS_CLIENT_CONFIGURATION".Connection.ConnectionHdl,
                           MethodHdl := "DB16104_U2_STA3_MEAS_CLIENT_CONFIGURATION".MethodLists.U02_STA3_MEAS_Method.MethodHdls[1],
                           Timeout := "DB16104_U2_STA3_MEAS_CLIENT_CONFIGURATION".Connection.ConnectInfo.SessionTimeout,
                           MethodResult := "DB16004_U2_STA3_MEAS_CLIENT_INTERFACE".U02_STA3_MEAS_Method.MethodResultList[1],
                           InputArguments := "DB16004_U2_STA3_MEAS_CLIENT_INTERFACE".U02_STA3_MEAS_Method."Trigger start layer thickness acquisition".Inputs,
                           OutputArguments := "DB16004_U2_STA3_MEAS_CLIENT_INTERFACE".U02_STA3_MEAS_Method."Trigger start layer thickness acquisition".Outputs,
                           Status => "DB16004_U2_STA3_MEAS_CLIENT_INTERFACE".U02_STA3_MEAS_Method.MethodStatusList[1]);
END_REGION

REGION Network 34: UNIT 2 STATION 3 MEASURING STOP MEASURING LAYER THICKNESS TRIGGER CALL
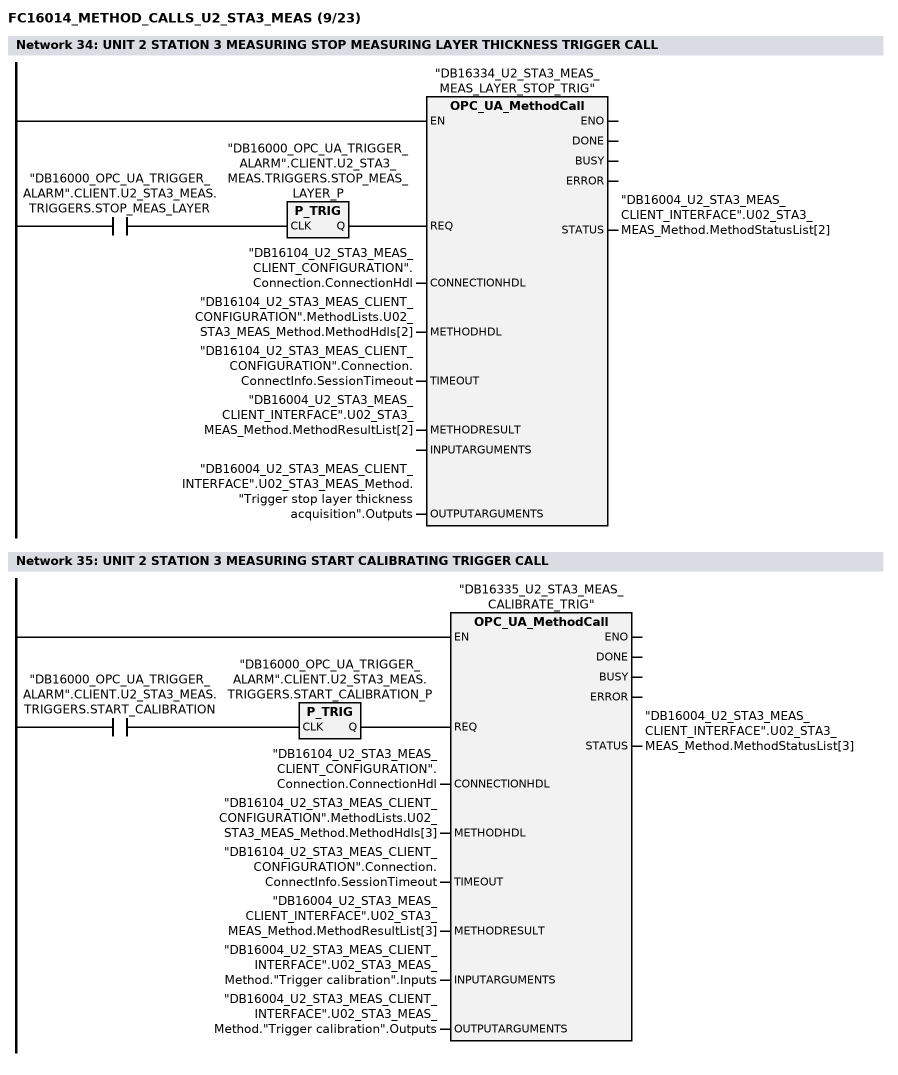
   RUNG wire#powerrail
      "DB16334_U2_STA3_MEAS_MEAS_LAYER_STOP_TRIG".OPC_UA_MethodCall(REQ := wire#w1, ConnectionHdl := "DB16104_U2_STA3_MEAS_CLIENT_CONFIGURATION".Connection.ConnectionHdl, MethodHdl := "DB16104_U2_STA3_MEAS_CLIENT_CONFIGURATION".MethodLists.U02_STA3_MEAS_Method.MethodHdls[2], Timeout := "DB16104_U2_STA3_MEAS_CLIENT_CONFIGURATION".Connection.ConnectInfo.SessionTimeout, MethodResult := "DB16004_U2_STA3_MEAS_CLIENT_INTERFACE".U02_STA3_MEAS_Method.MethodResultList[2], InputArguments :=, OutputArguments := "DB16004_U2_STA3_MEAS_CLIENT_INTERFACE".U02_STA3_MEAS_Method."Trigger stop layer thickness acquisition".Outputs, Done =>, Busy =>, Error =>, Status => "DB16004_U2_STA3_MEAS_CLIENT_INTERFACE".U02_STA3_MEAS_Method.MethodStatusList[2])
   END_RUNG
   RUNG wire#powerrail
      Contact( "DB16000_OPC_UA_TRIGGER_ALARM".CLIENT.U2_STA3_MEAS.TRIGGERS.STOP_MEAS_LAYER )
      P_Trig( "DB16000_OPC_UA_TRIGGER_ALARM".CLIENT.U2_STA3_MEAS.TRIGGERS.STOP_MEAS_LAYER_P )
   END_RUNG wire#w1
   // the same network as SCL:
   #_w1 := "DB16000_OPC_UA_TRIGGER_ALARM".CLIENT.U2_STA3_MEAS.TRIGGERS.STOP_MEAS_LAYER AND NOT "DB16000_OPC_UA_TRIGGER_ALARM".CLIENT.U2_STA3_MEAS.TRIGGERS.STOP_MEAS_LAYER_P;   // rising edge
   "DB16000_OPC_UA_TRIGGER_ALARM".CLIENT.U2_STA3_MEAS.TRIGGERS.STOP_MEAS_LAYER_P := "DB16000_OPC_UA_TRIGGER_ALARM".CLIENT.U2_STA3_MEAS.TRIGGERS.STOP_MEAS_LAYER;
   "DB16334_U2_STA3_MEAS_MEAS_LAYER_STOP_TRIG"(REQ := #_w1,   // OPC_UA_MethodCall
                           ConnectionHdl := "DB16104_U2_STA3_MEAS_CLIENT_CONFIGURATION".Connection.ConnectionHdl,
                           MethodHdl := "DB16104_U2_STA3_MEAS_CLIENT_CONFIGURATION".MethodLists.U02_STA3_MEAS_Method.MethodHdls[2],
                           Timeout := "DB16104_U2_STA3_MEAS_CLIENT_CONFIGURATION".Connection.ConnectInfo.SessionTimeout,
                           MethodResult := "DB16004_U2_STA3_MEAS_CLIENT_INTERFACE".U02_STA3_MEAS_Method.MethodResultList[2],
                           OutputArguments := "DB16004_U2_STA3_MEAS_CLIENT_INTERFACE".U02_STA3_MEAS_Method."Trigger stop layer thickness acquisition".Outputs,
                           Status => "DB16004_U2_STA3_MEAS_CLIENT_INTERFACE".U02_STA3_MEAS_Method.MethodStatusList[2]);
END_REGION

REGION Network 35: UNIT 2 STATION 3 MEASURING START CALIBRATING TRIGGER CALL
   RUNG wire#powerrail
      "DB16335_U2_STA3_MEAS_CALIBRATE_TRIG".OPC_UA_MethodCall(REQ := wire#w1, ConnectionHdl := "DB16104_U2_STA3_MEAS_CLIENT_CONFIGURATION".Connection.ConnectionHdl, MethodHdl := "DB16104_U2_STA3_MEAS_CLIENT_CONFIGURATION".MethodLists.U02_STA3_MEAS_Method.MethodHdls[3], Timeout := "DB16104_U2_STA3_MEAS_CLIENT_CONFIGURATION".Connection.ConnectInfo.SessionTimeout, MethodResult := "DB16004_U2_STA3_MEAS_CLIENT_INTERFACE".U02_STA3_MEAS_Method.MethodResultList[3], InputArguments := "DB16004_U2_STA3_MEAS_CLIENT_INTERFACE".U02_STA3_MEAS_Method."Trigger calibration".Inputs, OutputArguments := "DB16004_U2_STA3_MEAS_CLIENT_INTERFACE".U02_STA3_MEAS_Method."Trigger calibration".Outputs, Done =>, Busy =>, Error =>, Status => "DB16004_U2_STA3_MEAS_CLIENT_INTERFACE".U02_STA3_MEAS_Method.MethodStatusList[3])
   END_RUNG
   RUNG wire#powerrail
      Contact( "DB16000_OPC_UA_TRIGGER_ALARM".CLIENT.U2_STA3_MEAS.TRIGGERS.START_CALIBRATION )
      P_Trig( "DB16000_OPC_UA_TRIGGER_ALARM".CLIENT.U2_STA3_MEAS.TRIGGERS.START_CALIBRATION_P )
   END_RUNG wire#w1
   // the same network as SCL:
   #_w1 := "DB16000_OPC_UA_TRIGGER_ALARM".CLIENT.U2_STA3_MEAS.TRIGGERS.START_CALIBRATION AND NOT "DB16000_OPC_UA_TRIGGER_ALARM".CLIENT.U2_STA3_MEAS.TRIGGERS.START_CALIBRATION_P;   // rising edge
   "DB16000_OPC_UA_TRIGGER_ALARM".CLIENT.U2_STA3_MEAS.TRIGGERS.START_CALIBRATION_P := "DB16000_OPC_UA_TRIGGER_ALARM".CLIENT.U2_STA3_MEAS.TRIGGERS.START_CALIBRATION;
   "DB16335_U2_STA3_MEAS_CALIBRATE_TRIG"(REQ := #_w1,   // OPC_UA_MethodCall
                           ConnectionHdl := "DB16104_U2_STA3_MEAS_CLIENT_CONFIGURATION".Connection.ConnectionHdl,
                           MethodHdl := "DB16104_U2_STA3_MEAS_CLIENT_CONFIGURATION".MethodLists.U02_STA3_MEAS_Method.MethodHdls[3],
                           Timeout := "DB16104_U2_STA3_MEAS_CLIENT_CONFIGURATION".Connection.ConnectInfo.SessionTimeout,
                           MethodResult := "DB16004_U2_STA3_MEAS_CLIENT_INTERFACE".U02_STA3_MEAS_Method.MethodResultList[3],
                           InputArguments := "DB16004_U2_STA3_MEAS_CLIENT_INTERFACE".U02_STA3_MEAS_Method."Trigger calibration".Inputs,
                           OutputArguments := "DB16004_U2_STA3_MEAS_CLIENT_INTERFACE".U02_STA3_MEAS_Method."Trigger calibration".Outputs,
                           Status => "DB16004_U2_STA3_MEAS_CLIENT_INTERFACE".U02_STA3_MEAS_Method.MethodStatusList[3]);
END_REGION

REGION Network 36: UNIT 2 STATION 3 MEASURING RESET PC TRIGGER CALL
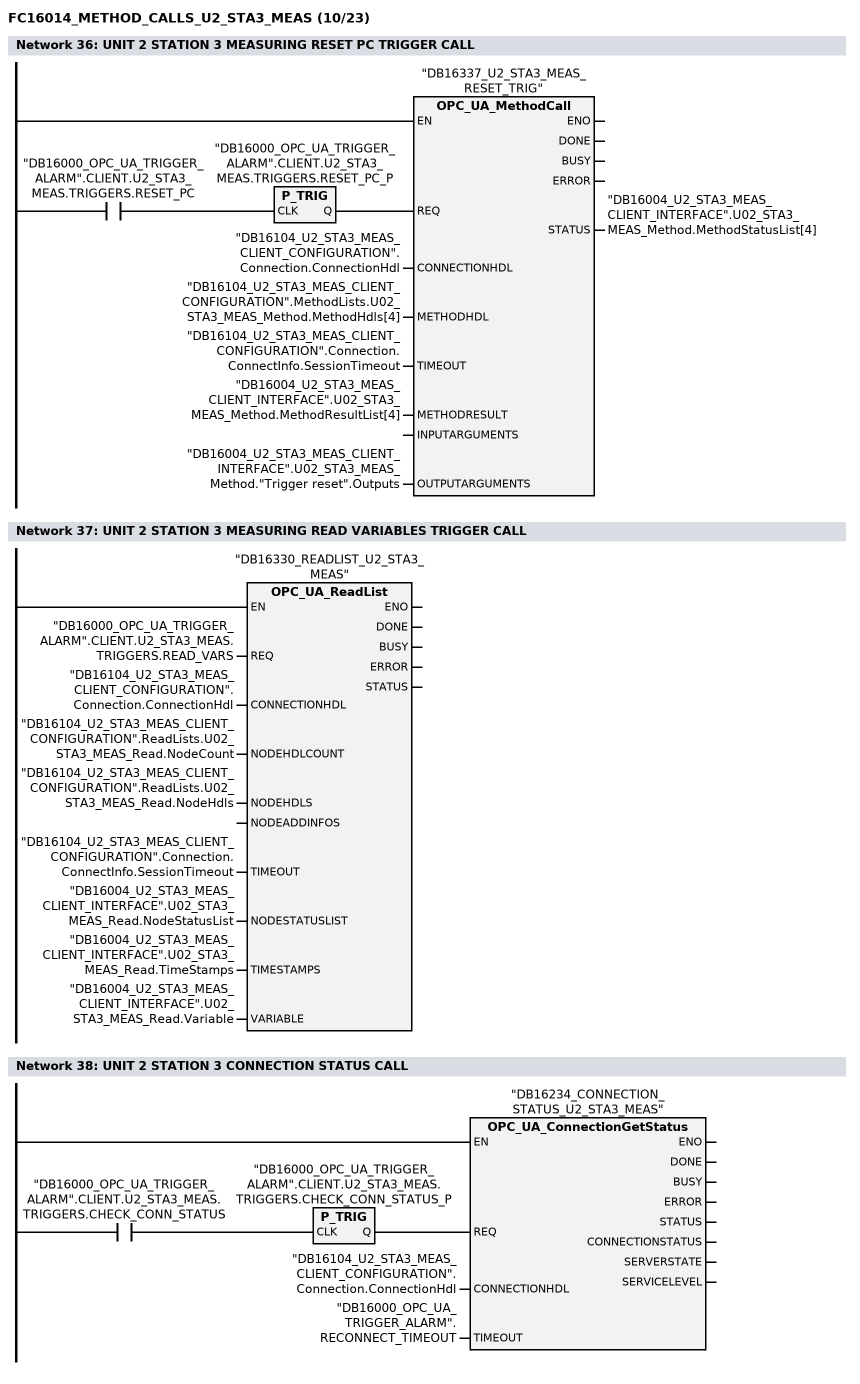
   RUNG wire#powerrail
      "DB16337_U2_STA3_MEAS_RESET_TRIG".OPC_UA_MethodCall(REQ := wire#w1, ConnectionHdl := "DB16104_U2_STA3_MEAS_CLIENT_CONFIGURATION".Connection.ConnectionHdl, MethodHdl := "DB16104_U2_STA3_MEAS_CLIENT_CONFIGURATION".MethodLists.U02_STA3_MEAS_Method.MethodHdls[4], Timeout := "DB16104_U2_STA3_MEAS_CLIENT_CONFIGURATION".Connection.ConnectInfo.SessionTimeout, MethodResult := "DB16004_U2_STA3_MEAS_CLIENT_INTERFACE".U02_STA3_MEAS_Method.MethodResultList[4], InputArguments :=, OutputArguments := "DB16004_U2_STA3_MEAS_CLIENT_INTERFACE".U02_STA3_MEAS_Method."Trigger reset".Outputs, Done =>, Busy =>, Error =>, Status => "DB16004_U2_STA3_MEAS_CLIENT_INTERFACE".U02_STA3_MEAS_Method.MethodStatusList[4])
   END_RUNG
   RUNG wire#powerrail
      Contact( "DB16000_OPC_UA_TRIGGER_ALARM".CLIENT.U2_STA3_MEAS.TRIGGERS.RESET_PC )
      P_Trig( "DB16000_OPC_UA_TRIGGER_ALARM".CLIENT.U2_STA3_MEAS.TRIGGERS.RESET_PC_P )
   END_RUNG wire#w1
   // the same network as SCL:
   #_w1 := "DB16000_OPC_UA_TRIGGER_ALARM".CLIENT.U2_STA3_MEAS.TRIGGERS.RESET_PC AND NOT "DB16000_OPC_UA_TRIGGER_ALARM".CLIENT.U2_STA3_MEAS.TRIGGERS.RESET_PC_P;   // rising edge
   "DB16000_OPC_UA_TRIGGER_ALARM".CLIENT.U2_STA3_MEAS.TRIGGERS.RESET_PC_P := "DB16000_OPC_UA_TRIGGER_ALARM".CLIENT.U2_STA3_MEAS.TRIGGERS.RESET_PC;
   "DB16337_U2_STA3_MEAS_RESET_TRIG"(REQ := #_w1,   // OPC_UA_MethodCall
                           ConnectionHdl := "DB16104_U2_STA3_MEAS_CLIENT_CONFIGURATION".Connection.ConnectionHdl,
                           MethodHdl := "DB16104_U2_STA3_MEAS_CLIENT_CONFIGURATION".MethodLists.U02_STA3_MEAS_Method.MethodHdls[4],
                           Timeout := "DB16104_U2_STA3_MEAS_CLIENT_CONFIGURATION".Connection.ConnectInfo.SessionTimeout,
                           MethodResult := "DB16004_U2_STA3_MEAS_CLIENT_INTERFACE".U02_STA3_MEAS_Method.MethodResultList[4],
                           OutputArguments := "DB16004_U2_STA3_MEAS_CLIENT_INTERFACE".U02_STA3_MEAS_Method."Trigger reset".Outputs,
                           Status => "DB16004_U2_STA3_MEAS_CLIENT_INTERFACE".U02_STA3_MEAS_Method.MethodStatusList[4]);
END_REGION

REGION Network 37: UNIT 2 STATION 3 MEASURING READ VARIABLES TRIGGER CALL
   RUNG wire#powerrail
      "DB16330_READLIST_U2_STA3_MEAS".OPC_UA_ReadList(REQ := "DB16000_OPC_UA_TRIGGER_ALARM".CLIENT.U2_STA3_MEAS.TRIGGERS.READ_VARS, ConnectionHdl := "DB16104_U2_STA3_MEAS_CLIENT_CONFIGURATION".Connection.ConnectionHdl, NodeHdlCount := "DB16104_U2_STA3_MEAS_CLIENT_CONFIGURATION".ReadLists.U02_STA3_MEAS_Read.NodeCount, NodeHdls := "DB16104_U2_STA3_MEAS_CLIENT_CONFIGURATION".ReadLists.U02_STA3_MEAS_Read.NodeHdls, NodeAddInfos :=, Timeout := "DB16104_U2_STA3_MEAS_CLIENT_CONFIGURATION".Connection.ConnectInfo.SessionTimeout, NodeStatusList := "DB16004_U2_STA3_MEAS_CLIENT_INTERFACE".U02_STA3_MEAS_Read.NodeStatusList, TimeStamps := "DB16004_U2_STA3_MEAS_CLIENT_INTERFACE".U02_STA3_MEAS_Read.TimeStamps, Variable := "DB16004_U2_STA3_MEAS_CLIENT_INTERFACE".U02_STA3_MEAS_Read.Variable, Done =>, Busy =>, Error =>, Status =>)
   END_RUNG
   // the same network as SCL:
   "DB16330_READLIST_U2_STA3_MEAS"(REQ := "DB16000_OPC_UA_TRIGGER_ALARM".CLIENT.U2_STA3_MEAS.TRIGGERS.READ_VARS,   // OPC_UA_ReadList
                           ConnectionHdl := "DB16104_U2_STA3_MEAS_CLIENT_CONFIGURATION".Connection.ConnectionHdl,
                           NodeHdlCount := "DB16104_U2_STA3_MEAS_CLIENT_CONFIGURATION".ReadLists.U02_STA3_MEAS_Read.NodeCount,
                           NodeHdls := "DB16104_U2_STA3_MEAS_CLIENT_CONFIGURATION".ReadLists.U02_STA3_MEAS_Read.NodeHdls,
                           Timeout := "DB16104_U2_STA3_MEAS_CLIENT_CONFIGURATION".Connection.ConnectInfo.SessionTimeout,
                           NodeStatusList := "DB16004_U2_STA3_MEAS_CLIENT_INTERFACE".U02_STA3_MEAS_Read.NodeStatusList,
                           TimeStamps := "DB16004_U2_STA3_MEAS_CLIENT_INTERFACE".U02_STA3_MEAS_Read.TimeStamps,
                           Variable := "DB16004_U2_STA3_MEAS_CLIENT_INTERFACE".U02_STA3_MEAS_Read.Variable);
END_REGION

REGION Network 38: UNIT 2 STATION 3 CONNECTION STATUS CALL
   RUNG wire#powerrail
      "DB16234_CONNECTION_STATUS_U2_STA3_MEAS".OPC_UA_ConnectionGetStatus(REQ := wire#w1, ConnectionHdl := "DB16104_U2_STA3_MEAS_CLIENT_CONFIGURATION".Connection.ConnectionHdl, Timeout := "DB16000_OPC_UA_TRIGGER_ALARM".RECONNECT_TIMEOUT, Done =>, Busy =>, Error =>, Status =>, ConnectionStatus =>, ServerState =>, ServiceLevel =>)
   END_RUNG
   RUNG wire#powerrail
      Contact( "DB16000_OPC_UA_TRIGGER_ALARM".CLIENT.U2_STA3_MEAS.TRIGGERS.CHECK_CONN_STATUS )
      P_Trig( "DB16000_OPC_UA_TRIGGER_ALARM".CLIENT.U2_STA3_MEAS.TRIGGERS.CHECK_CONN_STATUS_P )
   END_RUNG wire#w1
   // the same network as SCL:
   #_w1 := "DB16000_OPC_UA_TRIGGER_ALARM".CLIENT.U2_STA3_MEAS.TRIGGERS.CHECK_CONN_STATUS AND NOT "DB16000_OPC_UA_TRIGGER_ALARM".CLIENT.U2_STA3_MEAS.TRIGGERS.CHECK_CONN_STATUS_P;   // rising edge
   "DB16000_OPC_UA_TRIGGER_ALARM".CLIENT.U2_STA3_MEAS.TRIGGERS.CHECK_CONN_STATUS_P := "DB16000_OPC_UA_TRIGGER_ALARM".CLIENT.U2_STA3_MEAS.TRIGGERS.CHECK_CONN_STATUS;
   "DB16234_CONNECTION_STATUS_U2_STA3_MEAS"(REQ := #_w1,   // OPC_UA_ConnectionGetStatus
                           ConnectionHdl := "DB16104_U2_STA3_MEAS_CLIENT_CONFIGURATION".Connection.ConnectionHdl,
                           Timeout := "DB16000_OPC_UA_TRIGGER_ALARM".RECONNECT_TIMEOUT);
END_REGION

REGION Network 39: UNIT 2 STATION 3 RELEASE HANDLE LIST CALL
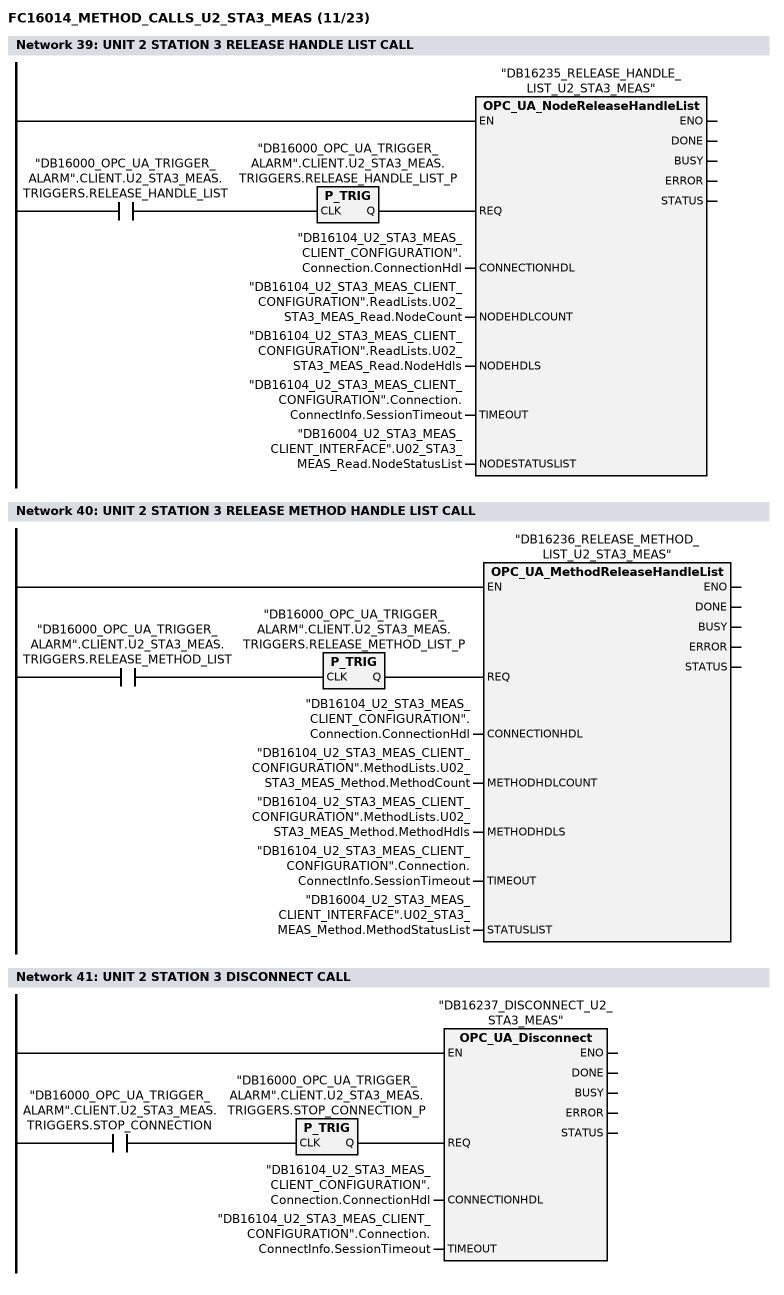
   RUNG wire#powerrail
      "DB16235_RELEASE_HANDLE_LIST_U2_STA3_MEAS".OPC_UA_NodeReleaseHandleList(REQ := wire#w1, ConnectionHdl := "DB16104_U2_STA3_MEAS_CLIENT_CONFIGURATION".Connection.ConnectionHdl, NodeHdlCount := "DB16104_U2_STA3_MEAS_CLIENT_CONFIGURATION".ReadLists.U02_STA3_MEAS_Read.NodeCount, NodeHdls := "DB16104_U2_STA3_MEAS_CLIENT_CONFIGURATION".ReadLists.U02_STA3_MEAS_Read.NodeHdls, Timeout := "DB16104_U2_STA3_MEAS_CLIENT_CONFIGURATION".Connection.ConnectInfo.SessionTimeout, NodeStatusList := "DB16004_U2_STA3_MEAS_CLIENT_INTERFACE".U02_STA3_MEAS_Read.NodeStatusList, Done =>, Busy =>, Error =>, Status =>)
   END_RUNG
   RUNG wire#powerrail
      Contact( "DB16000_OPC_UA_TRIGGER_ALARM".CLIENT.U2_STA3_MEAS.TRIGGERS.RELEASE_HANDLE_LIST )
      P_Trig( "DB16000_OPC_UA_TRIGGER_ALARM".CLIENT.U2_STA3_MEAS.TRIGGERS.RELEASE_HANDLE_LIST_P )
   END_RUNG wire#w1
   // the same network as SCL:
   #_w1 := "DB16000_OPC_UA_TRIGGER_ALARM".CLIENT.U2_STA3_MEAS.TRIGGERS.RELEASE_HANDLE_LIST AND NOT "DB16000_OPC_UA_TRIGGER_ALARM".CLIENT.U2_STA3_MEAS.TRIGGERS.RELEASE_HANDLE_LIST_P;   // rising edge
   "DB16000_OPC_UA_TRIGGER_ALARM".CLIENT.U2_STA3_MEAS.TRIGGERS.RELEASE_HANDLE_LIST_P := "DB16000_OPC_UA_TRIGGER_ALARM".CLIENT.U2_STA3_MEAS.TRIGGERS.RELEASE_HANDLE_LIST;
   "DB16235_RELEASE_HANDLE_LIST_U2_STA3_MEAS"(REQ := #_w1,   // OPC_UA_NodeReleaseHandleList
                           ConnectionHdl := "DB16104_U2_STA3_MEAS_CLIENT_CONFIGURATION".Connection.ConnectionHdl,
                           NodeHdlCount := "DB16104_U2_STA3_MEAS_CLIENT_CONFIGURATION".ReadLists.U02_STA3_MEAS_Read.NodeCount,
                           NodeHdls := "DB16104_U2_STA3_MEAS_CLIENT_CONFIGURATION".ReadLists.U02_STA3_MEAS_Read.NodeHdls,
                           Timeout := "DB16104_U2_STA3_MEAS_CLIENT_CONFIGURATION".Connection.ConnectInfo.SessionTimeout,
                           NodeStatusList := "DB16004_U2_STA3_MEAS_CLIENT_INTERFACE".U02_STA3_MEAS_Read.NodeStatusList);
END_REGION

REGION Network 40: UNIT 2 STATION 3 RELEASE METHOD HANDLE LIST CALL
   RUNG wire#powerrail
      "DB16236_RELEASE_METHOD_LIST_U2_STA3_MEAS".OPC_UA_MethodReleaseHandleList(REQ := wire#w1, ConnectionHdl := "DB16104_U2_STA3_MEAS_CLIENT_CONFIGURATION".Connection.ConnectionHdl, MethodHdlCount := "DB16104_U2_STA3_MEAS_CLIENT_CONFIGURATION".MethodLists.U02_STA3_MEAS_Method.MethodCount, MethodHdls := "DB16104_U2_STA3_MEAS_CLIENT_CONFIGURATION".MethodLists.U02_STA3_MEAS_Method.MethodHdls, Timeout := "DB16104_U2_STA3_MEAS_CLIENT_CONFIGURATION".Connection.ConnectInfo.SessionTimeout, StatusList := "DB16004_U2_STA3_MEAS_CLIENT_INTERFACE".U02_STA3_MEAS_Method.MethodStatusList, Done =>, Busy =>, Error =>, Status =>)
   END_RUNG
   RUNG wire#powerrail
      Contact( "DB16000_OPC_UA_TRIGGER_ALARM".CLIENT.U2_STA3_MEAS.TRIGGERS.RELEASE_METHOD_LIST )
      P_Trig( "DB16000_OPC_UA_TRIGGER_ALARM".CLIENT.U2_STA3_MEAS.TRIGGERS.RELEASE_METHOD_LIST_P )
   END_RUNG wire#w1
   // the same network as SCL:
   #_w1 := "DB16000_OPC_UA_TRIGGER_ALARM".CLIENT.U2_STA3_MEAS.TRIGGERS.RELEASE_METHOD_LIST AND NOT "DB16000_OPC_UA_TRIGGER_ALARM".CLIENT.U2_STA3_MEAS.TRIGGERS.RELEASE_METHOD_LIST_P;   // rising edge
   "DB16000_OPC_UA_TRIGGER_ALARM".CLIENT.U2_STA3_MEAS.TRIGGERS.RELEASE_METHOD_LIST_P := "DB16000_OPC_UA_TRIGGER_ALARM".CLIENT.U2_STA3_MEAS.TRIGGERS.RELEASE_METHOD_LIST;
   "DB16236_RELEASE_METHOD_LIST_U2_STA3_MEAS"(REQ := #_w1,   // OPC_UA_MethodReleaseHandleList
                           ConnectionHdl := "DB16104_U2_STA3_MEAS_CLIENT_CONFIGURATION".Connection.ConnectionHdl,
                           MethodHdlCount := "DB16104_U2_STA3_MEAS_CLIENT_CONFIGURATION".MethodLists.U02_STA3_MEAS_Method.MethodCount,
                           MethodHdls := "DB16104_U2_STA3_MEAS_CLIENT_CONFIGURATION".MethodLists.U02_STA3_MEAS_Method.MethodHdls,
                           Timeout := "DB16104_U2_STA3_MEAS_CLIENT_CONFIGURATION".Connection.ConnectInfo.SessionTimeout,
                           StatusList := "DB16004_U2_STA3_MEAS_CLIENT_INTERFACE".U02_STA3_MEAS_Method.MethodStatusList);
END_REGION

REGION Network 41: UNIT 2 STATION 3 DISCONNECT CALL
   RUNG wire#powerrail
      "DB16237_DISCONNECT_U2_STA3_MEAS".OPC_UA_Disconnect(REQ := wire#w1, ConnectionHdl := "DB16104_U2_STA3_MEAS_CLIENT_CONFIGURATION".Connection.ConnectionHdl, Timeout := "DB16104_U2_STA3_MEAS_CLIENT_CONFIGURATION".Connection.ConnectInfo.SessionTimeout, Done =>, Busy =>, Error =>, Status =>)
   END_RUNG
   RUNG wire#powerrail
      Contact( "DB16000_OPC_UA_TRIGGER_ALARM".CLIENT.U2_STA3_MEAS.TRIGGERS.STOP_CONNECTION )
      P_Trig( "DB16000_OPC_UA_TRIGGER_ALARM".CLIENT.U2_STA3_MEAS.TRIGGERS.STOP_CONNECTION_P )
   END_RUNG wire#w1
   // the same network as SCL:
   #_w1 := "DB16000_OPC_UA_TRIGGER_ALARM".CLIENT.U2_STA3_MEAS.TRIGGERS.STOP_CONNECTION AND NOT "DB16000_OPC_UA_TRIGGER_ALARM".CLIENT.U2_STA3_MEAS.TRIGGERS.STOP_CONNECTION_P;   // rising edge
   "DB16000_OPC_UA_TRIGGER_ALARM".CLIENT.U2_STA3_MEAS.TRIGGERS.STOP_CONNECTION_P := "DB16000_OPC_UA_TRIGGER_ALARM".CLIENT.U2_STA3_MEAS.TRIGGERS.STOP_CONNECTION;
   "DB16237_DISCONNECT_U2_STA3_MEAS"(REQ := #_w1,   // OPC_UA_Disconnect
                           ConnectionHdl := "DB16104_U2_STA3_MEAS_CLIENT_CONFIGURATION".Connection.ConnectionHdl,
                           Timeout := "DB16104_U2_STA3_MEAS_CLIENT_CONFIGURATION".Connection.ConnectInfo.SessionTimeout);
END_REGION

REGION Network 42: UNIT 2 STATION 3 MEAS RECONNECT
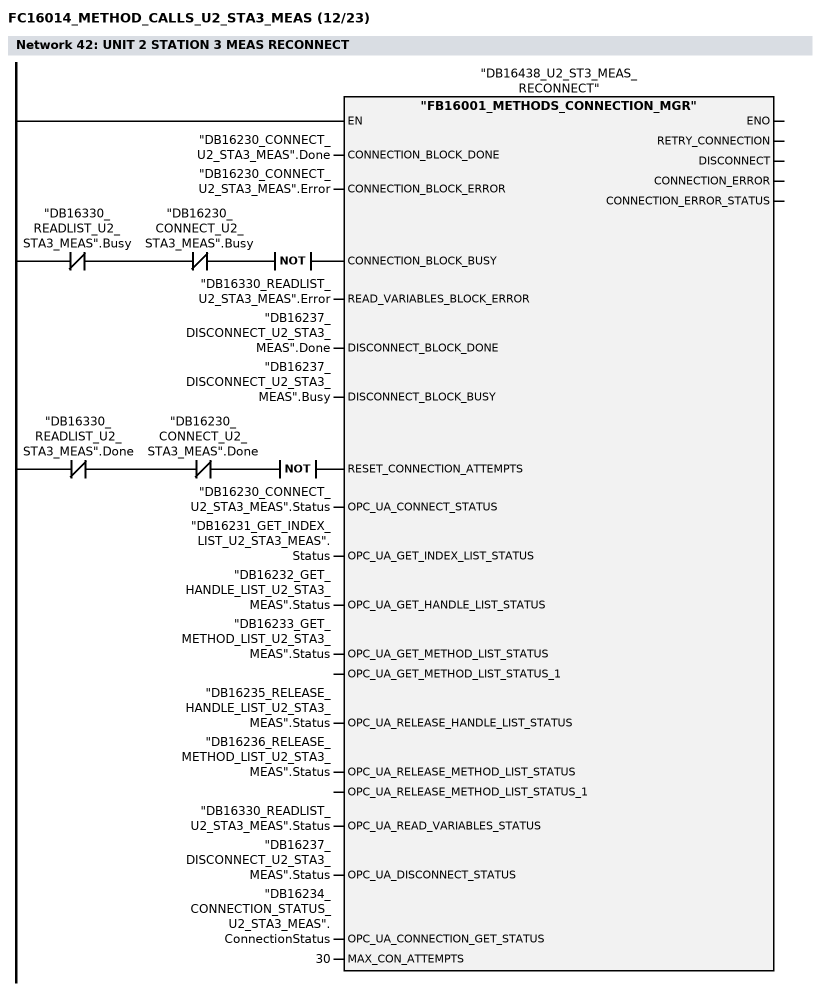
   RUNG wire#powerrail
      "DB16438_U2_ST3_MEAS_RECONNECT"(CONNECTION_BLOCK_BUSY := wire#w1, RESET_CONNECTION_ATTEMPTS := wire#w2, CONNECTION_BLOCK_DONE := "DB16230_CONNECT_U2_STA3_MEAS".Done, CONNECTION_BLOCK_ERROR := "DB16230_CONNECT_U2_STA3_MEAS".Error, READ_VARIABLES_BLOCK_ERROR := "DB16330_READLIST_U2_STA3_MEAS".Error, DISCONNECT_BLOCK_DONE := "DB16237_DISCONNECT_U2_STA3_MEAS".Done, DISCONNECT_BLOCK_BUSY := "DB16237_DISCONNECT_U2_STA3_MEAS".Busy, OPC_UA_CONNECT_STATUS := "DB16230_CONNECT_U2_STA3_MEAS".Status, OPC_UA_GET_INDEX_LIST_STATUS := "DB16231_GET_INDEX_LIST_U2_STA3_MEAS".Status, OPC_UA_GET_HANDLE_LIST_STATUS := "DB16232_GET_HANDLE_LIST_U2_STA3_MEAS".Status, OPC_UA_GET_METHOD_LIST_STATUS := "DB16233_GET_METHOD_LIST_U2_STA3_MEAS".Status, OPC_UA_GET_METHOD_LIST_STATUS_1 :=, OPC_UA_RELEASE_HANDLE_LIST_STATUS := "DB16235_RELEASE_HANDLE_LIST_U2_STA3_MEAS".Status, OPC_UA_RELEASE_METHOD_LIST_STATUS := "DB16236_RELEASE_METHOD_LIST_U2_STA3_MEAS".Status, OPC_UA_RELEASE_METHOD_LIST_STATUS_1 :=, OPC_UA_READ_VARIABLES_STATUS := "DB16330_READLIST_U2_STA3_MEAS".Status, OPC_UA_DISCONNECT_STATUS := "DB16237_DISCONNECT_U2_STA3_MEAS".Status, OPC_UA_CONNECTION_GET_STATUS := "DB16234_CONNECTION_STATUS_U2_STA3_MEAS".ConnectionStatus, MAX_CON_ATTEMPTS := 30, RETRY_CONNECTION =>, DISCONNECT =>, CONNECTION_ERROR =>, CONNECTION_ERROR_STATUS =>)
   END_RUNG
   RUNG wire#powerrail
      I_Contact( "DB16330_READLIST_U2_STA3_MEAS".Busy )
      I_Contact( "DB16230_CONNECT_U2_STA3_MEAS".Busy )
      Not()
   END_RUNG wire#w1
   RUNG wire#powerrail
      I_Contact( "DB16330_READLIST_U2_STA3_MEAS".Done )
      I_Contact( "DB16230_CONNECT_U2_STA3_MEAS".Done )
      Not()
   END_RUNG wire#w2
   // the same network as SCL:
   "DB16438_U2_ST3_MEAS_RECONNECT"(CONNECTION_BLOCK_DONE := "DB16230_CONNECT_U2_STA3_MEAS".Done,   // "FB16001_METHODS_CONNECTION_MGR"
                           CONNECTION_BLOCK_ERROR := "DB16230_CONNECT_U2_STA3_MEAS".Error,
                           CONNECTION_BLOCK_BUSY := NOT (NOT "DB16330_READLIST_U2_STA3_MEAS".Busy AND NOT "DB16230_CONNECT_U2_STA3_MEAS".Busy),
                           READ_VARIABLES_BLOCK_ERROR := "DB16330_READLIST_U2_STA3_MEAS".Error,
                           DISCONNECT_BLOCK_DONE := "DB16237_DISCONNECT_U2_STA3_MEAS".Done,
                           DISCONNECT_BLOCK_BUSY := "DB16237_DISCONNECT_U2_STA3_MEAS".Busy,
                           RESET_CONNECTION_ATTEMPTS := NOT (NOT "DB16330_READLIST_U2_STA3_MEAS".Done AND NOT "DB16230_CONNECT_U2_STA3_MEAS".Done),
                           OPC_UA_CONNECT_STATUS := "DB16230_CONNECT_U2_STA3_MEAS".Status,
                           OPC_UA_GET_INDEX_LIST_STATUS := "DB16231_GET_INDEX_LIST_U2_STA3_MEAS".Status,
                           OPC_UA_GET_HANDLE_LIST_STATUS := "DB16232_GET_HANDLE_LIST_U2_STA3_MEAS".Status,
                           OPC_UA_GET_METHOD_LIST_STATUS := "DB16233_GET_METHOD_LIST_U2_STA3_MEAS".Status,
                           OPC_UA_RELEASE_HANDLE_LIST_STATUS := "DB16235_RELEASE_HANDLE_LIST_U2_STA3_MEAS".Status,
                           OPC_UA_RELEASE_METHOD_LIST_STATUS := "DB16236_RELEASE_METHOD_LIST_U2_STA3_MEAS".Status,
                           OPC_UA_READ_VARIABLES_STATUS := "DB16330_READLIST_U2_STA3_MEAS".Status,
                           OPC_UA_DISCONNECT_STATUS := "DB16237_DISCONNECT_U2_STA3_MEAS".Status,
                           OPC_UA_CONNECTION_GET_STATUS := "DB16234_CONNECTION_STATUS_U2_STA3_MEAS".ConnectionStatus,
                           MAX_CON_ATTEMPTS := 30);
END_REGION

REGION Network 43: UNIT 2 NOOZLE SURFACE DISTANCE UPDATE
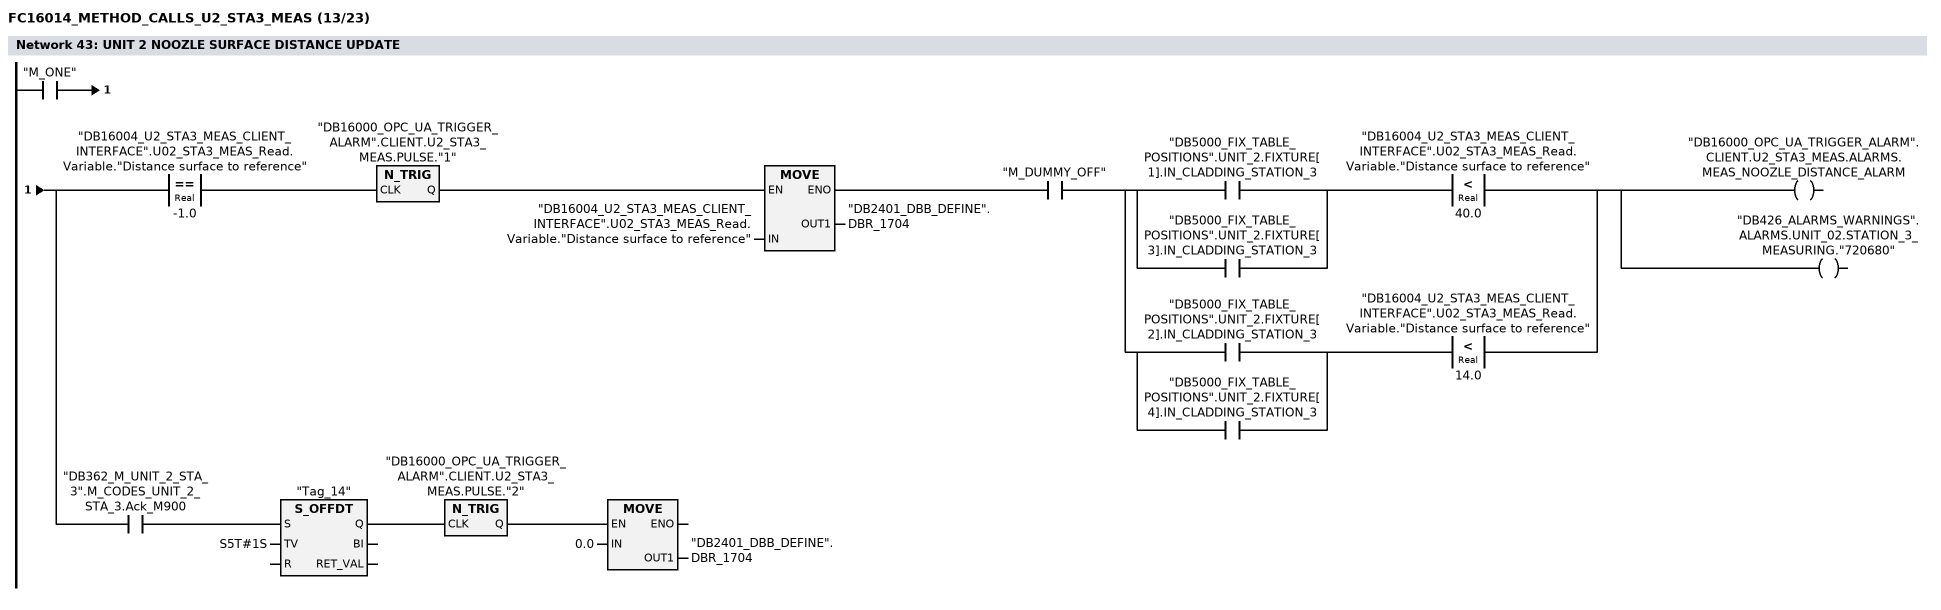
   RUNG wire#powerrail
      Contact( "M_ONE" )
      wire#w1
      { S7_Templates := "SrcType := Real" } EQ_Contact(in1 := "DB16004_U2_STA3_MEAS_CLIENT_INTERFACE".U02_STA3_MEAS_Read.Variable."Distance surface to reference", in2 := -1.0)
      N_Trig( "DB16000_OPC_UA_TRIGGER_ALARM".CLIENT.U2_STA3_MEAS.PULSE."1" )
      Move(in := "DB16004_U2_STA3_MEAS_CLIENT_INTERFACE".U02_STA3_MEAS_Read.Variable."Distance surface to reference", out1 => "DB2401_DBB_DEFINE".DBR_1704)
      Contact( "M_DUMMY_OFF" )
      wire#w2
      Contact( "DB5000_FIX_TABLE_POSITIONS".UNIT_2.FIXTURE[1].IN_CLADDING_STATION_3 )
      wire#w3
      { S7_Templates := "SrcType := Real" } LT_Contact(in1 := "DB16004_U2_STA3_MEAS_CLIENT_INTERFACE".U02_STA3_MEAS_Read.Variable."Distance surface to reference", in2 := 40.0)
      wire#w4
      Coil( "DB16000_OPC_UA_TRIGGER_ALARM".CLIENT.U2_STA3_MEAS.ALARMS.MEAS_NOOZLE_DISTANCE_ALARM )
   END_RUNG
   RUNG wire#w2
      Contact( "DB5000_FIX_TABLE_POSITIONS".UNIT_2.FIXTURE[3].IN_CLADDING_STATION_3 )
   END_RUNG wire#w3
   RUNG wire#w2
      Contact( "DB5000_FIX_TABLE_POSITIONS".UNIT_2.FIXTURE[2].IN_CLADDING_STATION_3 )
      wire#w5
      { S7_Templates := "SrcType := Real" } LT_Contact(in1 := "DB16004_U2_STA3_MEAS_CLIENT_INTERFACE".U02_STA3_MEAS_Read.Variable."Distance surface to reference", in2 := 14.0)
   END_RUNG wire#w4
   RUNG wire#w2
      Contact( "DB5000_FIX_TABLE_POSITIONS".UNIT_2.FIXTURE[4].IN_CLADDING_STATION_3 )
   END_RUNG wire#w5
   RUNG wire#w4
      Coil( "DB426_ALARMS_WARNINGS".ALARMS.UNIT_02.STATION_3_MEASURING."720680" )
   END_RUNG
   RUNG wire#w1
      Contact( "DB362_M_UNIT_2_STA_3".M_CODES_UNIT_2_STA_3.Ack_M900 )
      S_OFFDT(T_NO := "Tag_14", TV := S5T#1S, R :=, BI =>, RET_VAL =>)
      N_Trig( "DB16000_OPC_UA_TRIGGER_ALARM".CLIENT.U2_STA3_MEAS.PULSE."2" )
      Move(in := 0.0, out1 => "DB2401_DBB_DEFINE".DBR_1704)
   END_RUNG
   // the same network as SCL:
   #_w1 := "M_ONE" AND ("DB16004_U2_STA3_MEAS_CLIENT_INTERFACE".U02_STA3_MEAS_Read.Variable."Distance surface to reference" = (-1.0));
   #_w2 := NOT #_w1 AND "DB16000_OPC_UA_TRIGGER_ALARM".CLIENT.U2_STA3_MEAS.PULSE."1";   // falling edge
   "DB16000_OPC_UA_TRIGGER_ALARM".CLIENT.U2_STA3_MEAS.PULSE."1" := #_w1;
   IF #_w2 THEN
       "DB2401_DBB_DEFINE".DBR_1704 := "DB16004_U2_STA3_MEAS_CLIENT_INTERFACE".U02_STA3_MEAS_Read.Variable."Distance surface to reference";
   END_IF;
   "DB16000_OPC_UA_TRIGGER_ALARM".CLIENT.U2_STA3_MEAS.ALARMS.MEAS_NOOZLE_DISTANCE_ALARM := #_w2 AND "M_DUMMY_OFF" AND ((("DB5000_FIX_TABLE_POSITIONS".UNIT_2.FIXTURE[1].IN_CLADDING_STATION_3 OR "DB5000_FIX_TABLE_POSITIONS".UNIT_2.FIXTURE[3].IN_CLADDING_STATION_3) AND ("DB16004_U2_STA3_MEAS_CLIENT_INTERFACE".U02_STA3_MEAS_Read.Variable."Distance surface to reference" < 40.0)) OR (("DB5000_FIX_TABLE_POSITIONS".UNIT_2.FIXTURE[2].IN_CLADDING_STATION_3 OR "DB5000_FIX_TABLE_POSITIONS".UNIT_2.FIXTURE[4].IN_CLADDING_STATION_3) AND ("DB16004_U2_STA3_MEAS_CLIENT_INTERFACE".U02_STA3_MEAS_Read.Variable."Distance surface to reference" < 14.0)));
   "DB426_ALARMS_WARNINGS".ALARMS.UNIT_02.STATION_3_MEASURING."720680" := "DB16000_OPC_UA_TRIGGER_ALARM".CLIENT.U2_STA3_MEAS.ALARMS.MEAS_NOOZLE_DISTANCE_ALARM;
   #_s5time1 := S_OFFDT(T_NO := "Tag_14",
                        S := "M_ONE" AND "DB362_M_UNIT_2_STA_3".M_CODES_UNIT_2_STA_3.Ack_M900,
                        TV := S5T#1S,
                        Q => #_w3);
   #_w4 := NOT #_w3 AND "DB16000_OPC_UA_TRIGGER_ALARM".CLIENT.U2_STA3_MEAS.PULSE."2";   // falling edge
   "DB16000_OPC_UA_TRIGGER_ALARM".CLIENT.U2_STA3_MEAS.PULSE."2" := #_w3;
   IF #_w4 THEN "DB2401_DBB_DEFINE".DBR_1704 := 0.0; END_IF;
END_REGION

REGION Network 44: UNIT 2 FIXTURES CALIBRATION STATUS UPDATE
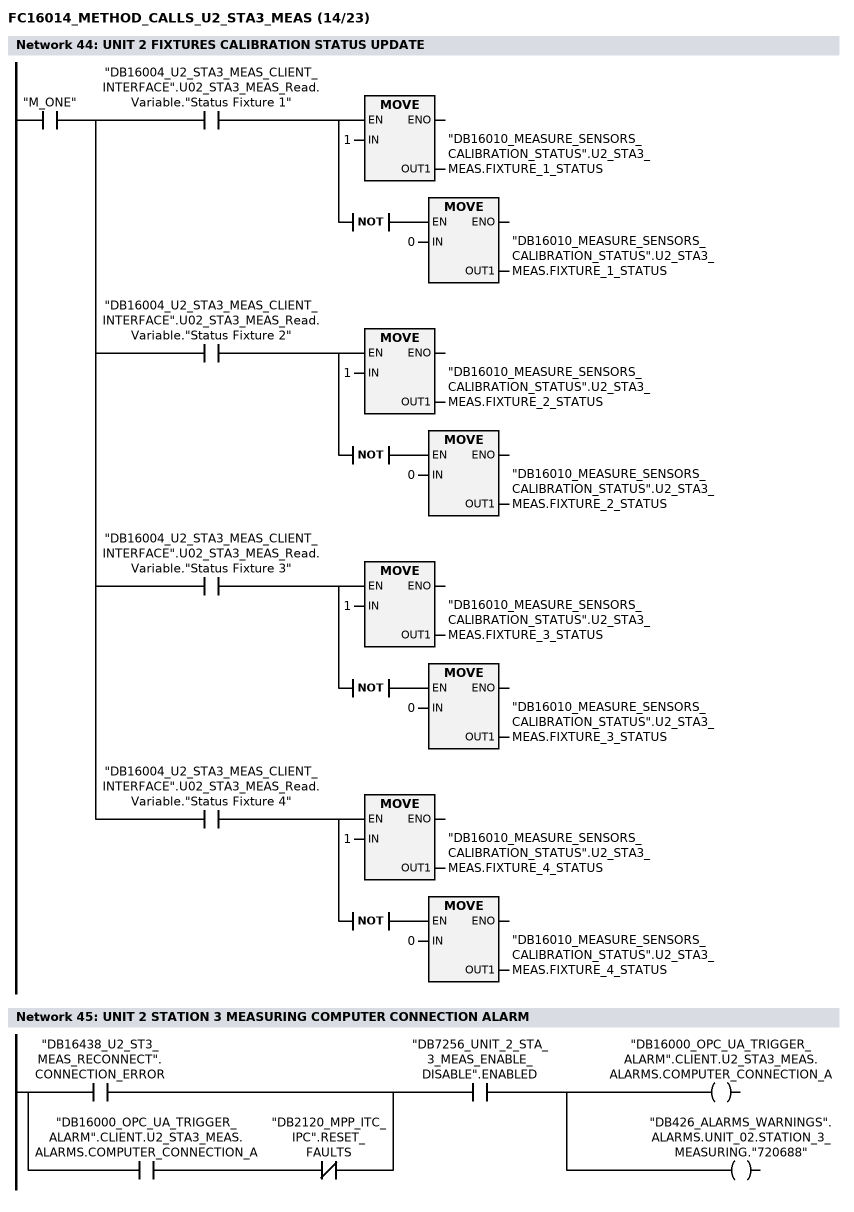
   RUNG wire#powerrail
      Contact( "M_ONE" )
      wire#w1
      Contact( "DB16004_U2_STA3_MEAS_CLIENT_INTERFACE".U02_STA3_MEAS_Read.Variable."Status Fixture 1" )
      wire#w2
      Move(in := 1, out1 => "DB16010_MEASURE_SENSORS_CALIBRATION_STATUS".U2_STA3_MEAS.FIXTURE_1_STATUS)
   END_RUNG
   RUNG wire#w2
      Not()
      Move(in := 0, out1 => "DB16010_MEASURE_SENSORS_CALIBRATION_STATUS".U2_STA3_MEAS.FIXTURE_1_STATUS)
   END_RUNG
   RUNG wire#w1
      Contact( "DB16004_U2_STA3_MEAS_CLIENT_INTERFACE".U02_STA3_MEAS_Read.Variable."Status Fixture 2" )
      wire#w3
      Move(in := 1, out1 => "DB16010_MEASURE_SENSORS_CALIBRATION_STATUS".U2_STA3_MEAS.FIXTURE_2_STATUS)
   END_RUNG
   RUNG wire#w3
      Not()
      Move(in := 0, out1 => "DB16010_MEASURE_SENSORS_CALIBRATION_STATUS".U2_STA3_MEAS.FIXTURE_2_STATUS)
   END_RUNG
   RUNG wire#w1
      Contact( "DB16004_U2_STA3_MEAS_CLIENT_INTERFACE".U02_STA3_MEAS_Read.Variable."Status Fixture 3" )
      wire#w4
      Move(in := 1, out1 => "DB16010_MEASURE_SENSORS_CALIBRATION_STATUS".U2_STA3_MEAS.FIXTURE_3_STATUS)
   END_RUNG
   RUNG wire#w4
      Not()
      Move(in := 0, out1 => "DB16010_MEASURE_SENSORS_CALIBRATION_STATUS".U2_STA3_MEAS.FIXTURE_3_STATUS)
   END_RUNG
   RUNG wire#w1
      Contact( "DB16004_U2_STA3_MEAS_CLIENT_INTERFACE".U02_STA3_MEAS_Read.Variable."Status Fixture 4" )
      wire#w5
      Move(in := 1, out1 => "DB16010_MEASURE_SENSORS_CALIBRATION_STATUS".U2_STA3_MEAS.FIXTURE_4_STATUS)
   END_RUNG
   RUNG wire#w5
      Not()
      Move(in := 0, out1 => "DB16010_MEASURE_SENSORS_CALIBRATION_STATUS".U2_STA3_MEAS.FIXTURE_4_STATUS)
   END_RUNG
   // the same network as SCL:
   #_w1 := "M_ONE" AND "DB16004_U2_STA3_MEAS_CLIENT_INTERFACE".U02_STA3_MEAS_Read.Variable."Status Fixture 1";
   IF #_w1 THEN "DB16010_MEASURE_SENSORS_CALIBRATION_STATUS".U2_STA3_MEAS.FIXTURE_1_STATUS := 1; END_IF;
   IF NOT #_w1 THEN "DB16010_MEASURE_SENSORS_CALIBRATION_STATUS".U2_STA3_MEAS.FIXTURE_1_STATUS := 0; END_IF;
   #_w2 := "M_ONE" AND "DB16004_U2_STA3_MEAS_CLIENT_INTERFACE".U02_STA3_MEAS_Read.Variable."Status Fixture 2";
   IF #_w2 THEN "DB16010_MEASURE_SENSORS_CALIBRATION_STATUS".U2_STA3_MEAS.FIXTURE_2_STATUS := 1; END_IF;
   IF NOT #_w2 THEN "DB16010_MEASURE_SENSORS_CALIBRATION_STATUS".U2_STA3_MEAS.FIXTURE_2_STATUS := 0; END_IF;
   #_w3 := "M_ONE" AND "DB16004_U2_STA3_MEAS_CLIENT_INTERFACE".U02_STA3_MEAS_Read.Variable."Status Fixture 3";
   IF #_w3 THEN "DB16010_MEASURE_SENSORS_CALIBRATION_STATUS".U2_STA3_MEAS.FIXTURE_3_STATUS := 1; END_IF;
   IF NOT #_w3 THEN "DB16010_MEASURE_SENSORS_CALIBRATION_STATUS".U2_STA3_MEAS.FIXTURE_3_STATUS := 0; END_IF;
   #_w4 := "M_ONE" AND "DB16004_U2_STA3_MEAS_CLIENT_INTERFACE".U02_STA3_MEAS_Read.Variable."Status Fixture 4";
   IF #_w4 THEN "DB16010_MEASURE_SENSORS_CALIBRATION_STATUS".U2_STA3_MEAS.FIXTURE_4_STATUS := 1; END_IF;
   IF NOT #_w4 THEN "DB16010_MEASURE_SENSORS_CALIBRATION_STATUS".U2_STA3_MEAS.FIXTURE_4_STATUS := 0; END_IF;
END_REGION

REGION Network 45: UNIT 2 STATION 3 MEASURING COMPUTER CONNECTION ALARM
   RUNG wire#powerrail
      Contact( "DB16438_U2_ST3_MEAS_RECONNECT".CONNECTION_ERROR )
      wire#w1
      Contact( "DB7256_UNIT_2_STA_3_MEAS_ENABLE_DISABLE".ENABLED )
      wire#w2
      Coil( "DB16000_OPC_UA_TRIGGER_ALARM".CLIENT.U2_STA3_MEAS.ALARMS.COMPUTER_CONNECTION_A )
   END_RUNG
   RUNG wire#powerrail
      Contact( "DB16000_OPC_UA_TRIGGER_ALARM".CLIENT.U2_STA3_MEAS.ALARMS.COMPUTER_CONNECTION_A )
      I_Contact( "DB2120_MPP_ITC_IPC".RESET_FAULTS )
   END_RUNG wire#w1
   RUNG wire#w2
      Coil( "DB426_ALARMS_WARNINGS".ALARMS.UNIT_02.STATION_3_MEASURING."720688" )
   END_RUNG
   // the same network as SCL:
   "DB16000_OPC_UA_TRIGGER_ALARM".CLIENT.U2_STA3_MEAS.ALARMS.COMPUTER_CONNECTION_A := ("DB16438_U2_ST3_MEAS_RECONNECT".CONNECTION_ERROR OR ("DB16000_OPC_UA_TRIGGER_ALARM".CLIENT.U2_STA3_MEAS.ALARMS.COMPUTER_CONNECTION_A AND NOT "DB2120_MPP_ITC_IPC".RESET_FAULTS)) AND "DB7256_UNIT_2_STA_3_MEAS_ENABLE_DISABLE".ENABLED;
   "DB426_ALARMS_WARNINGS".ALARMS.UNIT_02.STATION_3_MEASURING."720688" := "DB16000_OPC_UA_TRIGGER_ALARM".CLIENT.U2_STA3_MEAS.ALARMS.COMPUTER_CONNECTION_A;
END_REGION

REGION Network 46: UNIT 2 STATION 3 MEASURING COMPUTER GET INDEX LIST ALARM
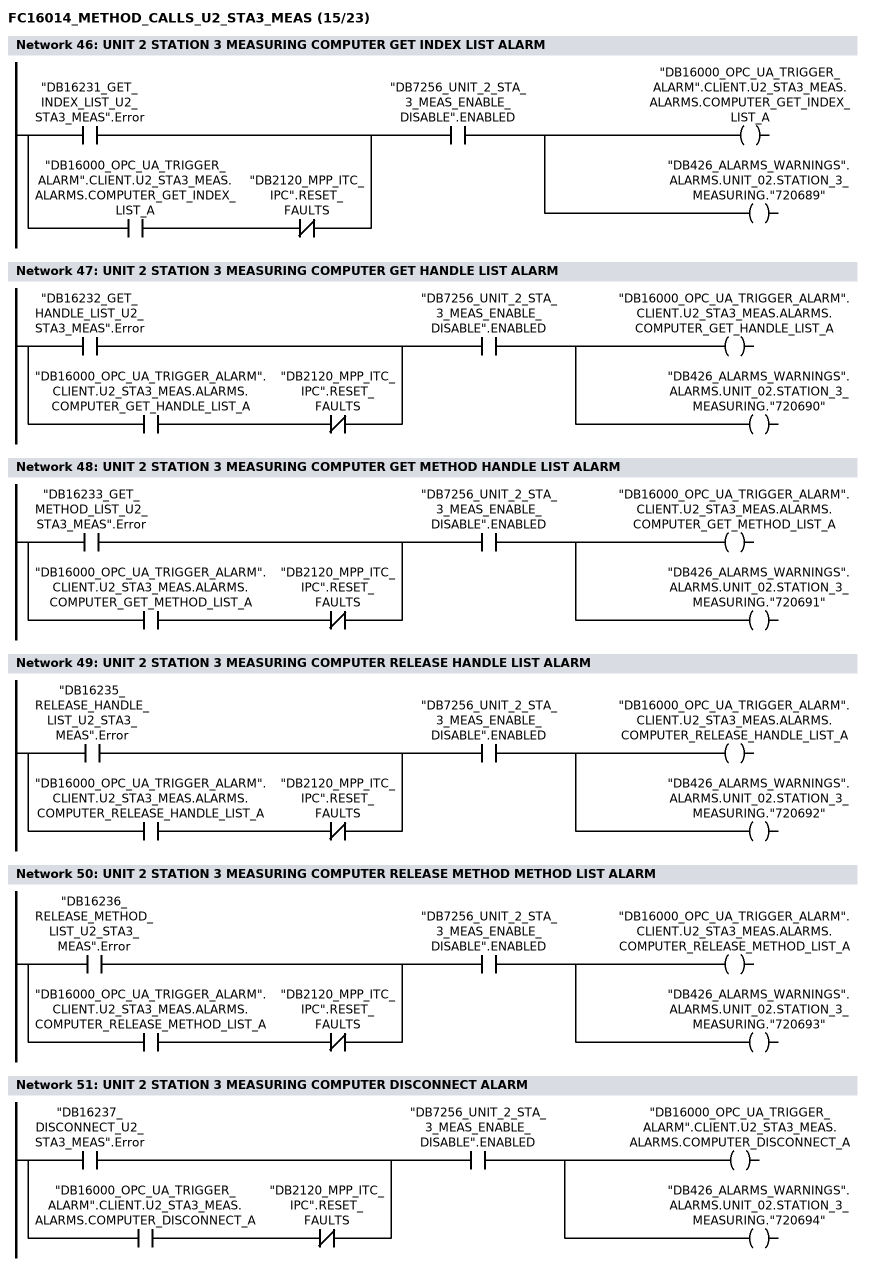
   RUNG wire#powerrail
      Contact( "DB16231_GET_INDEX_LIST_U2_STA3_MEAS".Error )
      wire#w1
      Contact( "DB7256_UNIT_2_STA_3_MEAS_ENABLE_DISABLE".ENABLED )
      wire#w2
      Coil( "DB16000_OPC_UA_TRIGGER_ALARM".CLIENT.U2_STA3_MEAS.ALARMS.COMPUTER_GET_INDEX_LIST_A )
   END_RUNG
   RUNG wire#powerrail
      Contact( "DB16000_OPC_UA_TRIGGER_ALARM".CLIENT.U2_STA3_MEAS.ALARMS.COMPUTER_GET_INDEX_LIST_A )
      I_Contact( "DB2120_MPP_ITC_IPC".RESET_FAULTS )
   END_RUNG wire#w1
   RUNG wire#w2
      Coil( "DB426_ALARMS_WARNINGS".ALARMS.UNIT_02.STATION_3_MEASURING."720689" )
   END_RUNG
   // the same network as SCL:
   "DB16000_OPC_UA_TRIGGER_ALARM".CLIENT.U2_STA3_MEAS.ALARMS.COMPUTER_GET_INDEX_LIST_A := ("DB16231_GET_INDEX_LIST_U2_STA3_MEAS".Error OR ("DB16000_OPC_UA_TRIGGER_ALARM".CLIENT.U2_STA3_MEAS.ALARMS.COMPUTER_GET_INDEX_LIST_A AND NOT "DB2120_MPP_ITC_IPC".RESET_FAULTS)) AND "DB7256_UNIT_2_STA_3_MEAS_ENABLE_DISABLE".ENABLED;
   "DB426_ALARMS_WARNINGS".ALARMS.UNIT_02.STATION_3_MEASURING."720689" := "DB16000_OPC_UA_TRIGGER_ALARM".CLIENT.U2_STA3_MEAS.ALARMS.COMPUTER_GET_INDEX_LIST_A;
END_REGION

REGION Network 47: UNIT 2 STATION 3 MEASURING COMPUTER GET HANDLE LIST ALARM
   RUNG wire#powerrail
      Contact( "DB16232_GET_HANDLE_LIST_U2_STA3_MEAS".Error )
      wire#w1
      Contact( "DB7256_UNIT_2_STA_3_MEAS_ENABLE_DISABLE".ENABLED )
      wire#w2
      Coil( "DB16000_OPC_UA_TRIGGER_ALARM".CLIENT.U2_STA3_MEAS.ALARMS.COMPUTER_GET_HANDLE_LIST_A )
   END_RUNG
   RUNG wire#powerrail
      Contact( "DB16000_OPC_UA_TRIGGER_ALARM".CLIENT.U2_STA3_MEAS.ALARMS.COMPUTER_GET_HANDLE_LIST_A )
      I_Contact( "DB2120_MPP_ITC_IPC".RESET_FAULTS )
   END_RUNG wire#w1
   RUNG wire#w2
      Coil( "DB426_ALARMS_WARNINGS".ALARMS.UNIT_02.STATION_3_MEASURING."720690" )
   END_RUNG
   // the same network as SCL:
   "DB16000_OPC_UA_TRIGGER_ALARM".CLIENT.U2_STA3_MEAS.ALARMS.COMPUTER_GET_HANDLE_LIST_A := ("DB16232_GET_HANDLE_LIST_U2_STA3_MEAS".Error OR ("DB16000_OPC_UA_TRIGGER_ALARM".CLIENT.U2_STA3_MEAS.ALARMS.COMPUTER_GET_HANDLE_LIST_A AND NOT "DB2120_MPP_ITC_IPC".RESET_FAULTS)) AND "DB7256_UNIT_2_STA_3_MEAS_ENABLE_DISABLE".ENABLED;
   "DB426_ALARMS_WARNINGS".ALARMS.UNIT_02.STATION_3_MEASURING."720690" := "DB16000_OPC_UA_TRIGGER_ALARM".CLIENT.U2_STA3_MEAS.ALARMS.COMPUTER_GET_HANDLE_LIST_A;
END_REGION

REGION Network 48: UNIT 2 STATION 3 MEASURING COMPUTER GET METHOD HANDLE LIST ALARM
   RUNG wire#powerrail
      Contact( "DB16233_GET_METHOD_LIST_U2_STA3_MEAS".Error )
      wire#w1
      Contact( "DB7256_UNIT_2_STA_3_MEAS_ENABLE_DISABLE".ENABLED )
      wire#w2
      Coil( "DB16000_OPC_UA_TRIGGER_ALARM".CLIENT.U2_STA3_MEAS.ALARMS.COMPUTER_GET_METHOD_LIST_A )
   END_RUNG
   RUNG wire#powerrail
      Contact( "DB16000_OPC_UA_TRIGGER_ALARM".CLIENT.U2_STA3_MEAS.ALARMS.COMPUTER_GET_METHOD_LIST_A )
      I_Contact( "DB2120_MPP_ITC_IPC".RESET_FAULTS )
   END_RUNG wire#w1
   RUNG wire#w2
      Coil( "DB426_ALARMS_WARNINGS".ALARMS.UNIT_02.STATION_3_MEASURING."720691" )
   END_RUNG
   // the same network as SCL:
   "DB16000_OPC_UA_TRIGGER_ALARM".CLIENT.U2_STA3_MEAS.ALARMS.COMPUTER_GET_METHOD_LIST_A := ("DB16233_GET_METHOD_LIST_U2_STA3_MEAS".Error OR ("DB16000_OPC_UA_TRIGGER_ALARM".CLIENT.U2_STA3_MEAS.ALARMS.COMPUTER_GET_METHOD_LIST_A AND NOT "DB2120_MPP_ITC_IPC".RESET_FAULTS)) AND "DB7256_UNIT_2_STA_3_MEAS_ENABLE_DISABLE".ENABLED;
   "DB426_ALARMS_WARNINGS".ALARMS.UNIT_02.STATION_3_MEASURING."720691" := "DB16000_OPC_UA_TRIGGER_ALARM".CLIENT.U2_STA3_MEAS.ALARMS.COMPUTER_GET_METHOD_LIST_A;
END_REGION

REGION Network 49: UNIT 2 STATION 3 MEASURING COMPUTER RELEASE HANDLE LIST ALARM
   RUNG wire#powerrail
      Contact( "DB16235_RELEASE_HANDLE_LIST_U2_STA3_MEAS".Error )
      wire#w1
      Contact( "DB7256_UNIT_2_STA_3_MEAS_ENABLE_DISABLE".ENABLED )
      wire#w2
      Coil( "DB16000_OPC_UA_TRIGGER_ALARM".CLIENT.U2_STA3_MEAS.ALARMS.COMPUTER_RELEASE_HANDLE_LIST_A )
   END_RUNG
   RUNG wire#powerrail
      Contact( "DB16000_OPC_UA_TRIGGER_ALARM".CLIENT.U2_STA3_MEAS.ALARMS.COMPUTER_RELEASE_HANDLE_LIST_A )
      I_Contact( "DB2120_MPP_ITC_IPC".RESET_FAULTS )
   END_RUNG wire#w1
   RUNG wire#w2
      Coil( "DB426_ALARMS_WARNINGS".ALARMS.UNIT_02.STATION_3_MEASURING."720692" )
   END_RUNG
   // the same network as SCL:
   "DB16000_OPC_UA_TRIGGER_ALARM".CLIENT.U2_STA3_MEAS.ALARMS.COMPUTER_RELEASE_HANDLE_LIST_A := ("DB16235_RELEASE_HANDLE_LIST_U2_STA3_MEAS".Error OR ("DB16000_OPC_UA_TRIGGER_ALARM".CLIENT.U2_STA3_MEAS.ALARMS.COMPUTER_RELEASE_HANDLE_LIST_A AND NOT "DB2120_MPP_ITC_IPC".RESET_FAULTS)) AND "DB7256_UNIT_2_STA_3_MEAS_ENABLE_DISABLE".ENABLED;
   "DB426_ALARMS_WARNINGS".ALARMS.UNIT_02.STATION_3_MEASURING."720692" := "DB16000_OPC_UA_TRIGGER_ALARM".CLIENT.U2_STA3_MEAS.ALARMS.COMPUTER_RELEASE_HANDLE_LIST_A;
END_REGION

REGION Network 50: UNIT 2 STATION 3 MEASURING COMPUTER RELEASE METHOD METHOD LIST ALARM
   RUNG wire#powerrail
      Contact( "DB16236_RELEASE_METHOD_LIST_U2_STA3_MEAS".Error )
      wire#w1
      Contact( "DB7256_UNIT_2_STA_3_MEAS_ENABLE_DISABLE".ENABLED )
      wire#w2
      Coil( "DB16000_OPC_UA_TRIGGER_ALARM".CLIENT.U2_STA3_MEAS.ALARMS.COMPUTER_RELEASE_METHOD_LIST_A )
   END_RUNG
   RUNG wire#powerrail
      Contact( "DB16000_OPC_UA_TRIGGER_ALARM".CLIENT.U2_STA3_MEAS.ALARMS.COMPUTER_RELEASE_METHOD_LIST_A )
      I_Contact( "DB2120_MPP_ITC_IPC".RESET_FAULTS )
   END_RUNG wire#w1
   RUNG wire#w2
      Coil( "DB426_ALARMS_WARNINGS".ALARMS.UNIT_02.STATION_3_MEASURING."720693" )
   END_RUNG
   // the same network as SCL:
   "DB16000_OPC_UA_TRIGGER_ALARM".CLIENT.U2_STA3_MEAS.ALARMS.COMPUTER_RELEASE_METHOD_LIST_A := ("DB16236_RELEASE_METHOD_LIST_U2_STA3_MEAS".Error OR ("DB16000_OPC_UA_TRIGGER_ALARM".CLIENT.U2_STA3_MEAS.ALARMS.COMPUTER_RELEASE_METHOD_LIST_A AND NOT "DB2120_MPP_ITC_IPC".RESET_FAULTS)) AND "DB7256_UNIT_2_STA_3_MEAS_ENABLE_DISABLE".ENABLED;
   "DB426_ALARMS_WARNINGS".ALARMS.UNIT_02.STATION_3_MEASURING."720693" := "DB16000_OPC_UA_TRIGGER_ALARM".CLIENT.U2_STA3_MEAS.ALARMS.COMPUTER_RELEASE_METHOD_LIST_A;
END_REGION

REGION Network 51: UNIT 2 STATION 3 MEASURING COMPUTER DISCONNECT ALARM
   RUNG wire#powerrail
      Contact( "DB16237_DISCONNECT_U2_STA3_MEAS".Error )
      wire#w1
      Contact( "DB7256_UNIT_2_STA_3_MEAS_ENABLE_DISABLE".ENABLED )
      wire#w2
      Coil( "DB16000_OPC_UA_TRIGGER_ALARM".CLIENT.U2_STA3_MEAS.ALARMS.COMPUTER_DISCONNECT_A )
   END_RUNG
   RUNG wire#powerrail
      Contact( "DB16000_OPC_UA_TRIGGER_ALARM".CLIENT.U2_STA3_MEAS.ALARMS.COMPUTER_DISCONNECT_A )
      I_Contact( "DB2120_MPP_ITC_IPC".RESET_FAULTS )
   END_RUNG wire#w1
   RUNG wire#w2
      Coil( "DB426_ALARMS_WARNINGS".ALARMS.UNIT_02.STATION_3_MEASURING."720694" )
   END_RUNG
   // the same network as SCL:
   "DB16000_OPC_UA_TRIGGER_ALARM".CLIENT.U2_STA3_MEAS.ALARMS.COMPUTER_DISCONNECT_A := ("DB16237_DISCONNECT_U2_STA3_MEAS".Error OR ("DB16000_OPC_UA_TRIGGER_ALARM".CLIENT.U2_STA3_MEAS.ALARMS.COMPUTER_DISCONNECT_A AND NOT "DB2120_MPP_ITC_IPC".RESET_FAULTS)) AND "DB7256_UNIT_2_STA_3_MEAS_ENABLE_DISABLE".ENABLED;
   "DB426_ALARMS_WARNINGS".ALARMS.UNIT_02.STATION_3_MEASURING."720694" := "DB16000_OPC_UA_TRIGGER_ALARM".CLIENT.U2_STA3_MEAS.ALARMS.COMPUTER_DISCONNECT_A;
END_REGION

REGION Network 52: UNIT 2 STATION 3 MEASURING MEASURING NOOZLE SURFACE DISTANCE METHOD CONNECTION ALARM
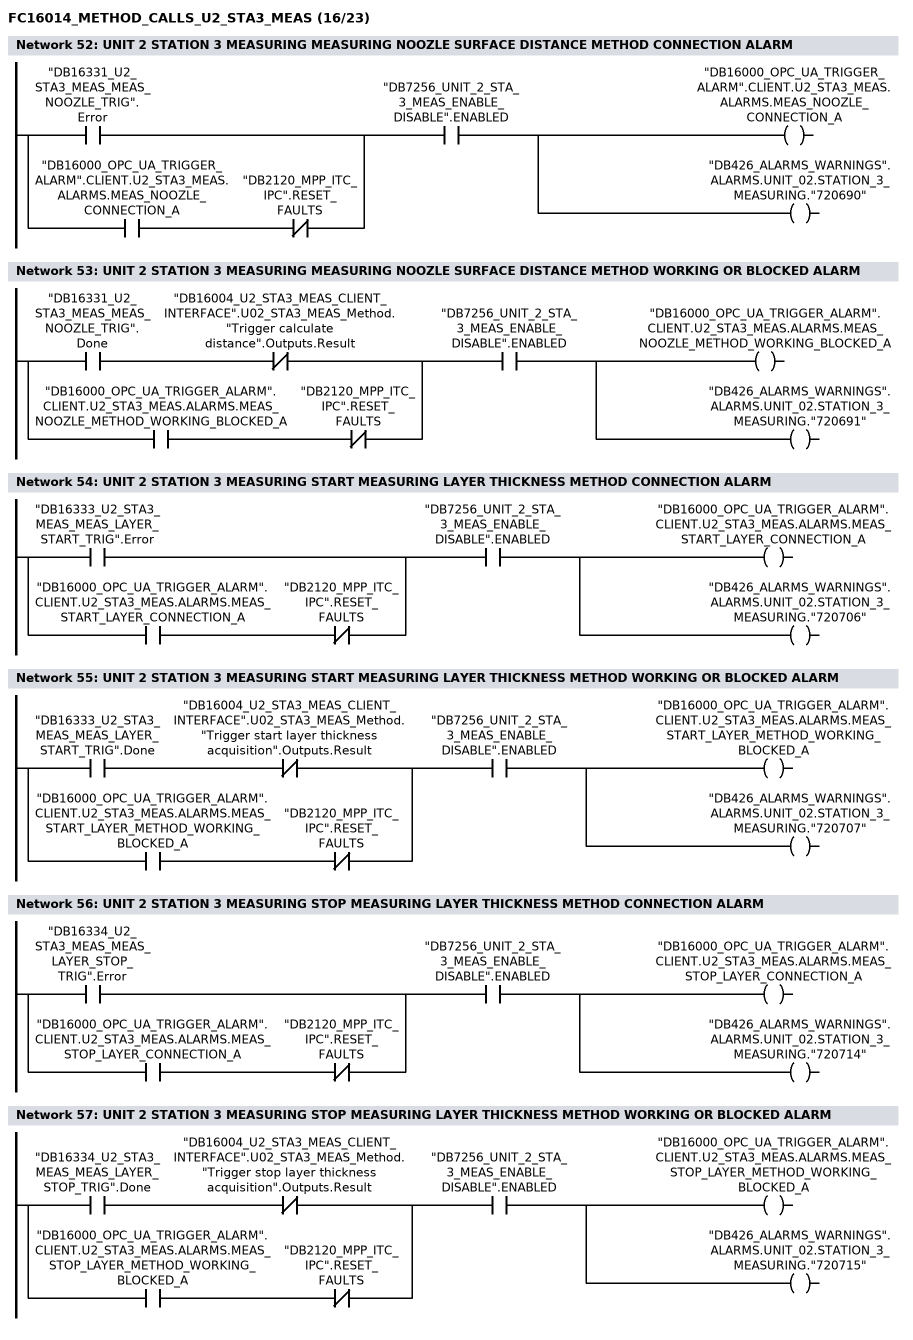
   RUNG wire#powerrail
      Contact( "DB16331_U2_STA3_MEAS_MEAS_NOOZLE_TRIG".Error )
      wire#w1
      Contact( "DB7256_UNIT_2_STA_3_MEAS_ENABLE_DISABLE".ENABLED )
      wire#w2
      Coil( "DB16000_OPC_UA_TRIGGER_ALARM".CLIENT.U2_STA3_MEAS.ALARMS.MEAS_NOOZLE_CONNECTION_A )
   END_RUNG
   RUNG wire#powerrail
      Contact( "DB16000_OPC_UA_TRIGGER_ALARM".CLIENT.U2_STA3_MEAS.ALARMS.MEAS_NOOZLE_CONNECTION_A )
      I_Contact( "DB2120_MPP_ITC_IPC".RESET_FAULTS )
   END_RUNG wire#w1
   RUNG wire#w2
      Coil( "DB426_ALARMS_WARNINGS".ALARMS.UNIT_02.STATION_3_MEASURING."720690" )
   END_RUNG
   // the same network as SCL:
   "DB16000_OPC_UA_TRIGGER_ALARM".CLIENT.U2_STA3_MEAS.ALARMS.MEAS_NOOZLE_CONNECTION_A := ("DB16331_U2_STA3_MEAS_MEAS_NOOZLE_TRIG".Error OR ("DB16000_OPC_UA_TRIGGER_ALARM".CLIENT.U2_STA3_MEAS.ALARMS.MEAS_NOOZLE_CONNECTION_A AND NOT "DB2120_MPP_ITC_IPC".RESET_FAULTS)) AND "DB7256_UNIT_2_STA_3_MEAS_ENABLE_DISABLE".ENABLED;
   "DB426_ALARMS_WARNINGS".ALARMS.UNIT_02.STATION_3_MEASURING."720690" := "DB16000_OPC_UA_TRIGGER_ALARM".CLIENT.U2_STA3_MEAS.ALARMS.MEAS_NOOZLE_CONNECTION_A;
END_REGION

REGION Network 53: UNIT 2 STATION 3 MEASURING MEASURING NOOZLE SURFACE DISTANCE METHOD WORKING OR BLOCKED ALARM
   RUNG wire#powerrail
      Contact( "DB16331_U2_STA3_MEAS_MEAS_NOOZLE_TRIG".Done )
      I_Contact( "DB16004_U2_STA3_MEAS_CLIENT_INTERFACE".U02_STA3_MEAS_Method."Trigger calculate distance".Outputs.Result )
      wire#w1
      Contact( "DB7256_UNIT_2_STA_3_MEAS_ENABLE_DISABLE".ENABLED )
      wire#w2
      Coil( "DB16000_OPC_UA_TRIGGER_ALARM".CLIENT.U2_STA3_MEAS.ALARMS.MEAS_NOOZLE_METHOD_WORKING_BLOCKED_A )
   END_RUNG
   RUNG wire#powerrail
      Contact( "DB16000_OPC_UA_TRIGGER_ALARM".CLIENT.U2_STA3_MEAS.ALARMS.MEAS_NOOZLE_METHOD_WORKING_BLOCKED_A )
      I_Contact( "DB2120_MPP_ITC_IPC".RESET_FAULTS )
   END_RUNG wire#w1
   RUNG wire#w2
      Coil( "DB426_ALARMS_WARNINGS".ALARMS.UNIT_02.STATION_3_MEASURING."720691" )
   END_RUNG
   // the same network as SCL:
   "DB16000_OPC_UA_TRIGGER_ALARM".CLIENT.U2_STA3_MEAS.ALARMS.MEAS_NOOZLE_METHOD_WORKING_BLOCKED_A := (("DB16331_U2_STA3_MEAS_MEAS_NOOZLE_TRIG".Done AND NOT "DB16004_U2_STA3_MEAS_CLIENT_INTERFACE".U02_STA3_MEAS_Method."Trigger calculate distance".Outputs.Result) OR ("DB16000_OPC_UA_TRIGGER_ALARM".CLIENT.U2_STA3_MEAS.ALARMS.MEAS_NOOZLE_METHOD_WORKING_BLOCKED_A AND NOT "DB2120_MPP_ITC_IPC".RESET_FAULTS)) AND "DB7256_UNIT_2_STA_3_MEAS_ENABLE_DISABLE".ENABLED;
   "DB426_ALARMS_WARNINGS".ALARMS.UNIT_02.STATION_3_MEASURING."720691" := "DB16000_OPC_UA_TRIGGER_ALARM".CLIENT.U2_STA3_MEAS.ALARMS.MEAS_NOOZLE_METHOD_WORKING_BLOCKED_A;
END_REGION

REGION Network 54: UNIT 2 STATION 3 MEASURING START MEASURING LAYER THICKNESS METHOD CONNECTION ALARM
   RUNG wire#powerrail
      Contact( "DB16333_U2_STA3_MEAS_MEAS_LAYER_START_TRIG".Error )
      wire#w1
      Contact( "DB7256_UNIT_2_STA_3_MEAS_ENABLE_DISABLE".ENABLED )
      wire#w2
      Coil( "DB16000_OPC_UA_TRIGGER_ALARM".CLIENT.U2_STA3_MEAS.ALARMS.MEAS_START_LAYER_CONNECTION_A )
   END_RUNG
   RUNG wire#powerrail
      Contact( "DB16000_OPC_UA_TRIGGER_ALARM".CLIENT.U2_STA3_MEAS.ALARMS.MEAS_START_LAYER_CONNECTION_A )
      I_Contact( "DB2120_MPP_ITC_IPC".RESET_FAULTS )
   END_RUNG wire#w1
   RUNG wire#w2
      Coil( "DB426_ALARMS_WARNINGS".ALARMS.UNIT_02.STATION_3_MEASURING."720706" )
   END_RUNG
   // the same network as SCL:
   "DB16000_OPC_UA_TRIGGER_ALARM".CLIENT.U2_STA3_MEAS.ALARMS.MEAS_START_LAYER_CONNECTION_A := ("DB16333_U2_STA3_MEAS_MEAS_LAYER_START_TRIG".Error OR ("DB16000_OPC_UA_TRIGGER_ALARM".CLIENT.U2_STA3_MEAS.ALARMS.MEAS_START_LAYER_CONNECTION_A AND NOT "DB2120_MPP_ITC_IPC".RESET_FAULTS)) AND "DB7256_UNIT_2_STA_3_MEAS_ENABLE_DISABLE".ENABLED;
   "DB426_ALARMS_WARNINGS".ALARMS.UNIT_02.STATION_3_MEASURING."720706" := "DB16000_OPC_UA_TRIGGER_ALARM".CLIENT.U2_STA3_MEAS.ALARMS.MEAS_START_LAYER_CONNECTION_A;
END_REGION

REGION Network 55: UNIT 2 STATION 3 MEASURING START MEASURING LAYER THICKNESS METHOD WORKING OR BLOCKED ALARM
   RUNG wire#powerrail
      Contact( "DB16333_U2_STA3_MEAS_MEAS_LAYER_START_TRIG".Done )
      I_Contact( "DB16004_U2_STA3_MEAS_CLIENT_INTERFACE".U02_STA3_MEAS_Method."Trigger start layer thickness acquisition".Outputs.Result )
      wire#w1
      Contact( "DB7256_UNIT_2_STA_3_MEAS_ENABLE_DISABLE".ENABLED )
      wire#w2
      Coil( "DB16000_OPC_UA_TRIGGER_ALARM".CLIENT.U2_STA3_MEAS.ALARMS.MEAS_START_LAYER_METHOD_WORKING_BLOCKED_A )
   END_RUNG
   RUNG wire#powerrail
      Contact( "DB16000_OPC_UA_TRIGGER_ALARM".CLIENT.U2_STA3_MEAS.ALARMS.MEAS_START_LAYER_METHOD_WORKING_BLOCKED_A )
      I_Contact( "DB2120_MPP_ITC_IPC".RESET_FAULTS )
   END_RUNG wire#w1
   RUNG wire#w2
      Coil( "DB426_ALARMS_WARNINGS".ALARMS.UNIT_02.STATION_3_MEASURING."720707" )
   END_RUNG
   // the same network as SCL:
   "DB16000_OPC_UA_TRIGGER_ALARM".CLIENT.U2_STA3_MEAS.ALARMS.MEAS_START_LAYER_METHOD_WORKING_BLOCKED_A := (("DB16333_U2_STA3_MEAS_MEAS_LAYER_START_TRIG".Done AND NOT "DB16004_U2_STA3_MEAS_CLIENT_INTERFACE".U02_STA3_MEAS_Method."Trigger start layer thickness acquisition".Outputs.Result) OR ("DB16000_OPC_UA_TRIGGER_ALARM".CLIENT.U2_STA3_MEAS.ALARMS.MEAS_START_LAYER_METHOD_WORKING_BLOCKED_A AND NOT "DB2120_MPP_ITC_IPC".RESET_FAULTS)) AND "DB7256_UNIT_2_STA_3_MEAS_ENABLE_DISABLE".ENABLED;
   "DB426_ALARMS_WARNINGS".ALARMS.UNIT_02.STATION_3_MEASURING."720707" := "DB16000_OPC_UA_TRIGGER_ALARM".CLIENT.U2_STA3_MEAS.ALARMS.MEAS_START_LAYER_METHOD_WORKING_BLOCKED_A;
END_REGION

REGION Network 56: UNIT 2 STATION 3 MEASURING STOP MEASURING LAYER THICKNESS METHOD CONNECTION ALARM
   RUNG wire#powerrail
      Contact( "DB16334_U2_STA3_MEAS_MEAS_LAYER_STOP_TRIG".Error )
      wire#w1
      Contact( "DB7256_UNIT_2_STA_3_MEAS_ENABLE_DISABLE".ENABLED )
      wire#w2
      Coil( "DB16000_OPC_UA_TRIGGER_ALARM".CLIENT.U2_STA3_MEAS.ALARMS.MEAS_STOP_LAYER_CONNECTION_A )
   END_RUNG
   RUNG wire#powerrail
      Contact( "DB16000_OPC_UA_TRIGGER_ALARM".CLIENT.U2_STA3_MEAS.ALARMS.MEAS_STOP_LAYER_CONNECTION_A )
      I_Contact( "DB2120_MPP_ITC_IPC".RESET_FAULTS )
   END_RUNG wire#w1
   RUNG wire#w2
      Coil( "DB426_ALARMS_WARNINGS".ALARMS.UNIT_02.STATION_3_MEASURING."720714" )
   END_RUNG
   // the same network as SCL:
   "DB16000_OPC_UA_TRIGGER_ALARM".CLIENT.U2_STA3_MEAS.ALARMS.MEAS_STOP_LAYER_CONNECTION_A := ("DB16334_U2_STA3_MEAS_MEAS_LAYER_STOP_TRIG".Error OR ("DB16000_OPC_UA_TRIGGER_ALARM".CLIENT.U2_STA3_MEAS.ALARMS.MEAS_STOP_LAYER_CONNECTION_A AND NOT "DB2120_MPP_ITC_IPC".RESET_FAULTS)) AND "DB7256_UNIT_2_STA_3_MEAS_ENABLE_DISABLE".ENABLED;
   "DB426_ALARMS_WARNINGS".ALARMS.UNIT_02.STATION_3_MEASURING."720714" := "DB16000_OPC_UA_TRIGGER_ALARM".CLIENT.U2_STA3_MEAS.ALARMS.MEAS_STOP_LAYER_CONNECTION_A;
END_REGION

REGION Network 57: UNIT 2 STATION 3 MEASURING STOP MEASURING LAYER THICKNESS METHOD WORKING OR BLOCKED ALARM
   RUNG wire#powerrail
      Contact( "DB16334_U2_STA3_MEAS_MEAS_LAYER_STOP_TRIG".Done )
      I_Contact( "DB16004_U2_STA3_MEAS_CLIENT_INTERFACE".U02_STA3_MEAS_Method."Trigger stop layer thickness acquisition".Outputs.Result )
      wire#w1
      Contact( "DB7256_UNIT_2_STA_3_MEAS_ENABLE_DISABLE".ENABLED )
      wire#w2
      Coil( "DB16000_OPC_UA_TRIGGER_ALARM".CLIENT.U2_STA3_MEAS.ALARMS.MEAS_STOP_LAYER_METHOD_WORKING_BLOCKED_A )
   END_RUNG
   RUNG wire#powerrail
      Contact( "DB16000_OPC_UA_TRIGGER_ALARM".CLIENT.U2_STA3_MEAS.ALARMS.MEAS_STOP_LAYER_METHOD_WORKING_BLOCKED_A )
      I_Contact( "DB2120_MPP_ITC_IPC".RESET_FAULTS )
   END_RUNG wire#w1
   RUNG wire#w2
      Coil( "DB426_ALARMS_WARNINGS".ALARMS.UNIT_02.STATION_3_MEASURING."720715" )
   END_RUNG
   // the same network as SCL:
   "DB16000_OPC_UA_TRIGGER_ALARM".CLIENT.U2_STA3_MEAS.ALARMS.MEAS_STOP_LAYER_METHOD_WORKING_BLOCKED_A := (("DB16334_U2_STA3_MEAS_MEAS_LAYER_STOP_TRIG".Done AND NOT "DB16004_U2_STA3_MEAS_CLIENT_INTERFACE".U02_STA3_MEAS_Method."Trigger stop layer thickness acquisition".Outputs.Result) OR ("DB16000_OPC_UA_TRIGGER_ALARM".CLIENT.U2_STA3_MEAS.ALARMS.MEAS_STOP_LAYER_METHOD_WORKING_BLOCKED_A AND NOT "DB2120_MPP_ITC_IPC".RESET_FAULTS)) AND "DB7256_UNIT_2_STA_3_MEAS_ENABLE_DISABLE".ENABLED;
   "DB426_ALARMS_WARNINGS".ALARMS.UNIT_02.STATION_3_MEASURING."720715" := "DB16000_OPC_UA_TRIGGER_ALARM".CLIENT.U2_STA3_MEAS.ALARMS.MEAS_STOP_LAYER_METHOD_WORKING_BLOCKED_A;
END_REGION

REGION Network 58: UNIT 2 STATION 3 MEASURING CALIBRATING METHOD CONNECTION ALARM
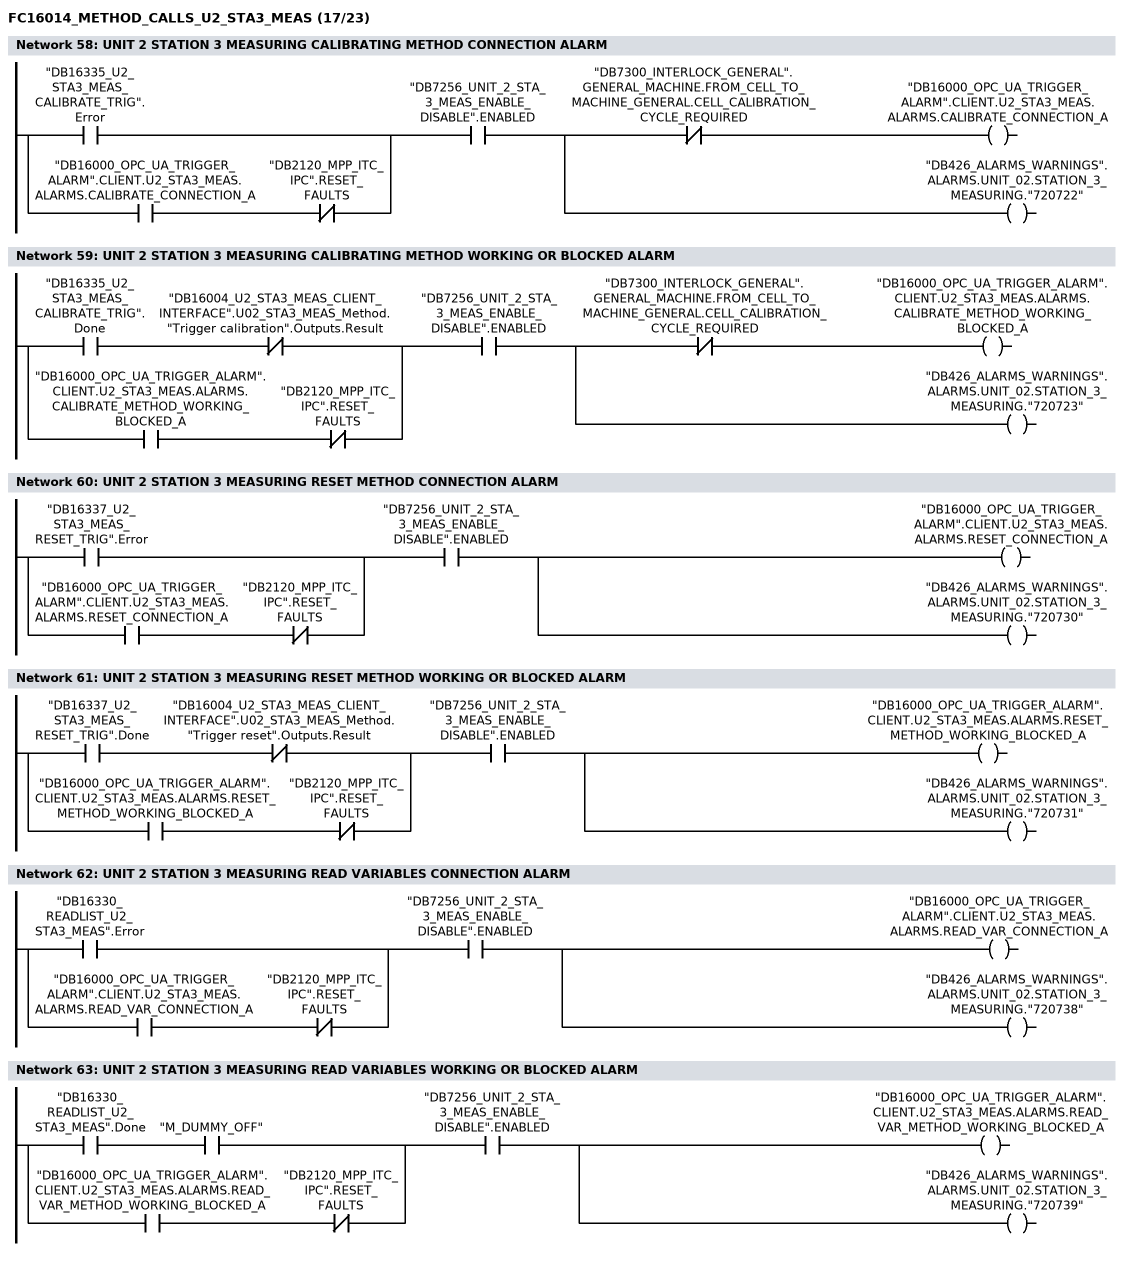
   RUNG wire#powerrail
      Contact( "DB16335_U2_STA3_MEAS_CALIBRATE_TRIG".Error )
      wire#w1
      Contact( "DB7256_UNIT_2_STA_3_MEAS_ENABLE_DISABLE".ENABLED )
      wire#w2
      I_Contact( "DB7300_INTERLOCK_GENERAL".GENERAL_MACHINE.FROM_CELL_TO_MACHINE_GENERAL.CELL_CALIBRATION_CYCLE_REQUIRED )
      Coil( "DB16000_OPC_UA_TRIGGER_ALARM".CLIENT.U2_STA3_MEAS.ALARMS.CALIBRATE_CONNECTION_A )
   END_RUNG
   RUNG wire#powerrail
      Contact( "DB16000_OPC_UA_TRIGGER_ALARM".CLIENT.U2_STA3_MEAS.ALARMS.CALIBRATE_CONNECTION_A )
      I_Contact( "DB2120_MPP_ITC_IPC".RESET_FAULTS )
   END_RUNG wire#w1
   RUNG wire#w2
      Coil( "DB426_ALARMS_WARNINGS".ALARMS.UNIT_02.STATION_3_MEASURING."720722" )
   END_RUNG
   // the same network as SCL:
   #_w1 := ("DB16335_U2_STA3_MEAS_CALIBRATE_TRIG".Error OR ("DB16000_OPC_UA_TRIGGER_ALARM".CLIENT.U2_STA3_MEAS.ALARMS.CALIBRATE_CONNECTION_A AND NOT "DB2120_MPP_ITC_IPC".RESET_FAULTS)) AND "DB7256_UNIT_2_STA_3_MEAS_ENABLE_DISABLE".ENABLED;
   "DB16000_OPC_UA_TRIGGER_ALARM".CLIENT.U2_STA3_MEAS.ALARMS.CALIBRATE_CONNECTION_A := #_w1 AND NOT "DB7300_INTERLOCK_GENERAL".GENERAL_MACHINE.FROM_CELL_TO_MACHINE_GENERAL.CELL_CALIBRATION_CYCLE_REQUIRED;
   "DB426_ALARMS_WARNINGS".ALARMS.UNIT_02.STATION_3_MEASURING."720722" := #_w1;
END_REGION

REGION Network 59: UNIT 2 STATION 3 MEASURING CALIBRATING METHOD WORKING OR BLOCKED ALARM
   RUNG wire#powerrail
      Contact( "DB16335_U2_STA3_MEAS_CALIBRATE_TRIG".Done )
      I_Contact( "DB16004_U2_STA3_MEAS_CLIENT_INTERFACE".U02_STA3_MEAS_Method."Trigger calibration".Outputs.Result )
      wire#w1
      Contact( "DB7256_UNIT_2_STA_3_MEAS_ENABLE_DISABLE".ENABLED )
      wire#w2
      I_Contact( "DB7300_INTERLOCK_GENERAL".GENERAL_MACHINE.FROM_CELL_TO_MACHINE_GENERAL.CELL_CALIBRATION_CYCLE_REQUIRED )
      Coil( "DB16000_OPC_UA_TRIGGER_ALARM".CLIENT.U2_STA3_MEAS.ALARMS.CALIBRATE_METHOD_WORKING_BLOCKED_A )
   END_RUNG
   RUNG wire#powerrail
      Contact( "DB16000_OPC_UA_TRIGGER_ALARM".CLIENT.U2_STA3_MEAS.ALARMS.CALIBRATE_METHOD_WORKING_BLOCKED_A )
      I_Contact( "DB2120_MPP_ITC_IPC".RESET_FAULTS )
   END_RUNG wire#w1
   RUNG wire#w2
      Coil( "DB426_ALARMS_WARNINGS".ALARMS.UNIT_02.STATION_3_MEASURING."720723" )
   END_RUNG
   // the same network as SCL:
   #_w1 := (("DB16335_U2_STA3_MEAS_CALIBRATE_TRIG".Done AND NOT "DB16004_U2_STA3_MEAS_CLIENT_INTERFACE".U02_STA3_MEAS_Method."Trigger calibration".Outputs.Result) OR ("DB16000_OPC_UA_TRIGGER_ALARM".CLIENT.U2_STA3_MEAS.ALARMS.CALIBRATE_METHOD_WORKING_BLOCKED_A AND NOT "DB2120_MPP_ITC_IPC".RESET_FAULTS)) AND "DB7256_UNIT_2_STA_3_MEAS_ENABLE_DISABLE".ENABLED;
   "DB16000_OPC_UA_TRIGGER_ALARM".CLIENT.U2_STA3_MEAS.ALARMS.CALIBRATE_METHOD_WORKING_BLOCKED_A := #_w1 AND NOT "DB7300_INTERLOCK_GENERAL".GENERAL_MACHINE.FROM_CELL_TO_MACHINE_GENERAL.CELL_CALIBRATION_CYCLE_REQUIRED;
   "DB426_ALARMS_WARNINGS".ALARMS.UNIT_02.STATION_3_MEASURING."720723" := #_w1;
END_REGION

REGION Network 60: UNIT 2 STATION 3 MEASURING RESET METHOD CONNECTION ALARM
   RUNG wire#powerrail
      Contact( "DB16337_U2_STA3_MEAS_RESET_TRIG".Error )
      wire#w1
      Contact( "DB7256_UNIT_2_STA_3_MEAS_ENABLE_DISABLE".ENABLED )
      wire#w2
      Coil( "DB16000_OPC_UA_TRIGGER_ALARM".CLIENT.U2_STA3_MEAS.ALARMS.RESET_CONNECTION_A )
   END_RUNG
   RUNG wire#powerrail
      Contact( "DB16000_OPC_UA_TRIGGER_ALARM".CLIENT.U2_STA3_MEAS.ALARMS.RESET_CONNECTION_A )
      I_Contact( "DB2120_MPP_ITC_IPC".RESET_FAULTS )
   END_RUNG wire#w1
   RUNG wire#w2
      Coil( "DB426_ALARMS_WARNINGS".ALARMS.UNIT_02.STATION_3_MEASURING."720730" )
   END_RUNG
   // the same network as SCL:
   "DB16000_OPC_UA_TRIGGER_ALARM".CLIENT.U2_STA3_MEAS.ALARMS.RESET_CONNECTION_A := ("DB16337_U2_STA3_MEAS_RESET_TRIG".Error OR ("DB16000_OPC_UA_TRIGGER_ALARM".CLIENT.U2_STA3_MEAS.ALARMS.RESET_CONNECTION_A AND NOT "DB2120_MPP_ITC_IPC".RESET_FAULTS)) AND "DB7256_UNIT_2_STA_3_MEAS_ENABLE_DISABLE".ENABLED;
   "DB426_ALARMS_WARNINGS".ALARMS.UNIT_02.STATION_3_MEASURING."720730" := "DB16000_OPC_UA_TRIGGER_ALARM".CLIENT.U2_STA3_MEAS.ALARMS.RESET_CONNECTION_A;
END_REGION

